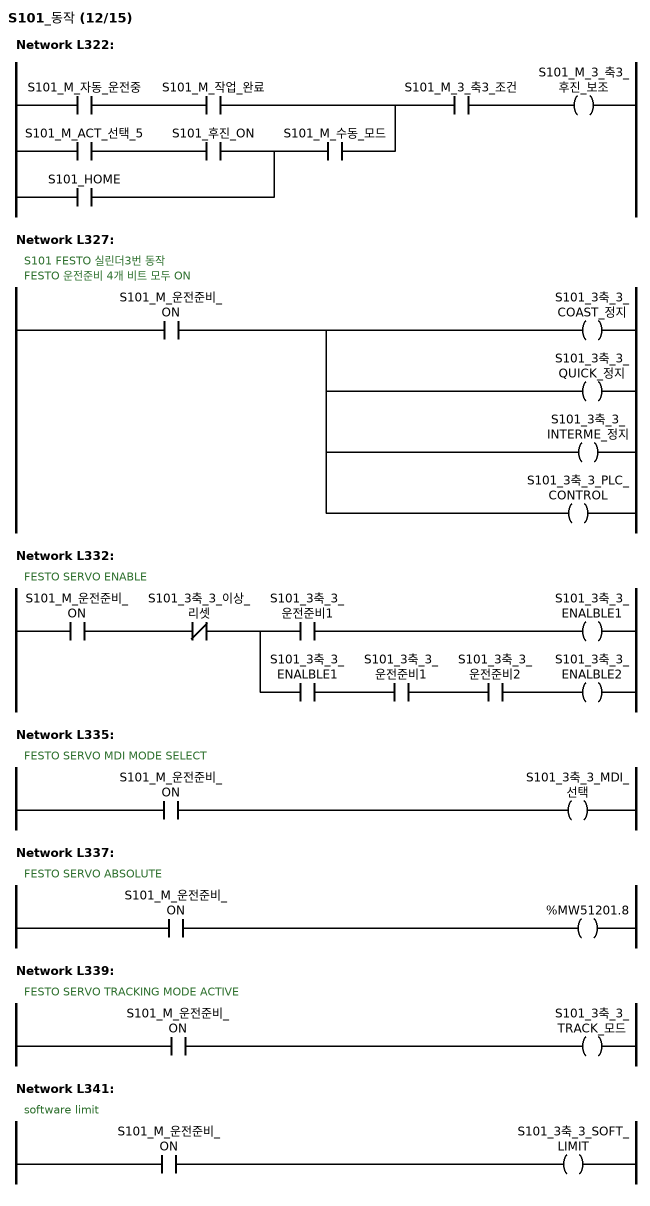
(* [picture p72: S101_동작 rungs L322-L341] *)
(* Rung L322 *)
S101_M_3_축3_후진_보조 := ((S101_M_자동_운전중 AND S101_M_작업_완료) OR (((S101_M_ACT_선택_5 AND S101_후진_ON) OR S101_HOME) AND S101_M_수동_모드)) AND S101_M_3_축3_조건;
(* S101 FESTO 실린더3번 동작 *)
(* FESTO 운전준비 4개 비트 모두 ON *)
(* Rung L327 *)
S101_3축_3_COAST_정지 := S101_M_운전준비_ON;
S101_3축_3_QUICK_정지 := S101_M_운전준비_ON;
S101_3축_3_INTERME_정지 := S101_M_운전준비_ON;
S101_3축_3_PLC_CONTROL := S101_M_운전준비_ON;
(* FESTO SERVO ENABLE *)
(* Rung L332 *)
S101_3축_3_ENALBLE1 := S101_M_운전준비_ON AND NOT S101_3축_3_이상_리셋 AND S101_3축_3_운전준비1;
S101_3축_3_ENALBLE2 := S101_M_운전준비_ON AND NOT S101_3축_3_이상_리셋 AND S101_3축_3_ENALBLE1 AND S101_3축_3_운전준비1 AND S101_3축_3_운전준비2;
(* FESTO SERVO MDI MODE SELECT *)
(* Rung L335 *)
S101_3축_3_MDI_선택 := S101_M_운전준비_ON;
(* FESTO SERVO ABSOLUTE *)
(* Rung L337 *)
%MW51201.8 := S101_M_운전준비_ON;
(* FESTO SERVO TRACKING MODE ACTIVE *)
(* Rung L339 *)
S101_3축_3_TRACK_모드 := S101_M_운전준비_ON;
(* software limit *)
(* Rung L341 *)
S101_3축_3_SOFT_LIMIT := S101_M_운전준비_ON;

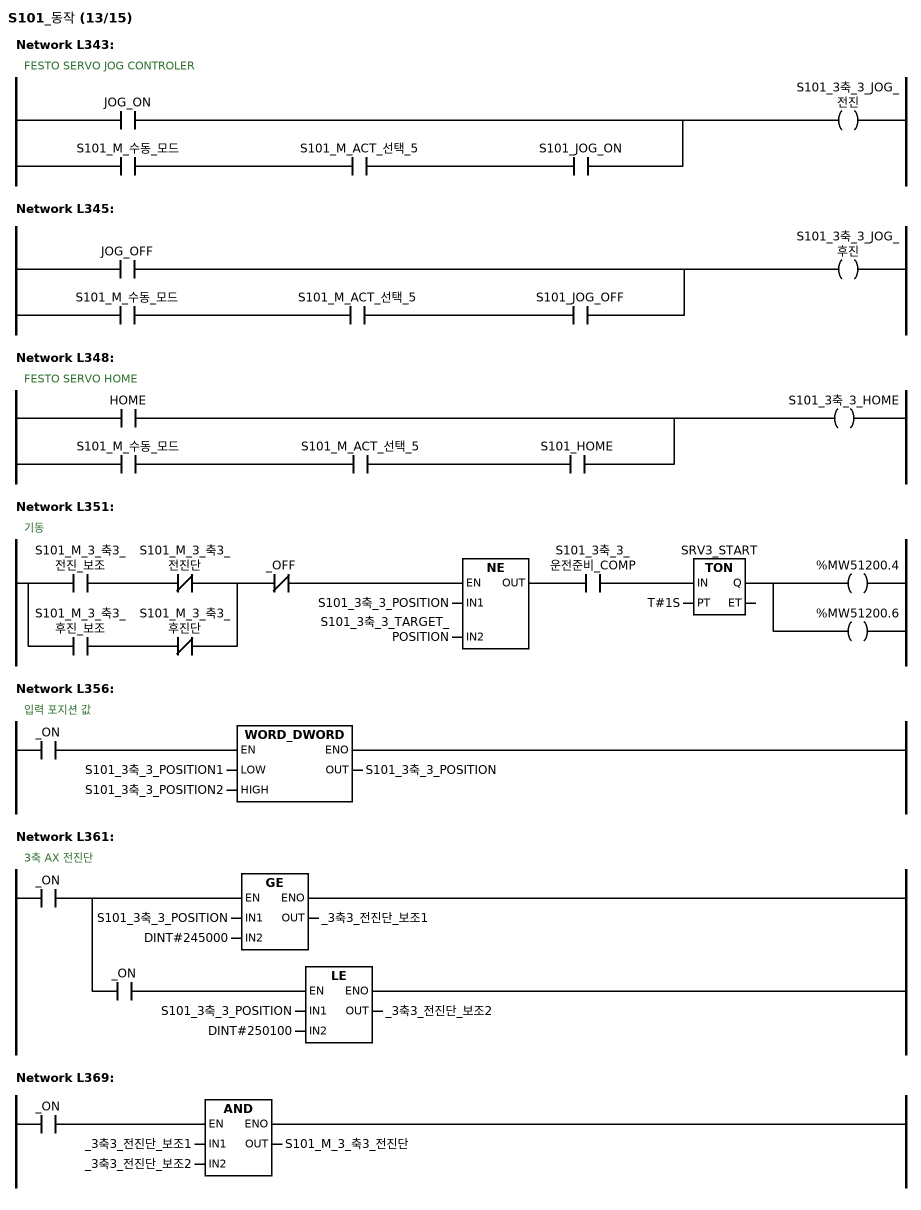
(* FESTO SERVO JOG CONTROLER *)
(* Rung L343 *)
S101_3축_3_JOG_전진 := JOG_ON OR (S101_M_수동_모드 AND S101_M_ACT_선택_5 AND S101_JOG_ON);
(* Rung L345 *)
S101_3축_3_JOG_후진 := JOG_OFF OR (S101_M_수동_모드 AND S101_M_ACT_선택_5 AND S101_JOG_OFF);
(* FESTO SERVO HOME *)
(* Rung L348 *)
S101_3축_3_HOME := HOME OR (S101_M_수동_모드 AND S101_M_ACT_선택_5 AND S101_HOME);
(* 기동 *)
(* Rung L351 *)
IF ((S101_M_3_축3_전진_보조 AND NOT S101_M_3_축3_전진단) OR (S101_M_3_축3_후진_보조 AND NOT S101_M_3_축3_후진단)) AND NOT _OFF THEN
    _t3 := S101_3축_3_POSITION <> S101_3축_3_TARGET_POSITION;
END_IF;
SRV3_START(IN := _t3 AND S101_3축_3_운전준비_COMP, PT := T#1S);
%MW51200.4 := SRV3_START.Q;
%MW51200.6 := SRV3_START.Q;
(* 입력 포지션 값 *)
(* Rung L356 *)
IF _ON THEN
    S101_3축_3_POSITION := WORD_DWORD(LOW := S101_3축_3_POSITION1, HIGH := S101_3축_3_POSITION2);
END_IF;
(* 3축 AX 전진단 *)
(* Rung L361 *)
IF _ON THEN _3축3_전진단_보조1 := S101_3축_3_POSITION >= DINT#245000; END_IF;
IF _ON AND _ON THEN _3축3_전진단_보조2 := S101_3축_3_POSITION <= DINT#250100; END_IF;
(* Rung L369 *)
IF _ON THEN S101_M_3_축3_전진단 := _3축3_전진단_보조1 AND _3축3_전진단_보조2; END_IF;

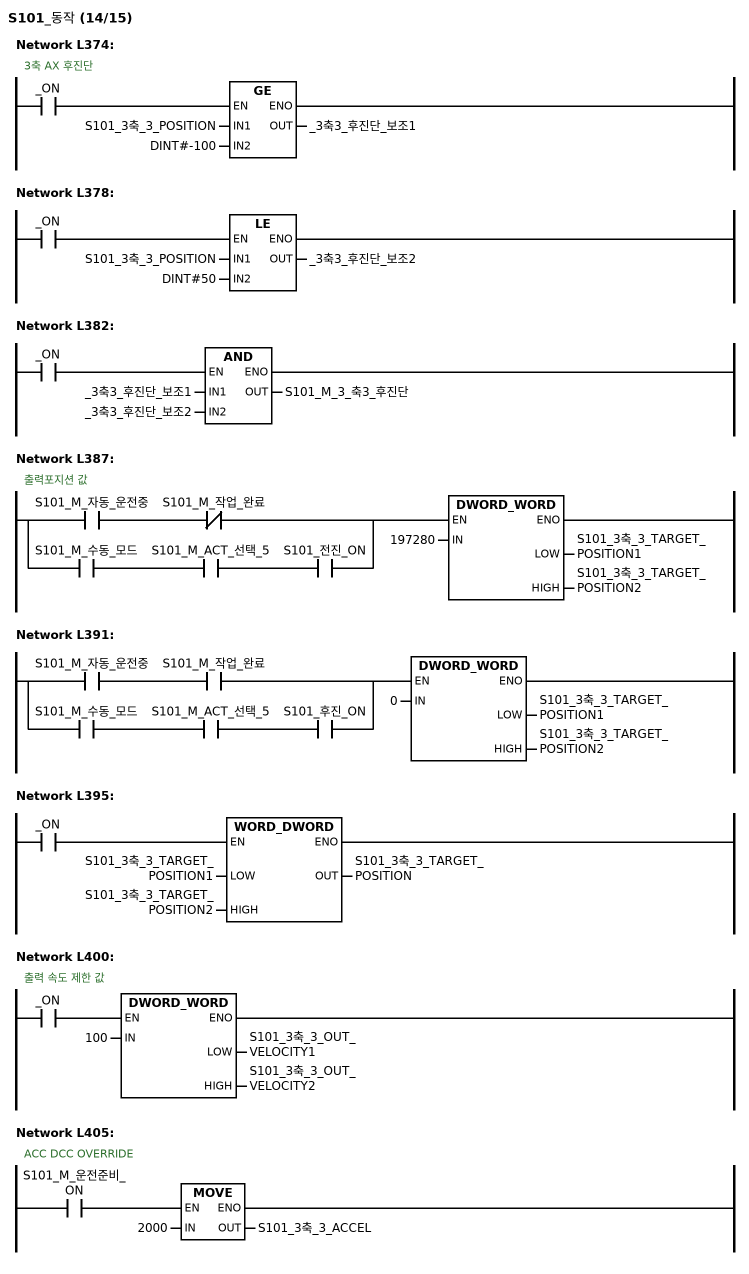
(* 3축 AX 후진단 *)
(* Rung L374 *)
IF _ON THEN _3축3_후진단_보조1 := S101_3축_3_POSITION >= (DINT#-100); END_IF;
(* Rung L378 *)
IF _ON THEN _3축3_후진단_보조2 := S101_3축_3_POSITION <= DINT#50; END_IF;
(* Rung L382 *)
IF _ON THEN S101_M_3_축3_후진단 := _3축3_후진단_보조1 AND _3축3_후진단_보조2; END_IF;
(* 출력포지션 값 *)
(* Rung L387 *)
IF (S101_M_자동_운전중 AND NOT S101_M_작업_완료) OR (S101_M_수동_모드 AND S101_M_ACT_선택_5 AND S101_전진_ON) THEN
    S101_3축_3_TARGET_POSITION1 := DWORD_WORD(IN := 197280, HIGH => S101_3축_3_TARGET_POSITION2);
END_IF;
(* Rung L391 *)
IF (S101_M_자동_운전중 AND S101_M_작업_완료) OR (S101_M_수동_모드 AND S101_M_ACT_선택_5 AND S101_후진_ON) THEN
    S101_3축_3_TARGET_POSITION1 := DWORD_WORD(IN := 0, HIGH => S101_3축_3_TARGET_POSITION2);
END_IF;
(* Rung L395 *)
IF _ON THEN
    S101_3축_3_TARGET_POSITION := WORD_DWORD(LOW := S101_3축_3_TARGET_POSITION1, HIGH := S101_3축_3_TARGET_POSITION2);
END_IF;
(* 출력 속도 제한 값 *)
(* Rung L400 *)
IF _ON THEN S101_3축_3_OUT_VELOCITY1 := DWORD_WORD(IN := 100, HIGH => S101_3축_3_OUT_VELOCITY2); END_IF;
(* ACC DCC OVERRIDE *)
(* Rung L405 *)
IF S101_M_운전준비_ON THEN S101_3축_3_ACCEL := 2000; END_IF;

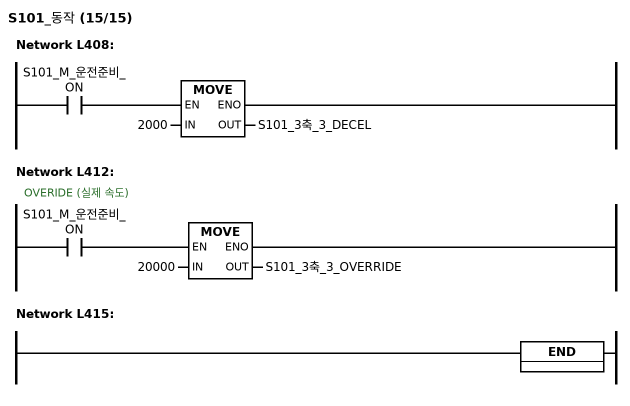
(* Rung L408 *)
IF S101_M_운전준비_ON THEN S101_3축_3_DECEL := 2000; END_IF;
(* OVERIDE (실제 속도) *)
(* Rung L412 *)
IF S101_M_운전준비_ON THEN S101_3축_3_OVERRIDE := 20000; END_IF;
(* Rung L415 *)
END();
END_PROGRAM

PROGRAM S101_LH_APRON_랙방 (* task: 스캔 프로그램 *)
VAR_EXTERNAL
    APRON_LH_RACK1_I_막장감지 : BOOL; (* AT %MW87211.2 *)
    APRON_LH_RACK1_I_종발이감지1 : BOOL; (* AT %MW87211.0 *)
    APRON_LH_RACK1_I_종발이감지2 : BOOL; (* AT %MW87211.1 *)
    APRON_LH_RACK2_I_막장감지 : BOOL; (* AT %MW87211.10 *)
    APRON_LH_RACK2_I_종발이감지1 : BOOL; (* AT %MW87211.8 *)
    APRON_LH_RACK2_I_종발이감지2 : BOOL; (* AT %MW87211.9 *)
    AWAYS_ON : BOOL; (* AT %MW3.1 *)
    OTR_RACK1_I_막장감지 : BOOL; (* AT %MW87020.2 *)
    OTR_RACK1_I_종발이감지1 : BOOL; (* AT %MW87020.0 *)
    OTR_RACK1_I_종발이감지2 : BOOL; (* AT %MW87020.1 *)
    OTR_RACK2_I_막장감지 : BOOL; (* AT %MW87020.10 *)
    OTR_RACK2_I_종발이감지1 : BOOL; (* AT %MW87020.8 *)
    OTR_RACK2_I_종발이감지2 : BOOL; (* AT %MW87020.9 *)
    R101_1_M_RB_PROG_NO : WORD; (* AT %MW20074 *)
    S101_LH_M_APRON_PLT1_FAULT : BOOL; (* AT %MW1200.6 *)
    S101_LH_M_APRON_PLT1_MATCH_OK : BOOL; (* AT %MW1200.5 *)
    S101_LH_M_APRON_PLT1_PLT_NONE : BOOL; (* AT %MW1200.2 *)
    S101_LH_M_APRON_PLT1_PLT_ON : BOOL; (* AT %MW1200.1 *)
    S101_LH_M_APRON_PLT1_PROG_OK : BOOL; (* AT %MW1200.0 *)
    S101_LH_M_APRON_PLT1_로딩완료 : BOOL; (* AT %MW1200.10 *)
    S101_LH_M_APRON_PLT1_제품수량 : WORD; (* AT %MW1224 *)
    S101_LH_M_APRON_PLT1_차종유 : BOOL; (* AT %MW1200.8 *)
    S101_LH_M_APRON_PLT1_차종코드 : WORD; (* AT %MW1216 *)
    S101_LH_M_APRON_PLT1_파트무 : BOOL; (* AT %MW1200.4 *)
    S101_LH_M_APRON_PLT1_파트유 : BOOL; (* AT %MW1200.3 *)
    S101_LH_M_APRON_PLT2_FAULT : BOOL; (* AT %MW1201.6 *)
    S101_LH_M_APRON_PLT2_MATCH_OK : BOOL; (* AT %MW1201.5 *)
    S101_LH_M_APRON_PLT2_PLT_NONE : BOOL; (* AT %MW1201.2 *)
    S101_LH_M_APRON_PLT2_PLT_ON : BOOL; (* AT %MW1201.1 *)
    S101_LH_M_APRON_PLT2_PROG_OK : BOOL; (* AT %MW1201.0 *)
    S101_LH_M_APRON_PLT2_로딩완료 : BOOL; (* AT %MW1201.10 *)
    S101_LH_M_APRON_PLT2_제품수량 : WORD; (* AT %MW1225 *)
    S101_LH_M_APRON_PLT2_차종유 : BOOL; (* AT %MW1201.8 *)
    S101_LH_M_APRON_PLT2_차종코드 : WORD; (* AT %MW1217 *)
    S101_LH_M_APRON_PLT2_파트무 : BOOL; (* AT %MW1201.4 *)
    S101_LH_M_APRON_PLT2_파트유 : BOOL; (* AT %MW1201.3 *)
    전체_M_이상_리셋 : BOOL; (* AT %MW308.2 *) (* 전체 M 이상 리셋 *)
END_VAR
VAR
    INST : TON;
    INST1 : TON;
    INST2 : TON;
    INST3 : TON;
    INST4 : TON;
    INST5 : TON;
    R201_1_M_I_RB_PROG_NO : INT;
    _R101_1_LH_APRON_PLT1_카운터_RST완료 : BOOL;
    _R101_1_LH_APRON_PLT1_카운터_RST요구 : BOOL;
    _R101_1_LH_APRON_PLT2_카운터_RST완료 : BOOL;
    _R101_1_LH_APRON_PLT2_카운터_RST요구 : BOOL;
    _R101_1_LH_PLT1_막장취출완료 : BOOL;
    _R101_1_LH_PLT2_막장취출완료 : BOOL;
    _R101_1_RB_비교_PROG_NO : INT;
    _R201_1_OTR_PLT1_카운터_RST완료 : BOOL;
    _R201_1_OTR_PLT1_카운터_RST요구 : BOOL;
    _R201_1_OTR_PLT2_카운터_RST완료 : BOOL;
    _R201_1_OTR_PLT2_카운터_RST요구 : BOOL;
    _R201_1_PLT1_막장취출완료 : BOOL;
    _R201_1_PLT2_막장취출완료 : BOOL;
    _R201_1_RB_비교_PROG_NO : INT;
    _R201_1_RB_비교_PROG_NO_INT : INT;
    _R201_1_막장취출완료 : BOOL;
    _랙1_제품수량 : INT;
    _랙1_차종코드 : INT;
    _랙2_제품수량 : INT;
    _랙2_차종코드 : INT;
END_VAR
VAR
    _p1 : BOOL;
    _p2 : BOOL;
END_VAR

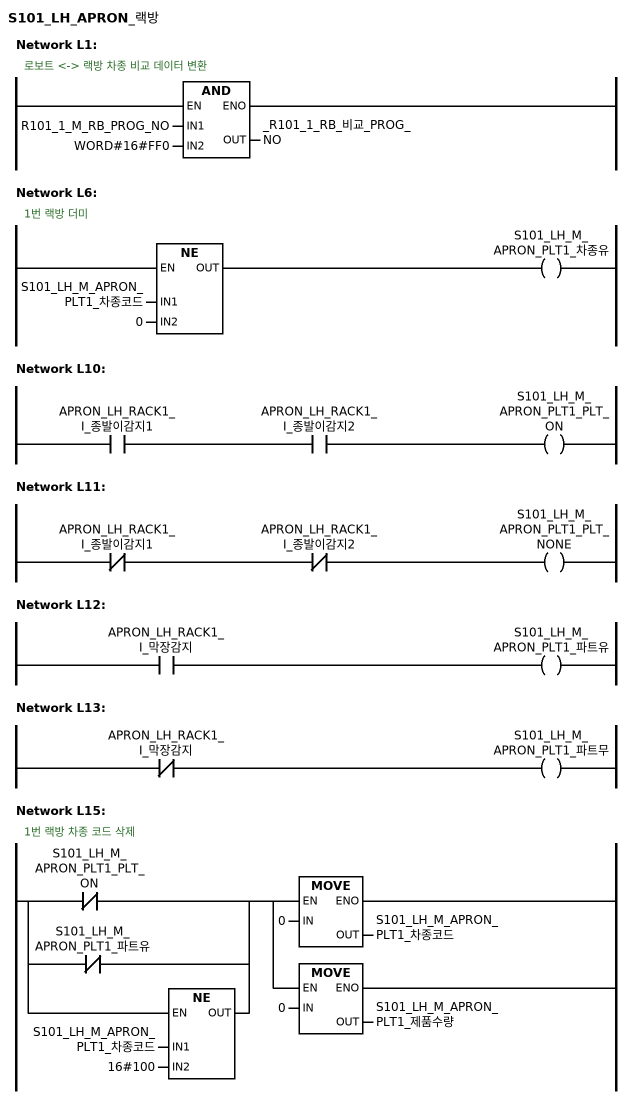
(* 로보트 <-> 랙방 차종 비교 데이터 변환 *)
(* Rung L1 *)
_R101_1_RB_비교_PROG_NO := R101_1_M_RB_PROG_NO AND WORD#16#FF0;
(* 1번 랙방 더미 *)
(* Rung L6 *)
S101_LH_M_APRON_PLT1_차종유 := S101_LH_M_APRON_PLT1_차종코드 <> 0;
(* Rung L10 *)
S101_LH_M_APRON_PLT1_PLT_ON := APRON_LH_RACK1_I_종발이감지1 AND APRON_LH_RACK1_I_종발이감지2;
(* Rung L11 *)
S101_LH_M_APRON_PLT1_PLT_NONE := NOT APRON_LH_RACK1_I_종발이감지1 AND NOT APRON_LH_RACK1_I_종발이감지2;
(* Rung L12 *)
S101_LH_M_APRON_PLT1_파트유 := APRON_LH_RACK1_I_막장감지;
(* Rung L13 *)
S101_LH_M_APRON_PLT1_파트무 := NOT APRON_LH_RACK1_I_막장감지;
(* 1번 랙방 차종 코드 삭제 *)
(* Rung L15 *)
_p1 := NOT S101_LH_M_APRON_PLT1_PLT_ON OR NOT S101_LH_M_APRON_PLT1_파트유 OR (S101_LH_M_APRON_PLT1_차종코드 <> 16#100);
IF _p1 THEN
    S101_LH_M_APRON_PLT1_차종코드 := 0;
    S101_LH_M_APRON_PLT1_제품수량 := 0;
END_IF;
(* 1번 랙방 차종 코드 입력 *)
(* Rung L22: network not rendered *)
(* not connected or not rendered: S101_LH_M_APRON_PLT1_로딩완료, S101_LH_M_APRON_PLT1_PLT_ON, S101_LH_M_APRON_PLT1_파트유, 16#100, S101_LH_M_APRON_PLT1_차종코드, 10, S101_LH_M_APRON_PLT1_제품수량 *)

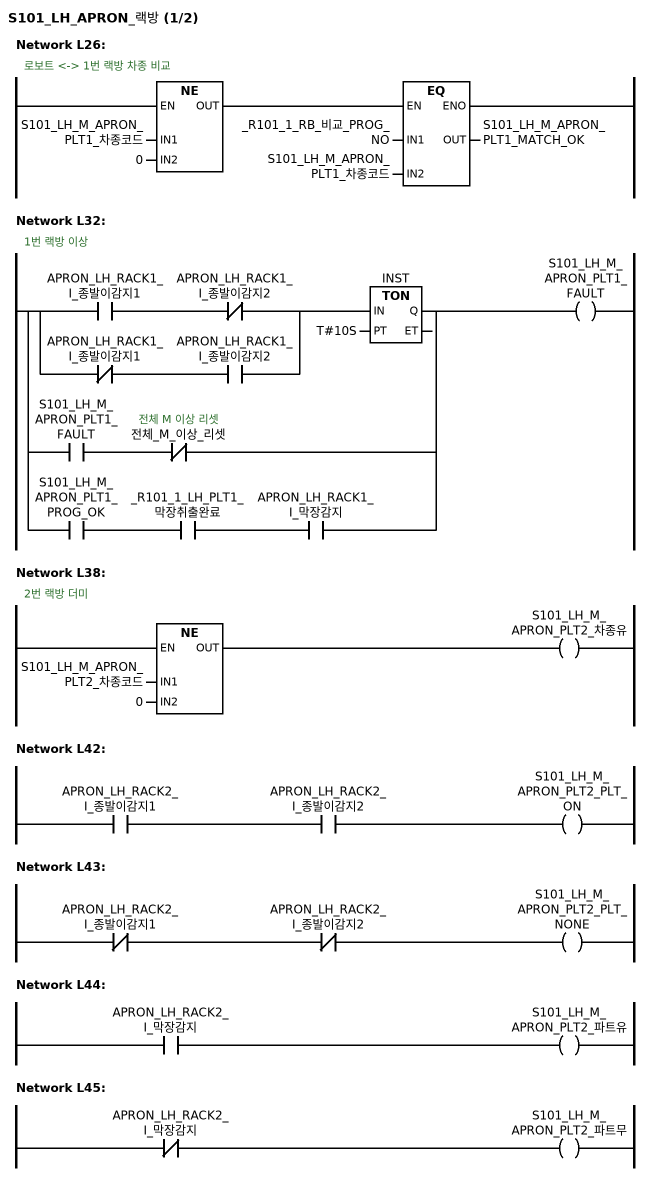
(* 로보트 <-> 1번 랙방 차종 비교 *)
(* Rung L26 *)
IF S101_LH_M_APRON_PLT1_차종코드 <> 0 THEN
    S101_LH_M_APRON_PLT1_MATCH_OK := _R101_1_RB_비교_PROG_NO = S101_LH_M_APRON_PLT1_차종코드;
END_IF;
(* 1번 랙방 이상 *)
(* Rung L32 *)
INST(IN := (APRON_LH_RACK1_I_종발이감지1 AND NOT APRON_LH_RACK1_I_종발이감지2) OR (NOT APRON_LH_RACK1_I_종발이감지1 AND APRON_LH_RACK1_I_종발이감지2), PT := T#10S);
S101_LH_M_APRON_PLT1_FAULT := INST.Q OR (S101_LH_M_APRON_PLT1_FAULT AND NOT 전체_M_이상_리셋) OR (S101_LH_M_APRON_PLT1_PROG_OK AND _R101_1_LH_PLT1_막장취출완료 AND APRON_LH_RACK1_I_막장감지);
(* 2번 랙방 더미 *)
(* Rung L38 *)
S101_LH_M_APRON_PLT2_차종유 := S101_LH_M_APRON_PLT2_차종코드 <> 0;
(* Rung L42 *)
S101_LH_M_APRON_PLT2_PLT_ON := APRON_LH_RACK2_I_종발이감지1 AND APRON_LH_RACK2_I_종발이감지2;
(* Rung L43 *)
S101_LH_M_APRON_PLT2_PLT_NONE := NOT APRON_LH_RACK2_I_종발이감지1 AND NOT APRON_LH_RACK2_I_종발이감지2;
(* Rung L44 *)
S101_LH_M_APRON_PLT2_파트유 := APRON_LH_RACK2_I_막장감지;
(* Rung L45 *)
S101_LH_M_APRON_PLT2_파트무 := NOT APRON_LH_RACK2_I_막장감지;

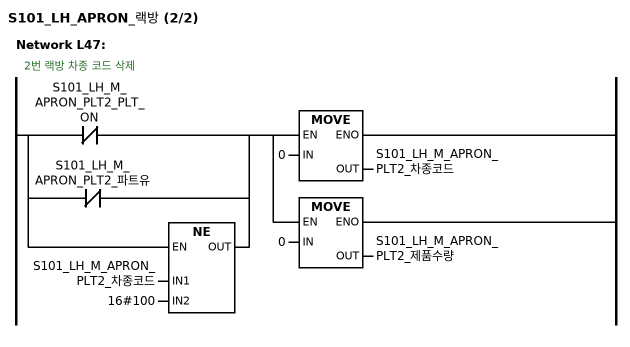
(* 2번 랙방 차종 코드 삭제 *)
(* Rung L47 *)
_p2 := NOT S101_LH_M_APRON_PLT2_PLT_ON OR NOT S101_LH_M_APRON_PLT2_파트유 OR (S101_LH_M_APRON_PLT2_차종코드 <> 16#100);
IF _p2 THEN
    S101_LH_M_APRON_PLT2_차종코드 := 0;
    S101_LH_M_APRON_PLT2_제품수량 := 0;
END_IF;
(* 2번 랙방 차종 코드 입력 *)
(* Rung L54: network not rendered *)
(* not connected or not rendered: S101_LH_M_APRON_PLT2_로딩완료, S101_LH_M_APRON_PLT2_PLT_ON, S101_LH_M_APRON_PLT2_파트유, 16#100, S101_LH_M_APRON_PLT2_차종코드, 10, S101_LH_M_APRON_PLT2_제품수량 *)

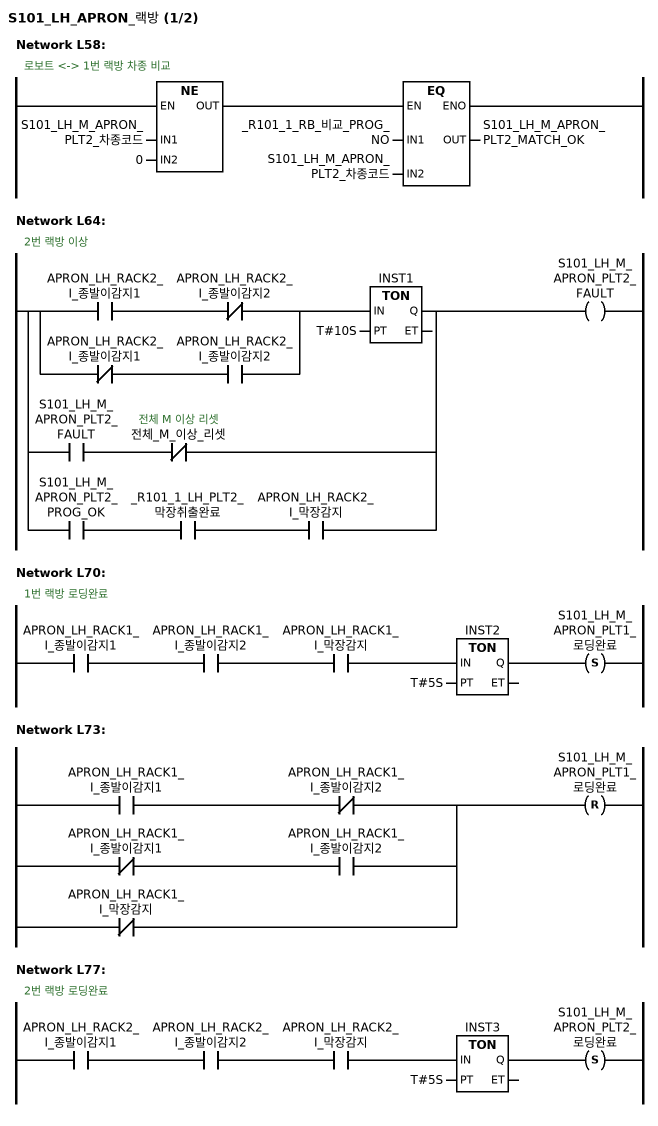
(* 로보트 <-> 1번 랙방 차종 비교 *)
(* Rung L58 *)
IF S101_LH_M_APRON_PLT2_차종코드 <> 0 THEN
    S101_LH_M_APRON_PLT2_MATCH_OK := _R101_1_RB_비교_PROG_NO = S101_LH_M_APRON_PLT2_차종코드;
END_IF;
(* 2번 랙방 이상 *)
(* Rung L64 *)
INST1(IN := (APRON_LH_RACK2_I_종발이감지1 AND NOT APRON_LH_RACK2_I_종발이감지2) OR (NOT APRON_LH_RACK2_I_종발이감지1 AND APRON_LH_RACK2_I_종발이감지2), PT := T#10S);
S101_LH_M_APRON_PLT2_FAULT := INST1.Q OR (S101_LH_M_APRON_PLT2_FAULT AND NOT 전체_M_이상_리셋) OR (S101_LH_M_APRON_PLT2_PROG_OK AND _R101_1_LH_PLT2_막장취출완료 AND APRON_LH_RACK2_I_막장감지);
(* 1번 랙방 로딩완료 *)
(* Rung L70 *)
INST2(IN := APRON_LH_RACK1_I_종발이감지1 AND APRON_LH_RACK1_I_종발이감지2 AND APRON_LH_RACK1_I_막장감지, PT := T#5S);
IF INST2.Q THEN S101_LH_M_APRON_PLT1_로딩완료 := TRUE; END_IF;
(* Rung L73 *)
IF (APRON_LH_RACK1_I_종발이감지1 AND NOT APRON_LH_RACK1_I_종발이감지2) OR (NOT APRON_LH_RACK1_I_종발이감지1 AND APRON_LH_RACK1_I_종발이감지2) OR NOT APRON_LH_RACK1_I_막장감지 THEN
    S101_LH_M_APRON_PLT1_로딩완료 := FALSE;
END_IF;
(* 2번 랙방 로딩완료 *)
(* Rung L77 *)
INST3(IN := APRON_LH_RACK2_I_종발이감지1 AND APRON_LH_RACK2_I_종발이감지2 AND APRON_LH_RACK2_I_막장감지, PT := T#5S);
IF INST3.Q THEN S101_LH_M_APRON_PLT2_로딩완료 := TRUE; END_IF;

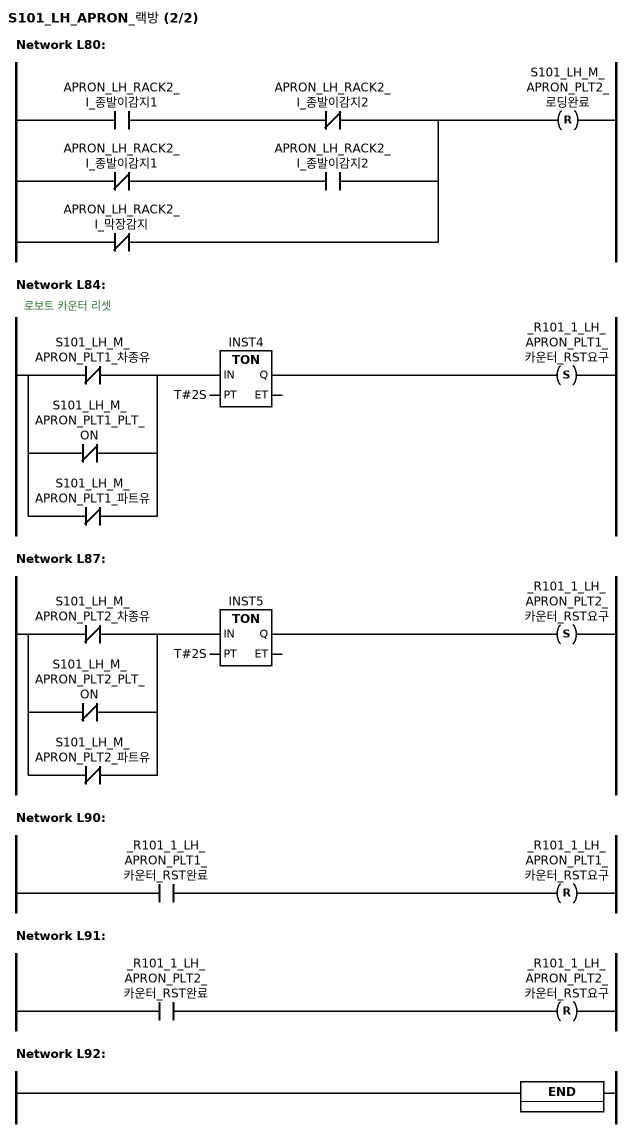
(* Rung L80 *)
IF (APRON_LH_RACK2_I_종발이감지1 AND NOT APRON_LH_RACK2_I_종발이감지2) OR (NOT APRON_LH_RACK2_I_종발이감지1 AND APRON_LH_RACK2_I_종발이감지2) OR NOT APRON_LH_RACK2_I_막장감지 THEN
    S101_LH_M_APRON_PLT2_로딩완료 := FALSE;
END_IF;
(* 로보트 카운터 리셋 *)
(* Rung L84 *)
INST4(IN := NOT S101_LH_M_APRON_PLT1_차종유 OR NOT S101_LH_M_APRON_PLT1_PLT_ON OR NOT S101_LH_M_APRON_PLT1_파트유, PT := T#2S);
IF INST4.Q THEN _R101_1_LH_APRON_PLT1_카운터_RST요구 := TRUE; END_IF;
(* Rung L87 *)
INST5(IN := NOT S101_LH_M_APRON_PLT2_차종유 OR NOT S101_LH_M_APRON_PLT2_PLT_ON OR NOT S101_LH_M_APRON_PLT2_파트유, PT := T#2S);
IF INST5.Q THEN _R101_1_LH_APRON_PLT2_카운터_RST요구 := TRUE; END_IF;
(* Rung L90 *)
IF _R101_1_LH_APRON_PLT1_카운터_RST완료 THEN _R101_1_LH_APRON_PLT1_카운터_RST요구 := FALSE; END_IF;
(* Rung L91 *)
IF _R101_1_LH_APRON_PLT2_카운터_RST완료 THEN _R101_1_LH_APRON_PLT2_카운터_RST요구 := FALSE; END_IF;
(* Rung L92 *)
END();
END_PROGRAM

PROGRAM S101_LH_APRON_랙방_우선순위 (* task: 스캔 프로그램 *)
VAR_EXTERNAL
    S101_LH_M_APRON_PLT1_PLT_ON : BOOL; (* AT %MW1200.1 *)
    S101_LH_M_APRON_PLT1_로딩완료 : BOOL; (* AT %MW1200.10 *)
    S101_LH_M_APRON_PLT1_차종유 : BOOL; (* AT %MW1200.8 *)
    S101_LH_M_APRON_PLT1_파트유 : BOOL; (* AT %MW1200.3 *)
    S101_LH_M_APRON_PLT2_PLT_ON : BOOL; (* AT %MW1201.1 *)
    S101_LH_M_APRON_PLT2_로딩완료 : BOOL; (* AT %MW1201.10 *)
    S101_LH_M_APRON_PLT2_차종유 : BOOL; (* AT %MW1201.8 *)
    S101_LH_M_APRON_PLT2_파트유 : BOOL; (* AT %MW1201.3 *)
    S101_LH_M_APRON_PLT_PRIORITY1 : WORD; (* AT %MW1208 *)
    S101_LH_M_APRON_PLT_PRIORITY2 : WORD; (* AT %MW1209 *)
    S101_LH_M_APRON_PLT_PRIORITY3 : WORD; (* AT %MW1210 *)
    S101_LH_M_APRON_PLT_PRIORITY4 : WORD; (* AT %MW1211 *)
    S101_LH_M_APRON_PLT_PRIORITY5 : WORD; (* AT %MW1212 *)
    S101_LH_M_APRON_PLT_PRIORITY6 : WORD; (* AT %MW1213 *)
    S101_LH_M_APRON_PLT_PRIORITY7 : WORD; (* AT %MW1214 *)
    S101_LH_M_APRON_PLT_PRIORITY8 : WORD; (* AT %MW1215 *)
END_VAR
VAR
    _p1 : BOOL;
    _t2 : BOOL;
    _t3 : BOOL;
    _t4 : BOOL;
    _t5 : BOOL;
    _t6 : BOOL;
    _t7 : BOOL;
    _t8 : BOOL;
    _t9 : BOOL;
    _p10 : BOOL;
    _t11 : BOOL;
    _t12 : BOOL;
    _t13 : BOOL;
    _t14 : BOOL;
    _t15 : BOOL;
    _t16 : BOOL;
    _t17 : BOOL;
    _t18 : BOOL;
END_VAR
(* 랙방번호 우선순위버퍼 전송 *)
(* Rung L1: network not rendered *)
(* not connected or not rendered: S101_LH_M_APRON_PLT1_로딩완료, S101_LH_M_APRON_PLT1_PLT_ON, S101_LH_M_APRON_PLT1_파트유, S101_LH_M_APRON_PLT1_차종유, S101_LH_M_APRON_PLT2_로딩완료, S101_LH_M_APRON_PLT2_PLT_ON, S101_LH_M_APRON_PLT2_파트유, S101_LH_M_APRON_PLT2_차종유, S101_LH_M_APRON_PLT_PRIORITY8, 0, S101_LH_M_APRON_PLT_PRIORITY8, 2, S101_LH_M_APRON_PLT_PRIORITY8 *)
(* 우선순위8->우선순위7 *)
(* Rung L9: network not rendered *)
(* not connected or not rendered: S101_LH_M_APRON_PLT_PRIORITY8, 0, S101_LH_M_APRON_PLT_PRIORITY7, 0, S101_LH_M_APRON_PLT_PRIORITY8, S101_LH_M_APRON_PLT_PRIORITY7, 0, S101_LH_M_APRON_PLT_PRIORITY8 *)
(* 우선순위7->우선순위6 *)
(* Rung L18: network not rendered *)
(* not connected or not rendered: S101_LH_M_APRON_PLT_PRIORITY7, 0, S101_LH_M_APRON_PLT_PRIORITY6, 0, S101_LH_M_APRON_PLT_PRIORITY7, S101_LH_M_APRON_PLT_PRIORITY6, 0, S101_LH_M_APRON_PLT_PRIORITY7 *)
(* 우선순위6->우선순위5 *)
(* Rung L27: network not rendered *)
(* not connected or not rendered: S101_LH_M_APRON_PLT_PRIORITY6, 0, S101_LH_M_APRON_PLT_PRIORITY5, 0, S101_LH_M_APRON_PLT_PRIORITY6, S101_LH_M_APRON_PLT_PRIORITY5, 0, S101_LH_M_APRON_PLT_PRIORITY6 *)
(* 우선순위5->우선순위4 *)
(* Rung L36: network not rendered *)
(* not connected or not rendered: S101_LH_M_APRON_PLT_PRIORITY5, 0, S101_LH_M_APRON_PLT_PRIORITY4, 0, S101_LH_M_APRON_PLT_PRIORITY5, S101_LH_M_APRON_PLT_PRIORITY4, 0, S101_LH_M_APRON_PLT_PRIORITY5 *)
(* 우선순위4->우선순위3 *)
(* Rung L45: network not rendered *)
(* not connected or not rendered: S101_LH_M_APRON_PLT_PRIORITY4, 0, S101_LH_M_APRON_PLT_PRIORITY3, 0, S101_LH_M_APRON_PLT_PRIORITY4, S101_LH_M_APRON_PLT_PRIORITY3, 0, S101_LH_M_APRON_PLT_PRIORITY4 *)
(* 우선순위3->우선순위2 *)
(* Rung L54: network not rendered *)
(* not connected or not rendered: S101_LH_M_APRON_PLT_PRIORITY3, 0, S101_LH_M_APRON_PLT_PRIORITY2, 0, S101_LH_M_APRON_PLT_PRIORITY3, S101_LH_M_APRON_PLT_PRIORITY2, 0, S101_LH_M_APRON_PLT_PRIORITY3 *)
(* 우선순위2->우선순위1 *)
(* Rung L63: network not rendered *)
(* not connected or not rendered: S101_LH_M_APRON_PLT_PRIORITY2, 0, S101_LH_M_APRON_PLT_PRIORITY1, 0, S101_LH_M_APRON_PLT_PRIORITY2, S101_LH_M_APRON_PLT_PRIORITY1, 0, S101_LH_M_APRON_PLT_PRIORITY2 *)

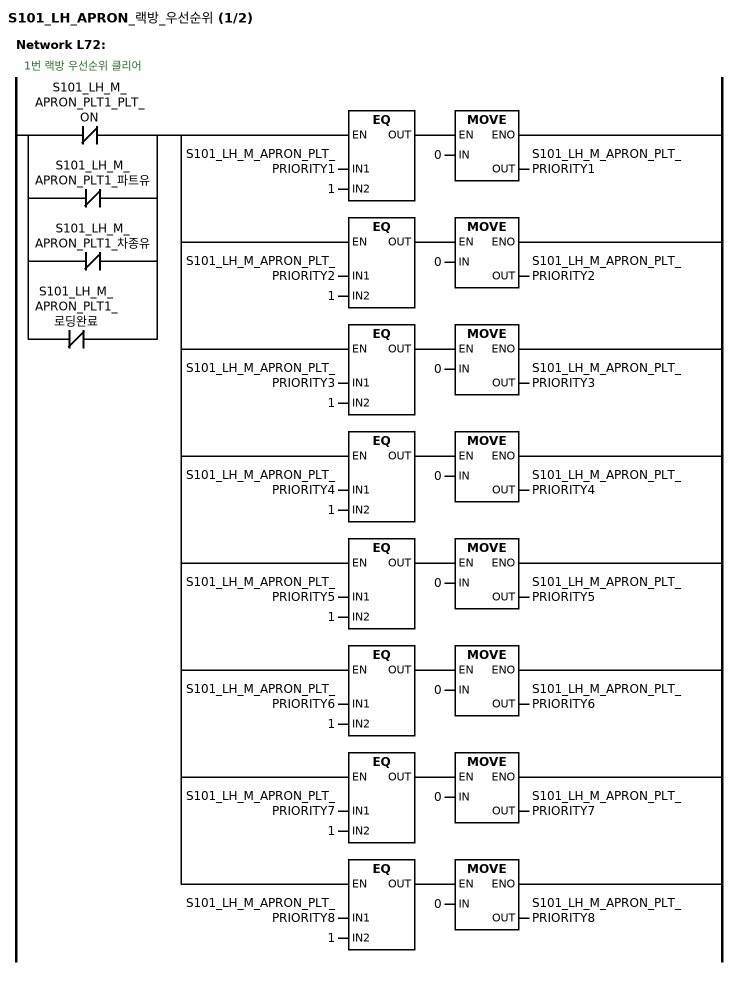
(* 1번 랙방 우선순위 클리어 *)
(* Rung L72 *)
_p1 := NOT S101_LH_M_APRON_PLT1_PLT_ON OR NOT S101_LH_M_APRON_PLT1_파트유 OR NOT S101_LH_M_APRON_PLT1_차종유 OR NOT S101_LH_M_APRON_PLT1_로딩완료;
IF _p1 THEN _t2 := S101_LH_M_APRON_PLT_PRIORITY1 = 1; END_IF;
IF _t2 THEN S101_LH_M_APRON_PLT_PRIORITY1 := 0; END_IF;
IF _p1 THEN _t3 := S101_LH_M_APRON_PLT_PRIORITY2 = 1; END_IF;
IF _t3 THEN S101_LH_M_APRON_PLT_PRIORITY2 := 0; END_IF;
IF _p1 THEN _t4 := S101_LH_M_APRON_PLT_PRIORITY3 = 1; END_IF;
IF _t4 THEN S101_LH_M_APRON_PLT_PRIORITY3 := 0; END_IF;
IF _p1 THEN _t5 := S101_LH_M_APRON_PLT_PRIORITY4 = 1; END_IF;
IF _t5 THEN S101_LH_M_APRON_PLT_PRIORITY4 := 0; END_IF;
IF _p1 THEN _t6 := S101_LH_M_APRON_PLT_PRIORITY5 = 1; END_IF;
IF _t6 THEN S101_LH_M_APRON_PLT_PRIORITY5 := 0; END_IF;
IF _p1 THEN _t7 := S101_LH_M_APRON_PLT_PRIORITY6 = 1; END_IF;
IF _t7 THEN S101_LH_M_APRON_PLT_PRIORITY6 := 0; END_IF;
IF _p1 THEN _t8 := S101_LH_M_APRON_PLT_PRIORITY7 = 1; END_IF;
IF _t8 THEN S101_LH_M_APRON_PLT_PRIORITY7 := 0; END_IF;
IF _p1 THEN _t9 := S101_LH_M_APRON_PLT_PRIORITY8 = 1; END_IF;
IF _t9 THEN S101_LH_M_APRON_PLT_PRIORITY8 := 0; END_IF;

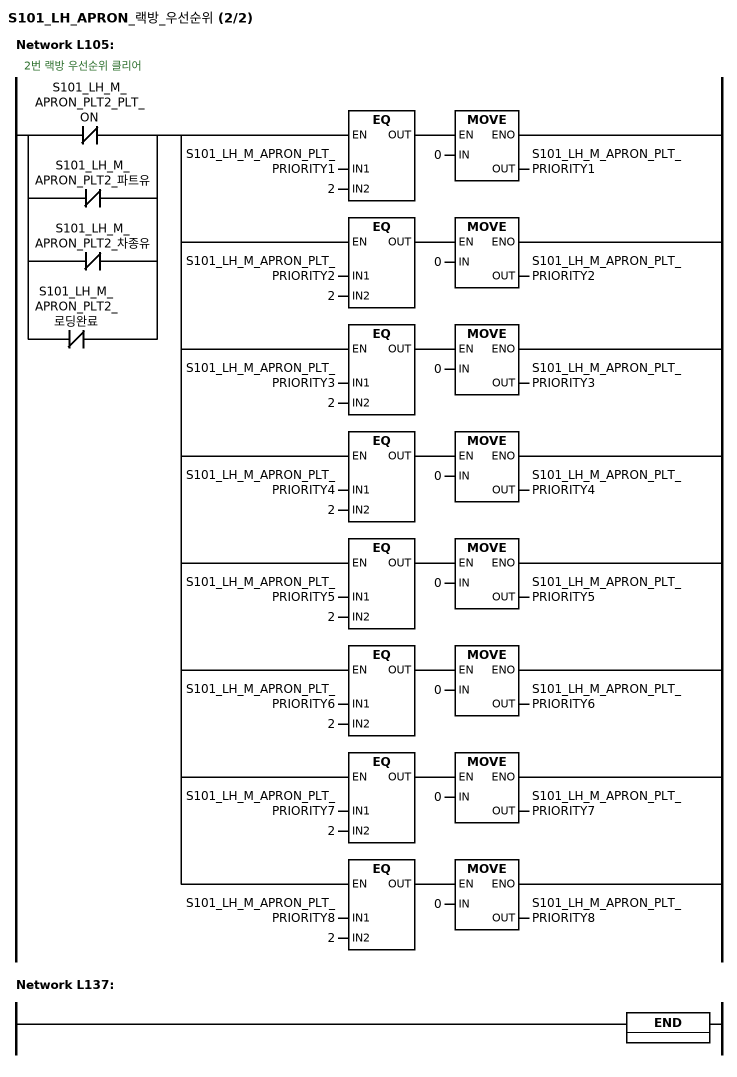
(* 2번 랙방 우선순위 클리어 *)
(* Rung L105 *)
_p10 := NOT S101_LH_M_APRON_PLT2_PLT_ON OR NOT S101_LH_M_APRON_PLT2_파트유 OR NOT S101_LH_M_APRON_PLT2_차종유 OR NOT S101_LH_M_APRON_PLT2_로딩완료;
IF _p10 THEN _t11 := S101_LH_M_APRON_PLT_PRIORITY1 = 2; END_IF;
IF _t11 THEN S101_LH_M_APRON_PLT_PRIORITY1 := 0; END_IF;
IF _p10 THEN _t12 := S101_LH_M_APRON_PLT_PRIORITY2 = 2; END_IF;
IF _t12 THEN S101_LH_M_APRON_PLT_PRIORITY2 := 0; END_IF;
IF _p10 THEN _t13 := S101_LH_M_APRON_PLT_PRIORITY3 = 2; END_IF;
IF _t13 THEN S101_LH_M_APRON_PLT_PRIORITY3 := 0; END_IF;
IF _p10 THEN _t14 := S101_LH_M_APRON_PLT_PRIORITY4 = 2; END_IF;
IF _t14 THEN S101_LH_M_APRON_PLT_PRIORITY4 := 0; END_IF;
IF _p10 THEN _t15 := S101_LH_M_APRON_PLT_PRIORITY5 = 2; END_IF;
IF _t15 THEN S101_LH_M_APRON_PLT_PRIORITY5 := 0; END_IF;
IF _p10 THEN _t16 := S101_LH_M_APRON_PLT_PRIORITY6 = 2; END_IF;
IF _t16 THEN S101_LH_M_APRON_PLT_PRIORITY6 := 0; END_IF;
IF _p10 THEN _t17 := S101_LH_M_APRON_PLT_PRIORITY7 = 2; END_IF;
IF _t17 THEN S101_LH_M_APRON_PLT_PRIORITY7 := 0; END_IF;
IF _p10 THEN _t18 := S101_LH_M_APRON_PLT_PRIORITY8 = 2; END_IF;
IF _t18 THEN S101_LH_M_APRON_PLT_PRIORITY8 := 0; END_IF;
(* Rung L137 *)
END();
END_PROGRAM

PROGRAM S101_RH_APRON_랙방 (* task: 스캔 프로그램 *)
VAR_EXTERNAL
    APRON_RH_RACK1_I_막장감지 : BOOL; (* AT %MW87210.2 *)
    APRON_RH_RACK1_I_종발이감지1 : BOOL; (* AT %MW87210.0 *)
    APRON_RH_RACK1_I_종발이감지2 : BOOL; (* AT %MW87210.1 *)
    APRON_RH_RACK2_I_막장감지 : BOOL; (* AT %MW87210.10 *)
    APRON_RH_RACK2_I_종발이감지1 : BOOL; (* AT %MW87210.8 *)
    APRON_RH_RACK2_I_종발이감지2 : BOOL; (* AT %MW87210.9 *)
    AWAYS_ON : BOOL; (* AT %MW3.1 *)
    OTR_RACK1_I_막장감지 : BOOL; (* AT %MW87020.2 *)
    OTR_RACK1_I_종발이감지1 : BOOL; (* AT %MW87020.0 *)
    OTR_RACK1_I_종발이감지2 : BOOL; (* AT %MW87020.1 *)
    OTR_RACK2_I_막장감지 : BOOL; (* AT %MW87020.10 *)
    OTR_RACK2_I_종발이감지1 : BOOL; (* AT %MW87020.8 *)
    OTR_RACK2_I_종발이감지2 : BOOL; (* AT %MW87020.9 *)
    R101_1_M_RB_PROG_NO : WORD; (* AT %MW20074 *)
    S101_LH_M_APRON_PLT1_FAULT : BOOL; (* AT %MW1200.6 *)
    S101_LH_M_APRON_PLT1_MATCH_OK : BOOL; (* AT %MW1200.5 *)
    S101_LH_M_APRON_PLT1_PLT_NONE : BOOL; (* AT %MW1200.2 *)
    S101_LH_M_APRON_PLT1_PLT_ON : BOOL; (* AT %MW1200.1 *)
    S101_LH_M_APRON_PLT1_PROG_OK : BOOL; (* AT %MW1200.0 *)
    S101_LH_M_APRON_PLT1_로딩완료 : BOOL; (* AT %MW1200.10 *)
    S101_LH_M_APRON_PLT1_제품수량 : WORD; (* AT %MW1224 *)
    S101_LH_M_APRON_PLT1_차종유 : BOOL; (* AT %MW1200.8 *)
    S101_LH_M_APRON_PLT1_차종코드 : WORD; (* AT %MW1216 *)
    S101_LH_M_APRON_PLT1_파트무 : BOOL; (* AT %MW1200.4 *)
    S101_LH_M_APRON_PLT1_파트유 : BOOL; (* AT %MW1200.3 *)
    S101_LH_M_APRON_PLT2_FAULT : BOOL; (* AT %MW1201.6 *)
    S101_LH_M_APRON_PLT2_MATCH_OK : BOOL; (* AT %MW1201.5 *)
    S101_LH_M_APRON_PLT2_PLT_NONE : BOOL; (* AT %MW1201.2 *)
    S101_LH_M_APRON_PLT2_PLT_ON : BOOL; (* AT %MW1201.1 *)
    S101_LH_M_APRON_PLT2_PROG_OK : BOOL; (* AT %MW1201.0 *)
    S101_LH_M_APRON_PLT2_로딩완료 : BOOL; (* AT %MW1201.10 *)
    S101_LH_M_APRON_PLT2_제품수량 : WORD; (* AT %MW1225 *)
    S101_LH_M_APRON_PLT2_차종유 : BOOL; (* AT %MW1201.8 *)
    S101_LH_M_APRON_PLT2_차종코드 : WORD; (* AT %MW1217 *)
    S101_LH_M_APRON_PLT2_파트무 : BOOL; (* AT %MW1201.4 *)
    S101_LH_M_APRON_PLT2_파트유 : BOOL; (* AT %MW1201.3 *)
    S101_RH_M_APRON_PLT1_FAULT : BOOL; (* AT %MW1250.6 *)
    S101_RH_M_APRON_PLT1_MATCH_OK : BOOL; (* AT %MW1250.5 *)
    S101_RH_M_APRON_PLT1_PLT_NONE : BOOL; (* AT %MW1250.2 *)
    S101_RH_M_APRON_PLT1_PLT_ON : BOOL; (* AT %MW1250.1 *)
    S101_RH_M_APRON_PLT1_PROG_OK : BOOL; (* AT %MW1250.0 *)
    S101_RH_M_APRON_PLT1_로딩완료 : BOOL; (* AT %MW1250.10 *)
    S101_RH_M_APRON_PLT1_제품수량 : WORD; (* AT %MW1274 *)
    S101_RH_M_APRON_PLT1_차종유 : BOOL; (* AT %MW1250.8 *)
    S101_RH_M_APRON_PLT1_차종코드 : WORD; (* AT %MW1266 *)
    S101_RH_M_APRON_PLT1_파트무 : BOOL;
    S101_RH_M_APRON_PLT1_파트유 : BOOL; (* AT %MW1250.3 *)
    S101_RH_M_APRON_PLT2_FAULT : BOOL; (* AT %MW1251.6 *)
    S101_RH_M_APRON_PLT2_MATCH_OK : BOOL; (* AT %MW1251.5 *)
    S101_RH_M_APRON_PLT2_PLT_NONE : BOOL; (* AT %MW1251.2 *)
    S101_RH_M_APRON_PLT2_PLT_ON : BOOL; (* AT %MW1251.1 *)
    S101_RH_M_APRON_PLT2_PROG_OK : BOOL; (* AT %MW1251.0 *)
    S101_RH_M_APRON_PLT2_로딩완료 : BOOL; (* AT %MW1251.10 *)
    S101_RH_M_APRON_PLT2_제품수량 : WORD; (* AT %MW1275 *)
    S101_RH_M_APRON_PLT2_차종유 : BOOL; (* AT %MW1251.8 *)
    S101_RH_M_APRON_PLT2_차종코드 : WORD; (* AT %MW1267 *)
    S101_RH_M_APRON_PLT2_파트무 : BOOL; (* AT %MW1251.4 *)
    S101_RH_M_APRON_PLT2_파트유 : BOOL; (* AT %MW1251.3 *)
    전체_M_이상_리셋 : BOOL; (* AT %MW308.2 *) (* 전체 M 이상 리셋 *)
END_VAR
VAR
    INST : TON;
    INST1 : TON;
    INST2 : TON;
    INST3 : TON;
    INST4 : TON;
    INST5 : TON;
    R201_1_M_I_RB_PROG_NO : INT;
    _R101_1_RB_비교_PROG_NO : INT;
    _R101_1_RH_APRON_PLT1_카운터_RST완료 : BOOL;
    _R101_1_RH_APRON_PLT1_카운터_RST요구 : BOOL;
    _R101_1_RH_APRON_PLT2_카운터_RST완료 : BOOL;
    _R101_1_RH_APRON_PLT2_카운터_RST요구 : BOOL;
    _R101_1_RH_PLT1_막장취출완료 : BOOL;
    _R101_1_RH_PLT2_막장취출완료 : BOOL;
    _R201_1_OTR_PLT1_카운터_RST완료 : BOOL;
    _R201_1_OTR_PLT1_카운터_RST요구 : BOOL;
    _R201_1_OTR_PLT2_카운터_RST완료 : BOOL;
    _R201_1_OTR_PLT2_카운터_RST요구 : BOOL;
    _R201_1_PLT1_막장취출완료 : BOOL;
    _R201_1_PLT2_막장취출완료 : BOOL;
    _R201_1_RB_비교_PROG_NO : INT;
    _R201_1_RB_비교_PROG_NO_INT : INT;
    _R201_1_막장취출완료 : BOOL;
    _랙1_제품수량 : INT;
    _랙1_차종코드 : INT;
    _랙2_제품수량 : INT;
    _랙2_차종코드 : INT;
END_VAR
VAR
    _p1 : BOOL;
    _p2 : BOOL;
END_VAR

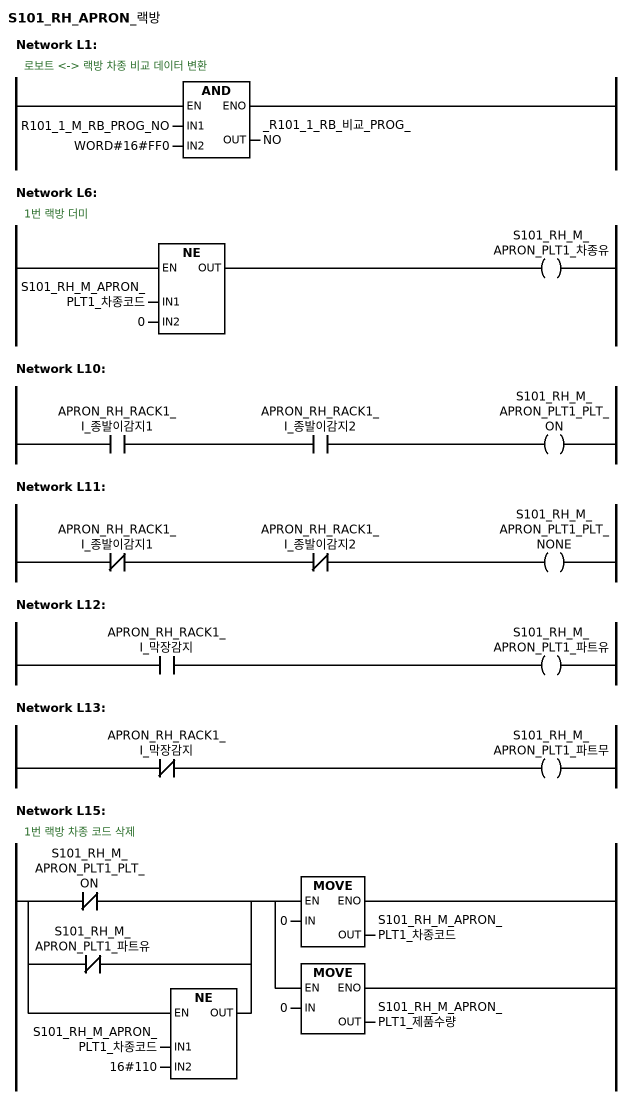
(* 로보트 <-> 랙방 차종 비교 데이터 변환 *)
(* Rung L1 *)
_R101_1_RB_비교_PROG_NO := R101_1_M_RB_PROG_NO AND WORD#16#FF0;
(* 1번 랙방 더미 *)
(* Rung L6 *)
S101_RH_M_APRON_PLT1_차종유 := S101_RH_M_APRON_PLT1_차종코드 <> 0;
(* Rung L10 *)
S101_RH_M_APRON_PLT1_PLT_ON := APRON_RH_RACK1_I_종발이감지1 AND APRON_RH_RACK1_I_종발이감지2;
(* Rung L11 *)
S101_RH_M_APRON_PLT1_PLT_NONE := NOT APRON_RH_RACK1_I_종발이감지1 AND NOT APRON_RH_RACK1_I_종발이감지2;
(* Rung L12 *)
S101_RH_M_APRON_PLT1_파트유 := APRON_RH_RACK1_I_막장감지;
(* Rung L13 *)
S101_RH_M_APRON_PLT1_파트무 := NOT APRON_RH_RACK1_I_막장감지;
(* 1번 랙방 차종 코드 삭제 *)
(* Rung L15 *)
_p1 := NOT S101_RH_M_APRON_PLT1_PLT_ON OR NOT S101_RH_M_APRON_PLT1_파트유 OR (S101_RH_M_APRON_PLT1_차종코드 <> 16#110);
IF _p1 THEN
    S101_RH_M_APRON_PLT1_차종코드 := 0;
    S101_RH_M_APRON_PLT1_제품수량 := 0;
END_IF;
(* 1번 랙방 차종 코드 입력 *)
(* Rung L22: network not rendered *)
(* not connected or not rendered: S101_RH_M_APRON_PLT1_로딩완료, S101_RH_M_APRON_PLT1_PLT_ON, S101_RH_M_APRON_PLT1_파트유, 16#110, S101_RH_M_APRON_PLT1_차종코드, 10, S101_RH_M_APRON_PLT1_제품수량 *)

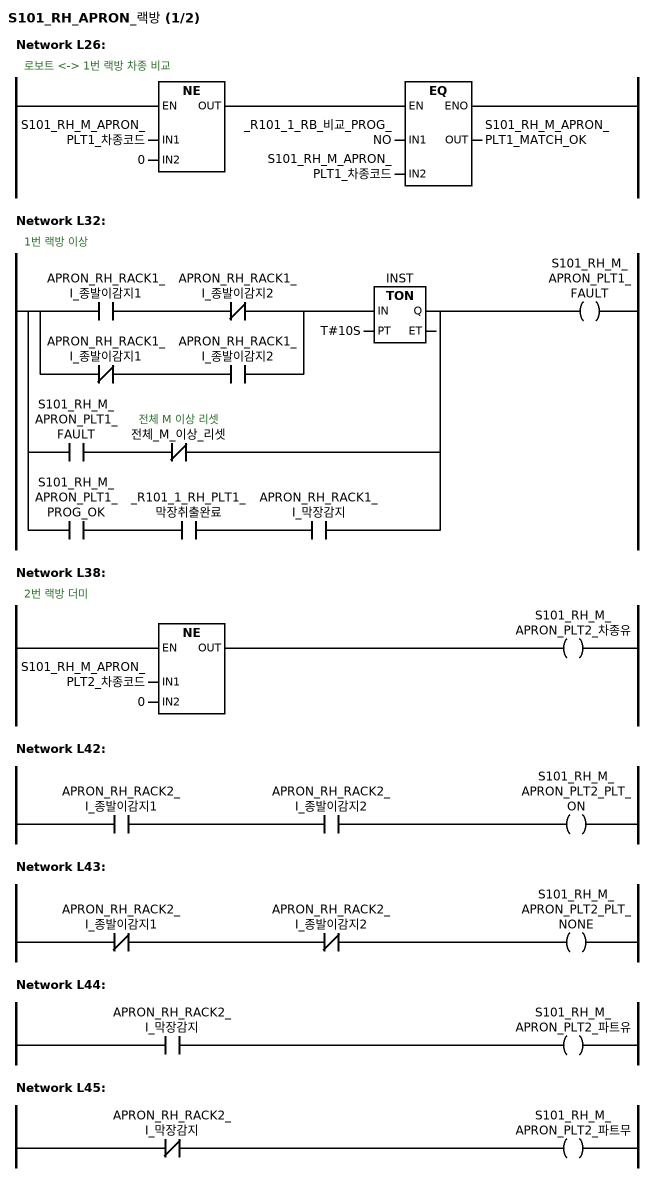
(* 로보트 <-> 1번 랙방 차종 비교 *)
(* Rung L26 *)
IF S101_RH_M_APRON_PLT1_차종코드 <> 0 THEN
    S101_RH_M_APRON_PLT1_MATCH_OK := _R101_1_RB_비교_PROG_NO = S101_RH_M_APRON_PLT1_차종코드;
END_IF;
(* 1번 랙방 이상 *)
(* Rung L32 *)
INST(IN := (APRON_RH_RACK1_I_종발이감지1 AND NOT APRON_RH_RACK1_I_종발이감지2) OR (NOT APRON_RH_RACK1_I_종발이감지1 AND APRON_RH_RACK1_I_종발이감지2), PT := T#10S);
S101_RH_M_APRON_PLT1_FAULT := INST.Q OR (S101_RH_M_APRON_PLT1_FAULT AND NOT 전체_M_이상_리셋) OR (S101_RH_M_APRON_PLT1_PROG_OK AND _R101_1_RH_PLT1_막장취출완료 AND APRON_RH_RACK1_I_막장감지);
(* 2번 랙방 더미 *)
(* Rung L38 *)
S101_RH_M_APRON_PLT2_차종유 := S101_RH_M_APRON_PLT2_차종코드 <> 0;
(* Rung L42 *)
S101_RH_M_APRON_PLT2_PLT_ON := APRON_RH_RACK2_I_종발이감지1 AND APRON_RH_RACK2_I_종발이감지2;
(* Rung L43 *)
S101_RH_M_APRON_PLT2_PLT_NONE := NOT APRON_RH_RACK2_I_종발이감지1 AND NOT APRON_RH_RACK2_I_종발이감지2;
(* Rung L44 *)
S101_RH_M_APRON_PLT2_파트유 := APRON_RH_RACK2_I_막장감지;
(* Rung L45 *)
S101_RH_M_APRON_PLT2_파트무 := NOT APRON_RH_RACK2_I_막장감지;

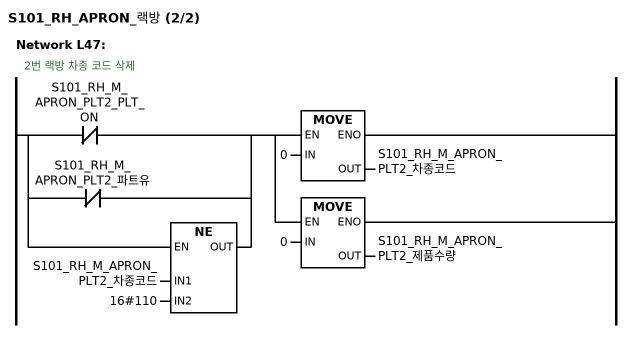
(* 2번 랙방 차종 코드 삭제 *)
(* Rung L47 *)
_p2 := NOT S101_RH_M_APRON_PLT2_PLT_ON OR NOT S101_RH_M_APRON_PLT2_파트유 OR (S101_RH_M_APRON_PLT2_차종코드 <> 16#110);
IF _p2 THEN
    S101_RH_M_APRON_PLT2_차종코드 := 0;
    S101_RH_M_APRON_PLT2_제품수량 := 0;
END_IF;
(* 2번 랙방 차종 코드 입력 *)
(* Rung L54: network not rendered *)
(* not connected or not rendered: S101_RH_M_APRON_PLT2_로딩완료, S101_RH_M_APRON_PLT2_PLT_ON, S101_RH_M_APRON_PLT2_파트유, 16#110, S101_RH_M_APRON_PLT2_차종코드, 10, S101_RH_M_APRON_PLT2_제품수량 *)

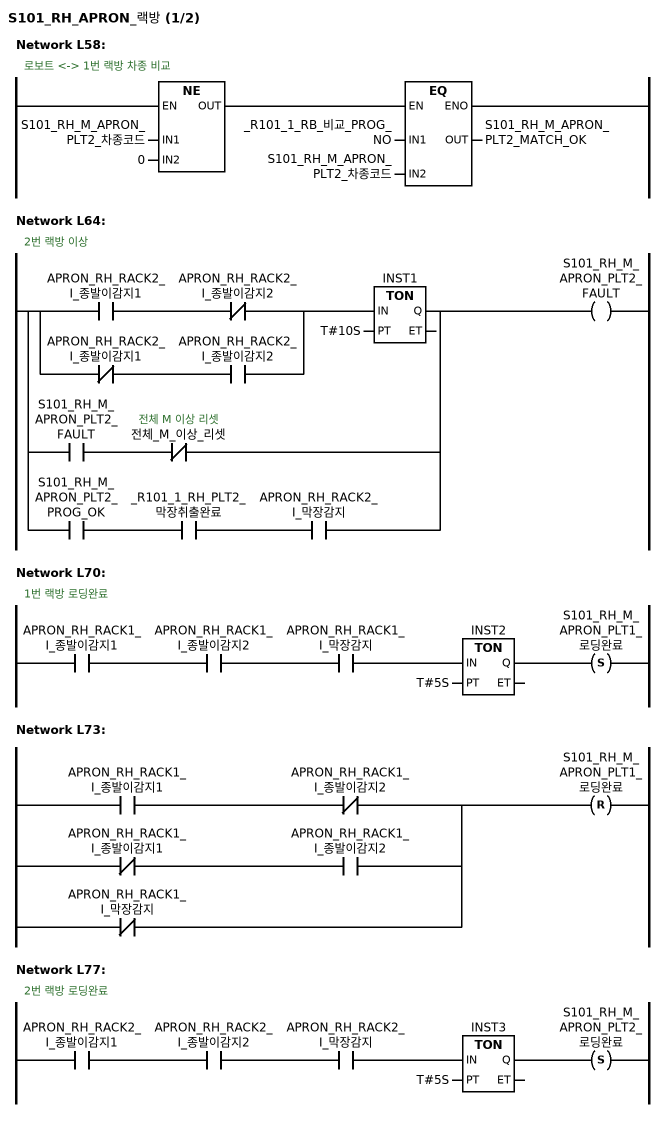
(* 로보트 <-> 1번 랙방 차종 비교 *)
(* Rung L58 *)
IF S101_RH_M_APRON_PLT2_차종코드 <> 0 THEN
    S101_RH_M_APRON_PLT2_MATCH_OK := _R101_1_RB_비교_PROG_NO = S101_RH_M_APRON_PLT2_차종코드;
END_IF;
(* 2번 랙방 이상 *)
(* Rung L64 *)
INST1(IN := (APRON_RH_RACK2_I_종발이감지1 AND NOT APRON_RH_RACK2_I_종발이감지2) OR (NOT APRON_RH_RACK2_I_종발이감지1 AND APRON_RH_RACK2_I_종발이감지2), PT := T#10S);
S101_RH_M_APRON_PLT2_FAULT := INST1.Q OR (S101_RH_M_APRON_PLT2_FAULT AND NOT 전체_M_이상_리셋) OR (S101_RH_M_APRON_PLT2_PROG_OK AND _R101_1_RH_PLT2_막장취출완료 AND APRON_RH_RACK2_I_막장감지);
(* 1번 랙방 로딩완료 *)
(* Rung L70 *)
INST2(IN := APRON_RH_RACK1_I_종발이감지1 AND APRON_RH_RACK1_I_종발이감지2 AND APRON_RH_RACK1_I_막장감지, PT := T#5S);
IF INST2.Q THEN S101_RH_M_APRON_PLT1_로딩완료 := TRUE; END_IF;
(* Rung L73 *)
IF (APRON_RH_RACK1_I_종발이감지1 AND NOT APRON_RH_RACK1_I_종발이감지2) OR (NOT APRON_RH_RACK1_I_종발이감지1 AND APRON_RH_RACK1_I_종발이감지2) OR NOT APRON_RH_RACK1_I_막장감지 THEN
    S101_RH_M_APRON_PLT1_로딩완료 := FALSE;
END_IF;
(* 2번 랙방 로딩완료 *)
(* Rung L77 *)
INST3(IN := APRON_RH_RACK2_I_종발이감지1 AND APRON_RH_RACK2_I_종발이감지2 AND APRON_RH_RACK2_I_막장감지, PT := T#5S);
IF INST3.Q THEN S101_RH_M_APRON_PLT2_로딩완료 := TRUE; END_IF;

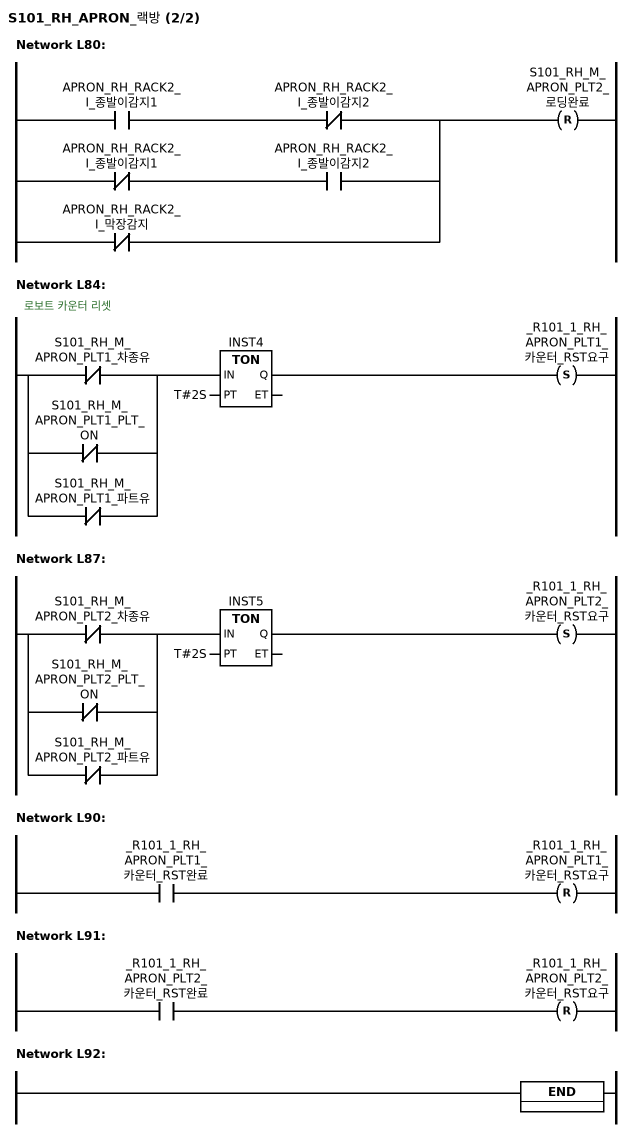
(* Rung L80 *)
IF (APRON_RH_RACK2_I_종발이감지1 AND NOT APRON_RH_RACK2_I_종발이감지2) OR (NOT APRON_RH_RACK2_I_종발이감지1 AND APRON_RH_RACK2_I_종발이감지2) OR NOT APRON_RH_RACK2_I_막장감지 THEN
    S101_RH_M_APRON_PLT2_로딩완료 := FALSE;
END_IF;
(* 로보트 카운터 리셋 *)
(* Rung L84 *)
INST4(IN := NOT S101_RH_M_APRON_PLT1_차종유 OR NOT S101_RH_M_APRON_PLT1_PLT_ON OR NOT S101_RH_M_APRON_PLT1_파트유, PT := T#2S);
IF INST4.Q THEN _R101_1_RH_APRON_PLT1_카운터_RST요구 := TRUE; END_IF;
(* Rung L87 *)
INST5(IN := NOT S101_RH_M_APRON_PLT2_차종유 OR NOT S101_RH_M_APRON_PLT2_PLT_ON OR NOT S101_RH_M_APRON_PLT2_파트유, PT := T#2S);
IF INST5.Q THEN _R101_1_RH_APRON_PLT2_카운터_RST요구 := TRUE; END_IF;
(* Rung L90 *)
IF _R101_1_RH_APRON_PLT1_카운터_RST완료 THEN _R101_1_RH_APRON_PLT1_카운터_RST요구 := FALSE; END_IF;
(* Rung L91 *)
IF _R101_1_RH_APRON_PLT2_카운터_RST완료 THEN _R101_1_RH_APRON_PLT2_카운터_RST요구 := FALSE; END_IF;
(* Rung L92 *)
END();
END_PROGRAM

PROGRAM S101_RH_APRON_랙방_우선순위 (* task: 스캔 프로그램 *)
VAR_EXTERNAL
    S101_LH_M_APRON_PLT1_PLT_ON : BOOL; (* AT %MW1200.1 *)
    S101_LH_M_APRON_PLT1_로딩완료 : BOOL; (* AT %MW1200.10 *)
    S101_LH_M_APRON_PLT1_차종유 : BOOL; (* AT %MW1200.8 *)
    S101_LH_M_APRON_PLT1_파트유 : BOOL; (* AT %MW1200.3 *)
    S101_LH_M_APRON_PLT2_PLT_ON : BOOL; (* AT %MW1201.1 *)
    S101_LH_M_APRON_PLT2_로딩완료 : BOOL; (* AT %MW1201.10 *)
    S101_LH_M_APRON_PLT2_차종유 : BOOL; (* AT %MW1201.8 *)
    S101_LH_M_APRON_PLT2_파트유 : BOOL; (* AT %MW1201.3 *)
    S101_LH_M_APRON_PLT_PRIORITY1 : WORD; (* AT %MW1208 *)
    S101_LH_M_APRON_PLT_PRIORITY2 : WORD; (* AT %MW1209 *)
    S101_LH_M_APRON_PLT_PRIORITY3 : WORD; (* AT %MW1210 *)
    S101_LH_M_APRON_PLT_PRIORITY4 : WORD; (* AT %MW1211 *)
    S101_LH_M_APRON_PLT_PRIORITY5 : WORD; (* AT %MW1212 *)
    S101_LH_M_APRON_PLT_PRIORITY6 : WORD; (* AT %MW1213 *)
    S101_LH_M_APRON_PLT_PRIORITY7 : WORD; (* AT %MW1214 *)
    S101_LH_M_APRON_PLT_PRIORITY8 : WORD; (* AT %MW1215 *)
    S101_RH_M_APRON_PLT1_PLT_ON : BOOL; (* AT %MW1250.1 *)
    S101_RH_M_APRON_PLT1_로딩완료 : BOOL; (* AT %MW1250.10 *)
    S101_RH_M_APRON_PLT1_차종유 : BOOL; (* AT %MW1250.8 *)
    S101_RH_M_APRON_PLT1_파트유 : BOOL; (* AT %MW1250.3 *)
    S101_RH_M_APRON_PLT2_PLT_ON : BOOL; (* AT %MW1251.1 *)
    S101_RH_M_APRON_PLT2_로딩완료 : BOOL; (* AT %MW1251.10 *)
    S101_RH_M_APRON_PLT2_차종유 : BOOL; (* AT %MW1251.8 *)
    S101_RH_M_APRON_PLT2_파트유 : BOOL; (* AT %MW1251.3 *)
    S101_RH_M_APRON_PLT_PRIORITY1 : WORD; (* AT %MW1258 *)
    S101_RH_M_APRON_PLT_PRIORITY2 : WORD; (* AT %MW1259 *)
    S101_RH_M_APRON_PLT_PRIORITY3 : WORD; (* AT %MW1260 *)
    S101_RH_M_APRON_PLT_PRIORITY4 : WORD; (* AT %MW1261 *)
    S101_RH_M_APRON_PLT_PRIORITY5 : WORD; (* AT %MW1262 *)
    S101_RH_M_APRON_PLT_PRIORITY6 : WORD; (* AT %MW1263 *)
    S101_RH_M_APRON_PLT_PRIORITY7 : WORD; (* AT %MW1264 *)
    S101_RH_M_APRON_PLT_PRIORITY8 : WORD; (* AT %MW1265 *)
END_VAR
VAR
    _p1 : BOOL;
    _t2 : BOOL;
    _t3 : BOOL;
    _t4 : BOOL;
    _t5 : BOOL;
    _t6 : BOOL;
    _t7 : BOOL;
    _t8 : BOOL;
    _t9 : BOOL;
    _p10 : BOOL;
    _t11 : BOOL;
    _t12 : BOOL;
    _t13 : BOOL;
    _t14 : BOOL;
    _t15 : BOOL;
    _t16 : BOOL;
    _t17 : BOOL;
    _t18 : BOOL;
END_VAR
(* 랙방번호 우선순위버퍼 전송 *)
(* Rung L1: network not rendered *)
(* not connected or not rendered: S101_RH_M_APRON_PLT1_로딩완료, S101_RH_M_APRON_PLT1_PLT_ON, S101_RH_M_APRON_PLT1_파트유, S101_RH_M_APRON_PLT1_차종유, S101_RH_M_APRON_PLT2_로딩완료, S101_RH_M_APRON_PLT2_PLT_ON, S101_RH_M_APRON_PLT2_파트유, S101_RH_M_APRON_PLT2_차종유, S101_RH_M_APRON_PLT_PRIORITY8, 0, S101_RH_M_APRON_PLT_PRIORITY8, 2, S101_RH_M_APRON_PLT_PRIORITY8 *)
(* 우선순위8->우선순위7 *)
(* Rung L9: network not rendered *)
(* not connected or not rendered: S101_RH_M_APRON_PLT_PRIORITY8, 0, S101_RH_M_APRON_PLT_PRIORITY7, 0, S101_RH_M_APRON_PLT_PRIORITY8, S101_RH_M_APRON_PLT_PRIORITY7, 0, S101_RH_M_APRON_PLT_PRIORITY8 *)
(* 우선순위7->우선순위6 *)
(* Rung L18: network not rendered *)
(* not connected or not rendered: S101_RH_M_APRON_PLT_PRIORITY7, 0, S101_RH_M_APRON_PLT_PRIORITY6, 0, S101_RH_M_APRON_PLT_PRIORITY7, S101_RH_M_APRON_PLT_PRIORITY6, 0, S101_RH_M_APRON_PLT_PRIORITY7 *)
(* 우선순위6->우선순위5 *)
(* Rung L27: network not rendered *)
(* not connected or not rendered: S101_RH_M_APRON_PLT_PRIORITY6, 0, S101_RH_M_APRON_PLT_PRIORITY5, 0, S101_RH_M_APRON_PLT_PRIORITY6, S101_RH_M_APRON_PLT_PRIORITY5, 0, S101_RH_M_APRON_PLT_PRIORITY6 *)
(* 우선순위5->우선순위4 *)
(* Rung L36: network not rendered *)
(* not connected or not rendered: S101_RH_M_APRON_PLT_PRIORITY5, 0, S101_RH_M_APRON_PLT_PRIORITY4, 0, S101_RH_M_APRON_PLT_PRIORITY5, S101_RH_M_APRON_PLT_PRIORITY4, 0, S101_RH_M_APRON_PLT_PRIORITY5 *)
(* 우선순위4->우선순위3 *)
(* Rung L45: network not rendered *)
(* not connected or not rendered: S101_RH_M_APRON_PLT_PRIORITY4, 0, S101_RH_M_APRON_PLT_PRIORITY3, 0, S101_RH_M_APRON_PLT_PRIORITY4, S101_RH_M_APRON_PLT_PRIORITY3, 0, S101_RH_M_APRON_PLT_PRIORITY4 *)
(* 우선순위3->우선순위2 *)
(* Rung L54: network not rendered *)
(* not connected or not rendered: S101_RH_M_APRON_PLT_PRIORITY3, 0, S101_RH_M_APRON_PLT_PRIORITY2, 0, S101_RH_M_APRON_PLT_PRIORITY3, S101_RH_M_APRON_PLT_PRIORITY2, 0, S101_RH_M_APRON_PLT_PRIORITY3 *)
(* 우선순위2->우선순위1 *)
(* Rung L63: network not rendered *)
(* not connected or not rendered: S101_RH_M_APRON_PLT_PRIORITY2, 0, S101_RH_M_APRON_PLT_PRIORITY1, 0, S101_RH_M_APRON_PLT_PRIORITY2, S101_RH_M_APRON_PLT_PRIORITY1, 0, S101_RH_M_APRON_PLT_PRIORITY2 *)

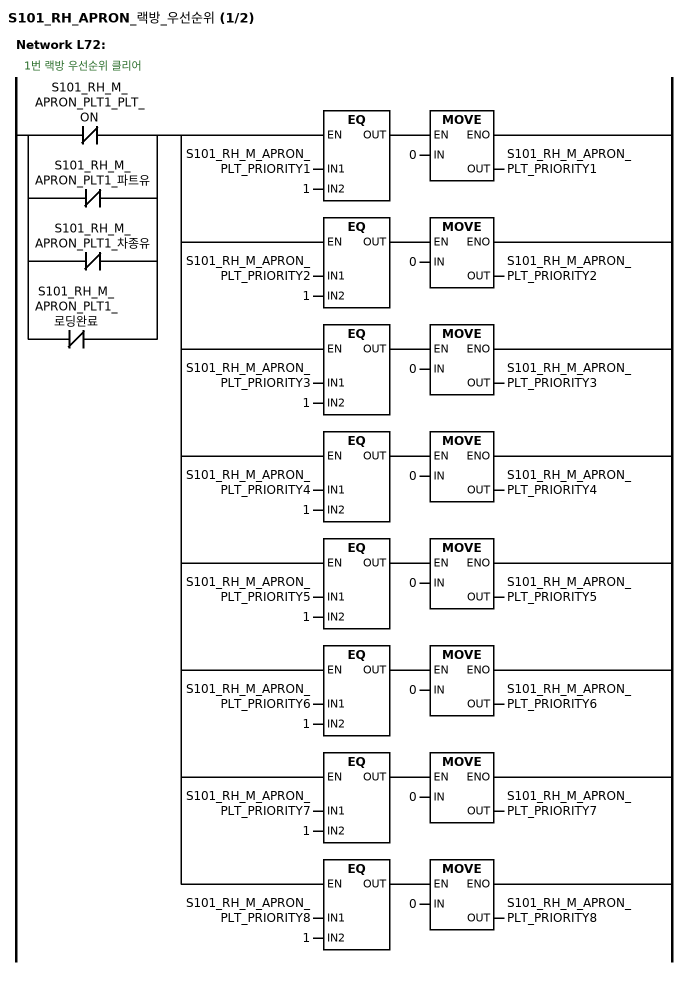
(* 1번 랙방 우선순위 클리어 *)
(* Rung L72 *)
_p1 := NOT S101_RH_M_APRON_PLT1_PLT_ON OR NOT S101_RH_M_APRON_PLT1_파트유 OR NOT S101_RH_M_APRON_PLT1_차종유 OR NOT S101_RH_M_APRON_PLT1_로딩완료;
IF _p1 THEN _t2 := S101_RH_M_APRON_PLT_PRIORITY1 = 1; END_IF;
IF _t2 THEN S101_RH_M_APRON_PLT_PRIORITY1 := 0; END_IF;
IF _p1 THEN _t3 := S101_RH_M_APRON_PLT_PRIORITY2 = 1; END_IF;
IF _t3 THEN S101_RH_M_APRON_PLT_PRIORITY2 := 0; END_IF;
IF _p1 THEN _t4 := S101_RH_M_APRON_PLT_PRIORITY3 = 1; END_IF;
IF _t4 THEN S101_RH_M_APRON_PLT_PRIORITY3 := 0; END_IF;
IF _p1 THEN _t5 := S101_RH_M_APRON_PLT_PRIORITY4 = 1; END_IF;
IF _t5 THEN S101_RH_M_APRON_PLT_PRIORITY4 := 0; END_IF;
IF _p1 THEN _t6 := S101_RH_M_APRON_PLT_PRIORITY5 = 1; END_IF;
IF _t6 THEN S101_RH_M_APRON_PLT_PRIORITY5 := 0; END_IF;
IF _p1 THEN _t7 := S101_RH_M_APRON_PLT_PRIORITY6 = 1; END_IF;
IF _t7 THEN S101_RH_M_APRON_PLT_PRIORITY6 := 0; END_IF;
IF _p1 THEN _t8 := S101_RH_M_APRON_PLT_PRIORITY7 = 1; END_IF;
IF _t8 THEN S101_RH_M_APRON_PLT_PRIORITY7 := 0; END_IF;
IF _p1 THEN _t9 := S101_RH_M_APRON_PLT_PRIORITY8 = 1; END_IF;
IF _t9 THEN S101_RH_M_APRON_PLT_PRIORITY8 := 0; END_IF;

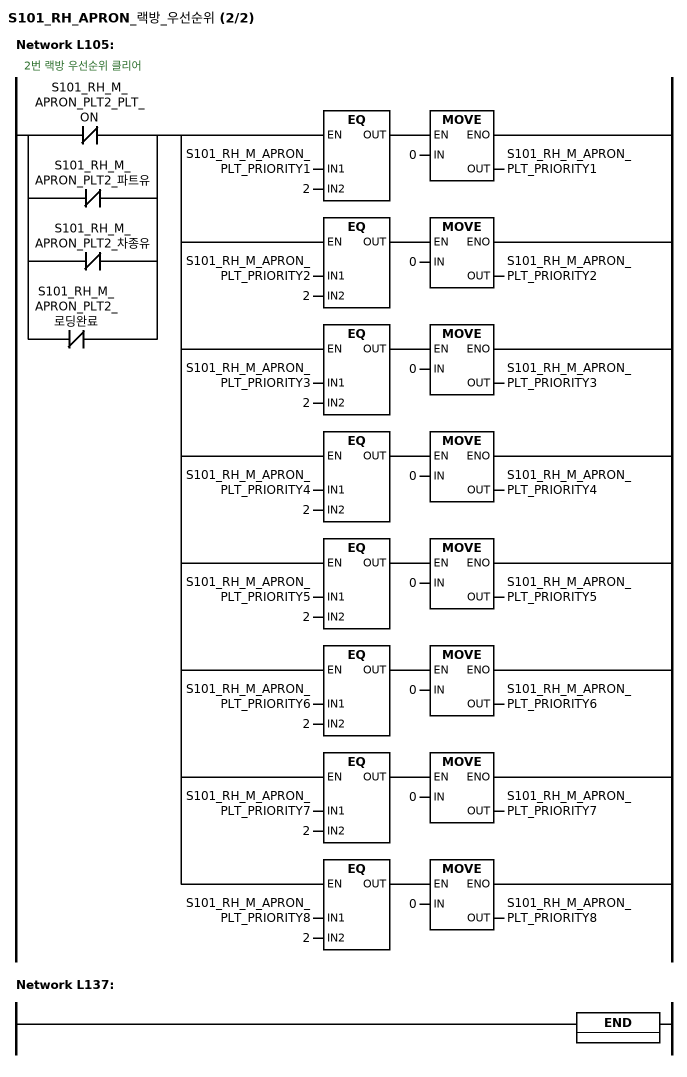
(* 2번 랙방 우선순위 클리어 *)
(* Rung L105 *)
_p10 := NOT S101_RH_M_APRON_PLT2_PLT_ON OR NOT S101_RH_M_APRON_PLT2_파트유 OR NOT S101_RH_M_APRON_PLT2_차종유 OR NOT S101_RH_M_APRON_PLT2_로딩완료;
IF _p10 THEN _t11 := S101_RH_M_APRON_PLT_PRIORITY1 = 2; END_IF;
IF _t11 THEN S101_RH_M_APRON_PLT_PRIORITY1 := 0; END_IF;
IF _p10 THEN _t12 := S101_RH_M_APRON_PLT_PRIORITY2 = 2; END_IF;
IF _t12 THEN S101_RH_M_APRON_PLT_PRIORITY2 := 0; END_IF;
IF _p10 THEN _t13 := S101_RH_M_APRON_PLT_PRIORITY3 = 2; END_IF;
IF _t13 THEN S101_RH_M_APRON_PLT_PRIORITY3 := 0; END_IF;
IF _p10 THEN _t14 := S101_RH_M_APRON_PLT_PRIORITY4 = 2; END_IF;
IF _t14 THEN S101_RH_M_APRON_PLT_PRIORITY4 := 0; END_IF;
IF _p10 THEN _t15 := S101_RH_M_APRON_PLT_PRIORITY5 = 2; END_IF;
IF _t15 THEN S101_RH_M_APRON_PLT_PRIORITY5 := 0; END_IF;
IF _p10 THEN _t16 := S101_RH_M_APRON_PLT_PRIORITY6 = 2; END_IF;
IF _t16 THEN S101_RH_M_APRON_PLT_PRIORITY6 := 0; END_IF;
IF _p10 THEN _t17 := S101_RH_M_APRON_PLT_PRIORITY7 = 2; END_IF;
IF _t17 THEN S101_RH_M_APRON_PLT_PRIORITY7 := 0; END_IF;
IF _p10 THEN _t18 := S101_RH_M_APRON_PLT_PRIORITY8 = 2; END_IF;
IF _t18 THEN S101_RH_M_APRON_PLT_PRIORITY8 := 0; END_IF;
(* Rung L137 *)
END();
END_PROGRAM

PROGRAM S101_로보트 (* task: 스캔 프로그램 *)
VAR_EXTERNAL
    AWAYS_OFF : BOOL; (* AT %MW3.0 *)
    AWAYS_ON : BOOL; (* AT %MW3.1 *)
    MCP_M_부저_정지 : BOOL; (* AT %MW350.5 *)
    MCP_M_비상정지 : BOOL; (* AT %MW350.7 *)
    MCP_PBL_운전준비_ON : BOOL; (* AT %MW87630.0 *) (* 입력 접점 00 *)
    R101_1_1_I_RB_INPUT : ARRAY[0..3] OF WORD; (* AT %MW84040 *)
    R101_1_1_M_I_RB_1차_작업완료 : BOOL; (* AT %MW20041.2 *)
    R101_1_1_M_I_RB_2차_작업완료 : BOOL; (* AT %MW20041.3 *)
    R101_1_1_M_I_RB_3차_작업완료 : BOOL; (* AT %MW20041.4 *)
    R101_1_1_M_I_RB_4차_작업완료 : BOOL; (* AT %MW20041.5 *)
    R101_1_1_M_I_RB_5차_작업완료 : BOOL; (* AT %MW20041.6 *)
    R101_1_1_M_I_RB_6차_작업완료 : BOOL; (* AT %MW20041.7 *)
    R101_1_1_M_I_RB_7차_작업완료 : BOOL; (* AT %MW20041.8 *)
    R101_1_1_M_I_RB_PAUSE_보조 : BOOL; (* AT %MW20040.5 *)
    R101_1_1_M_I_RB_PLC_RUN_CHK_이상 : BOOL; (* AT %MW20040.7 *)
    R101_1_1_M_I_RB_간섭무_1 : BOOL; (* AT %MW20042.0 *)
    R101_1_1_M_I_RB_간섭무_10 : BOOL; (* AT %MW20042.9 *)
    R101_1_1_M_I_RB_간섭무_11 : BOOL; (* AT %MW20042.10 *)
    R101_1_1_M_I_RB_간섭무_12 : BOOL; (* AT %MW20042.11 *)
    R101_1_1_M_I_RB_간섭무_2 : BOOL; (* AT %MW20042.1 *)
    R101_1_1_M_I_RB_간섭무_3 : BOOL; (* AT %MW20042.2 *)
    R101_1_1_M_I_RB_간섭무_4 : BOOL; (* AT %MW20042.3 *)
    R101_1_1_M_I_RB_간섭무_5 : BOOL; (* AT %MW20042.4 *)
    R101_1_1_M_I_RB_간섭무_6 : BOOL; (* AT %MW20042.5 *)
    R101_1_1_M_I_RB_간섭무_7 : BOOL; (* AT %MW20042.6 *)
    R101_1_1_M_I_RB_간섭무_8 : BOOL; (* AT %MW20042.7 *)
    R101_1_1_M_I_RB_간섭무_9 : BOOL; (* AT %MW20042.8 *)
    R101_1_1_M_I_RB_비상정지 : BOOL; (* AT %MW20040.4 *)
    R101_1_1_M_I_RB_운전준비 : BOOL; (* AT %MW20040.0 *)
    R101_1_1_M_I_RB_원위치 : BOOL; (* AT %MW20040.3 *)
    R101_1_1_M_I_RB_이상 : BOOL; (* AT %MW20040.2 *)
    R101_1_1_M_I_RB_자동 : BOOL; (* AT %MW20040.1 *)
    R101_1_1_M_I_RB_최종작업완료 : BOOL; (* AT %MW20041.0 *)
    R101_1_1_M_I_RB_프로그램_이상 : BOOL; (* AT %MW20040.6 *)
    R101_1_1_M_O_RB_1_CYCLE_SET : BOOL; (* AT %MW21040.3 *)
    R101_1_1_M_O_RB_1차_작업완료_리셋 : BOOL; (* AT %MW21042.0 *)
    R101_1_1_M_O_RB_2차_작업완료_리셋 : BOOL; (* AT %MW21042.1 *)
    R101_1_1_M_O_RB_2차_진입OK : BOOL; (* AT %MW21041.8 *)
    R101_1_1_M_O_RB_3차_작업완료_리셋 : BOOL; (* AT %MW21042.2 *)
    R101_1_1_M_O_RB_3차_진입OK : BOOL; (* AT %MW21041.9 *)
    R101_1_1_M_O_RB_4차_작업완료_리셋 : BOOL; (* AT %MW21042.3 *)
    R101_1_1_M_O_RB_4차_진입OK : BOOL; (* AT %MW21041.10 *)
    R101_1_1_M_O_RB_5차_작업완료_리셋 : BOOL; (* AT %MW21042.4 *)
    R101_1_1_M_O_RB_5차_진입OK : BOOL; (* AT %MW21041.11 *)
    R101_1_1_M_O_RB_6차_작업완료_리셋 : BOOL; (* AT %MW21042.5 *)
    R101_1_1_M_O_RB_6차_진입OK : BOOL; (* AT %MW21041.12 *)
    R101_1_1_M_O_RB_7차_작업완료_리셋 : BOOL; (* AT %MW21042.6 *)
    R101_1_1_M_O_RB_7차_진입OK : BOOL; (* AT %MW21041.13 *)
    R101_1_1_M_O_RB_ATD_OK : BOOL; (* AT %MW21040.6 *)
    R101_1_1_M_O_RB_PLT_10_진입OK : BOOL; (* AT %MW21043.10 *)
    R101_1_1_M_O_RB_PLT_11_진입OK : BOOL; (* AT %MW21043.11 *)
    R101_1_1_M_O_RB_PLT_12_진입OK : BOOL; (* AT %MW21043.12 *)
    R101_1_1_M_O_RB_PLT_1_진입OK : BOOL; (* AT %MW21043.1 *)
    R101_1_1_M_O_RB_PLT_2_진입OK : BOOL; (* AT %MW21043.2 *)
    R101_1_1_M_O_RB_PLT_3_진입OK : BOOL; (* AT %MW21043.3 *)
    R101_1_1_M_O_RB_PLT_4_진입OK : BOOL; (* AT %MW21043.4 *)
    R101_1_1_M_O_RB_PLT_5_진입OK : BOOL; (* AT %MW21043.5 *)
    R101_1_1_M_O_RB_PLT_6_진입OK : BOOL; (* AT %MW21043.6 *)
    R101_1_1_M_O_RB_PLT_7_진입OK : BOOL; (* AT %MW21043.7 *)
    R101_1_1_M_O_RB_PLT_8_진입OK : BOOL; (* AT %MW21043.8 *)
    R101_1_1_M_O_RB_PLT_9_진입OK : BOOL; (* AT %MW21043.9 *)
    R101_1_1_M_O_RB_PLT_카운터리셋_보조 : BOOL; (* AT %MW21040.10 *)
    R101_1_1_M_O_RB_RESTART_OK : BOOL; (* AT %MW21040.2 *)
    R101_1_1_M_O_RB_START_OK : BOOL; (* AT %MW21040.0 *)
    R101_1_1_M_O_RB_TEST_MODE_5000회 : BOOL; (* AT %MW21040.12 *)
    R101_1_1_M_O_RB_TIP_교체_시작 : BOOL; (* AT %MW21040.7 *)
    R101_1_1_M_O_RB_TIP_교체_완료 : BOOL; (* AT %MW21040.8 *)
    R101_1_1_M_O_RB_VIP_MODE : BOOL; (* AT %MW21040.11 *)
    R101_1_1_M_O_RB_냉각수_차단_요청 : BOOL; (* AT %MW21040.9 *)
    R101_1_1_M_O_RB_진입OK_AX차종 : BOOL; (* AT %MW21041.0 *)
    R101_1_1_M_O_RB_진입OK_B차종 : BOOL; (* AT %MW21041.1 *)
    R101_1_1_M_O_RB_진입OK_C차종 : BOOL; (* AT %MW21041.2 *)
    R101_1_1_M_O_RB_진입OK_D차종 : BOOL; (* AT %MW21041.3 *)
    R101_1_1_M_O_RB_진입OK_E차종 : BOOL; (* AT %MW21041.4 *)
    R101_1_1_M_O_RB_진입OK_F차종 : BOOL; (* AT %MW21041.5 *)
    R101_1_1_M_O_RB_진입OK_G차종 : BOOL; (* AT %MW21041.6 *)
    R101_1_1_M_O_RB_진입OK_H차종 : BOOL; (* AT %MW21041.7 *)
    R101_1_1_M_O_RB_최종_작업완료_리셋 : BOOL; (* AT %MW21040.5 *)
    R101_1_1_M_O_RB_프로그램_OK : BOOL; (* AT %MW21040.1 *)
    R101_1_1_M_RB_PROG_NO : WORD; (* AT %MW20044 *)
    R101_1_1_M_STN_차종_ON : BOOL; (* AT %MW1002.2 *)
    R101_1_1_M_차종1_AX : BOOL; (* AT %MW10001.0 *) (* R101_1_1_M_차종1_AX *)
    R101_1_1_O_RB_OUTPUT : ARRAY[0..3] OF WORD; (* AT %MW94040 *)
    R101_1_I_RB_INPUT : ARRAY[0..3] OF WORD; (* AT %MW84070 *)
    R101_1_M_I_RB_1차_작업완료 : BOOL; (* AT %MW20071.2 *)
    R101_1_M_I_RB_2차_작업완료 : BOOL; (* AT %MW20071.3 *)
    R101_1_M_I_RB_3차_작업완료 : BOOL; (* AT %MW20071.4 *)
    R101_1_M_I_RB_4차_작업완료 : BOOL; (* AT %MW20071.5 *)
    R101_1_M_I_RB_5차_작업완료 : BOOL; (* AT %MW20071.6 *)
    R101_1_M_I_RB_6차_작업완료 : BOOL; (* AT %MW20071.7 *)
    R101_1_M_I_RB_7차_작업완료 : BOOL; (* AT %MW20071.8 *)
    R101_1_M_I_RB_PAUSE_보조 : BOOL; (* AT %MW20070.5 *)
    R101_1_M_I_RB_PLC_RUN_CHK_이상 : BOOL; (* AT %MW20070.7 *)
    R101_1_M_I_RB_간섭무_1 : BOOL; (* AT %MW20072.0 *)
    R101_1_M_I_RB_간섭무_10 : BOOL; (* AT %MW20072.9 *)
    R101_1_M_I_RB_간섭무_11 : BOOL; (* AT %MW20072.10 *)
    R101_1_M_I_RB_간섭무_12 : BOOL; (* AT %MW20072.11 *)
    R101_1_M_I_RB_간섭무_2 : BOOL; (* AT %MW20072.1 *)
    R101_1_M_I_RB_간섭무_3 : BOOL; (* AT %MW20072.2 *)
    R101_1_M_I_RB_간섭무_4 : BOOL; (* AT %MW20072.3 *)
    R101_1_M_I_RB_간섭무_5 : BOOL; (* AT %MW20072.4 *)
    R101_1_M_I_RB_간섭무_6 : BOOL; (* AT %MW20072.5 *)
    R101_1_M_I_RB_간섭무_7 : BOOL; (* AT %MW20072.6 *)
    R101_1_M_I_RB_간섭무_8 : BOOL; (* AT %MW20072.7 *)
    R101_1_M_I_RB_간섭무_9 : BOOL; (* AT %MW20072.8 *)
    R101_1_M_I_RB_비상정지 : BOOL; (* AT %MW20070.4 *)
    R101_1_M_I_RB_운전준비 : BOOL; (* AT %MW20070.0 *)
    R101_1_M_I_RB_원위치 : BOOL; (* AT %MW20070.3 *)
    R101_1_M_I_RB_이상 : BOOL; (* AT %MW20070.2 *)
    R101_1_M_I_RB_자동 : BOOL; (* AT %MW20070.1 *)
    R101_1_M_I_RB_최종작업완료 : BOOL; (* AT %MW20071.0 *)
    R101_1_M_I_RB_프로그램_이상 : BOOL; (* AT %MW20070.6 *)
    R101_1_M_O_RB_1_CYCLE_SET : BOOL; (* AT %MW21070.3 *)
    R101_1_M_O_RB_1차_작업완료_리셋 : BOOL; (* AT %MW21072.0 *)
    R101_1_M_O_RB_2차_작업완료_리셋 : BOOL; (* AT %MW21072.1 *)
    R101_1_M_O_RB_2차_진입OK : BOOL; (* AT %MW21071.8 *)
    R101_1_M_O_RB_3차_작업완료_리셋 : BOOL; (* AT %MW21072.2 *)
    R101_1_M_O_RB_3차_진입OK : BOOL; (* AT %MW21071.9 *)
    R101_1_M_O_RB_4차_작업완료_리셋 : BOOL; (* AT %MW21072.3 *)
    R101_1_M_O_RB_4차_진입OK : BOOL; (* AT %MW21071.10 *)
    R101_1_M_O_RB_5차_작업완료_리셋 : BOOL; (* AT %MW21072.4 *)
    R101_1_M_O_RB_5차_진입OK : BOOL; (* AT %MW21071.11 *)
    R101_1_M_O_RB_6차_작업완료_리셋 : BOOL; (* AT %MW21072.5 *)
    R101_1_M_O_RB_6차_진입OK : BOOL; (* AT %MW21071.12 *)
    R101_1_M_O_RB_7차_작업완료_리셋 : BOOL; (* AT %MW21072.6 *)
    R101_1_M_O_RB_7차_진입OK : BOOL; (* AT %MW21071.13 *)
    R101_1_M_O_RB_ATD_OK : BOOL; (* AT %MW21070.6 *)
    R101_1_M_O_RB_PLT_10_진입OK : BOOL; (* AT %MW21073.10 *)
    R101_1_M_O_RB_PLT_11_진입OK : BOOL; (* AT %MW21073.11 *)
    R101_1_M_O_RB_PLT_12_진입OK : BOOL; (* AT %MW21073.12 *)
    R101_1_M_O_RB_PLT_1_진입OK : BOOL; (* AT %MW21073.1 *)
    R101_1_M_O_RB_PLT_2_진입OK : BOOL; (* AT %MW21073.2 *)
    R101_1_M_O_RB_PLT_3_진입OK : BOOL; (* AT %MW21073.3 *)
    R101_1_M_O_RB_PLT_4_진입OK : BOOL; (* AT %MW21073.4 *)
    R101_1_M_O_RB_PLT_5_진입OK : BOOL; (* AT %MW21073.5 *)
    R101_1_M_O_RB_PLT_6_진입OK : BOOL; (* AT %MW21073.6 *)
    R101_1_M_O_RB_PLT_7_진입OK : BOOL; (* AT %MW21073.7 *)
    R101_1_M_O_RB_PLT_8_진입OK : BOOL; (* AT %MW21073.8 *)
    R101_1_M_O_RB_PLT_9_진입OK : BOOL; (* AT %MW21073.9 *)
    R101_1_M_O_RB_PLT_카운터리셋_보조 : BOOL; (* AT %MW21070.10 *)
    R101_1_M_O_RB_RESTART_OK : BOOL; (* AT %MW21070.2 *)
    R101_1_M_O_RB_START_OK : BOOL; (* AT %MW21070.0 *)
    R101_1_M_O_RB_TEST_MODE_5000회 : BOOL; (* AT %MW21070.12 *)
    R101_1_M_O_RB_TIP_교체_시작 : BOOL; (* AT %MW21070.7 *)
    R101_1_M_O_RB_TIP_교체_완료 : BOOL; (* AT %MW21070.8 *)
    R101_1_M_O_RB_VIP_MODE : BOOL; (* AT %MW21070.11 *)
    R101_1_M_O_RB_냉각수_차단_요청 : BOOL; (* AT %MW21070.9 *)
    R101_1_M_O_RB_진입OK_AX차종 : BOOL; (* AT %MW21071.0 *)
    R101_1_M_O_RB_진입OK_B차종 : BOOL; (* AT %MW21071.1 *)
    R101_1_M_O_RB_진입OK_C차종 : BOOL; (* AT %MW21071.2 *)
    R101_1_M_O_RB_진입OK_D차종 : BOOL; (* AT %MW21071.3 *)
    R101_1_M_O_RB_진입OK_E차종 : BOOL; (* AT %MW21071.4 *)
    R101_1_M_O_RB_진입OK_F차종 : BOOL; (* AT %MW21071.5 *)
    R101_1_M_O_RB_진입OK_G차종 : BOOL; (* AT %MW21071.6 *)
    R101_1_M_O_RB_진입OK_H차종 : BOOL; (* AT %MW21071.7 *)
    R101_1_M_O_RB_최종_작업완료_리셋 : BOOL; (* AT %MW21070.5 *)
    R101_1_M_O_RB_프로그램_OK : BOOL; (* AT %MW21070.1 *)
    R101_1_M_RB_PROG_NO : WORD; (* AT %MW20074 *)
    R101_1_O_RB_MUTUAL_INT1 : BOOL; (* AT %MW94073.0 *)
    R101_1_O_RB_OUTPUT : ARRAY[0..3] OF WORD; (* AT %MW94070 *)
    R101_2_I_RB_INPUT : ARRAY[0..3] OF WORD; (* AT %MW84060 *)
    R101_2_M_I_RB_1차_작업완료 : BOOL; (* AT %MW20061.2 *)
    R101_2_M_I_RB_2차_작업완료 : BOOL; (* AT %MW20061.3 *)
    R101_2_M_I_RB_3차_작업완료 : BOOL; (* AT %MW20061.4 *)
    R101_2_M_I_RB_4차_작업완료 : BOOL; (* AT %MW20061.5 *)
    R101_2_M_I_RB_5차_작업완료 : BOOL; (* AT %MW20061.6 *)
    R101_2_M_I_RB_6차_작업완료 : BOOL; (* AT %MW20061.7 *)
    R101_2_M_I_RB_7차_작업완료 : BOOL; (* AT %MW20061.8 *)
    R101_2_M_I_RB_PAUSE_보조 : BOOL; (* AT %MW20060.5 *)
    R101_2_M_I_RB_PLC_RUN_CHK_이상 : BOOL; (* AT %MW20060.7 *)
    R101_2_M_I_RB_간섭무_1 : BOOL; (* AT %MW20062.0 *)
    R101_2_M_I_RB_간섭무_10 : BOOL; (* AT %MW20062.9 *)
    R101_2_M_I_RB_간섭무_11 : BOOL; (* AT %MW20062.10 *)
    R101_2_M_I_RB_간섭무_12 : BOOL; (* AT %MW20062.11 *)
    R101_2_M_I_RB_간섭무_2 : BOOL; (* AT %MW20062.1 *)
    R101_2_M_I_RB_간섭무_3 : BOOL; (* AT %MW20062.2 *)
    R101_2_M_I_RB_간섭무_4 : BOOL; (* AT %MW20062.3 *)
    R101_2_M_I_RB_간섭무_5 : BOOL; (* AT %MW20062.4 *)
    R101_2_M_I_RB_간섭무_6 : BOOL; (* AT %MW20062.5 *)
    R101_2_M_I_RB_간섭무_7 : BOOL; (* AT %MW20062.6 *)
    R101_2_M_I_RB_간섭무_8 : BOOL; (* AT %MW20062.7 *)
    R101_2_M_I_RB_간섭무_9 : BOOL; (* AT %MW20062.8 *)
    R101_2_M_I_RB_비상정지 : BOOL; (* AT %MW20060.4 *)
    R101_2_M_I_RB_운전준비 : BOOL; (* AT %MW20060.0 *)
    R101_2_M_I_RB_원위치 : BOOL; (* AT %MW20060.3 *)
    R101_2_M_I_RB_이상 : BOOL; (* AT %MW20060.2 *)
    R101_2_M_I_RB_자동 : BOOL; (* AT %MW20060.1 *)
    R101_2_M_I_RB_최종작업완료 : BOOL; (* AT %MW20061.0 *)
    R101_2_M_I_RB_프로그램_이상 : BOOL; (* AT %MW20060.6 *)
    R101_2_M_O_RB_1_CYCLE_SET : BOOL; (* AT %MW21060.3 *)
    R101_2_M_O_RB_1차_작업완료_리셋 : BOOL; (* AT %MW21062.0 *)
    R101_2_M_O_RB_2차_작업완료_리셋 : BOOL; (* AT %MW21062.1 *)
    R101_2_M_O_RB_2차_진입OK : BOOL; (* AT %MW21061.8 *)
    R101_2_M_O_RB_3차_작업완료_리셋 : BOOL; (* AT %MW21062.2 *)
    R101_2_M_O_RB_3차_진입OK : BOOL; (* AT %MW21061.9 *)
    R101_2_M_O_RB_4차_작업완료_리셋 : BOOL; (* AT %MW21062.3 *)
    R101_2_M_O_RB_4차_진입OK : BOOL; (* AT %MW21061.10 *)
    R101_2_M_O_RB_5차_작업완료_리셋 : BOOL; (* AT %MW21062.4 *)
    R101_2_M_O_RB_5차_진입OK : BOOL; (* AT %MW21061.11 *)
    R101_2_M_O_RB_6차_작업완료_리셋 : BOOL; (* AT %MW21062.5 *)
    R101_2_M_O_RB_6차_진입OK : BOOL; (* AT %MW21061.12 *)
    R101_2_M_O_RB_7차_작업완료_리셋 : BOOL; (* AT %MW21062.6 *)
    R101_2_M_O_RB_7차_진입OK : BOOL; (* AT %MW21061.13 *)
    R101_2_M_O_RB_ATD_OK : BOOL; (* AT %MW21060.6 *)
    R101_2_M_O_RB_PLT_10_진입OK : BOOL; (* AT %MW21063.10 *)
    R101_2_M_O_RB_PLT_11_진입OK : BOOL; (* AT %MW21063.11 *)
    R101_2_M_O_RB_PLT_12_진입OK : BOOL; (* AT %MW21063.12 *)
    R101_2_M_O_RB_PLT_1_진입OK : BOOL; (* AT %MW21063.1 *)
    R101_2_M_O_RB_PLT_2_진입OK : BOOL; (* AT %MW21063.2 *)
    R101_2_M_O_RB_PLT_3_진입OK : BOOL; (* AT %MW21063.3 *)
    R101_2_M_O_RB_PLT_4_진입OK : BOOL; (* AT %MW21063.4 *)
    R101_2_M_O_RB_PLT_5_진입OK : BOOL; (* AT %MW21063.5 *)
    R101_2_M_O_RB_PLT_6_진입OK : BOOL; (* AT %MW21063.6 *)
    R101_2_M_O_RB_PLT_7_진입OK : BOOL; (* AT %MW21063.7 *)
    R101_2_M_O_RB_PLT_8_진입OK : BOOL; (* AT %MW21063.8 *)
    R101_2_M_O_RB_PLT_9_진입OK : BOOL; (* AT %MW21063.9 *)
    R101_2_M_O_RB_PLT_카운터리셋_보조 : BOOL; (* AT %MW21060.10 *)
    R101_2_M_O_RB_RESTART_OK : BOOL; (* AT %MW21060.2 *)
    R101_2_M_O_RB_START_OK : BOOL; (* AT %MW21060.0 *)
    R101_2_M_O_RB_TEST_MODE_5000회 : BOOL; (* AT %MW21060.12 *)
    R101_2_M_O_RB_TIP_교체_시작 : BOOL; (* AT %MW21060.7 *)
    R101_2_M_O_RB_TIP_교체_완료 : BOOL; (* AT %MW21060.8 *)
    R101_2_M_O_RB_VIP_MODE : BOOL; (* AT %MW21060.11 *)
    R101_2_M_O_RB_냉각수_차단_요청 : BOOL; (* AT %MW21060.9 *)
    R101_2_M_O_RB_진입OK_AX차종 : BOOL; (* AT %MW21061.0 *)
    R101_2_M_O_RB_진입OK_B차종 : BOOL; (* AT %MW21061.1 *)
    R101_2_M_O_RB_진입OK_C차종 : BOOL; (* AT %MW21061.2 *)
    R101_2_M_O_RB_진입OK_D차종 : BOOL; (* AT %MW21061.3 *)
    R101_2_M_O_RB_진입OK_E차종 : BOOL; (* AT %MW21061.4 *)
    R101_2_M_O_RB_진입OK_F차종 : BOOL; (* AT %MW21061.5 *)
    R101_2_M_O_RB_진입OK_G차종 : BOOL; (* AT %MW21061.6 *)
    R101_2_M_O_RB_진입OK_H차종 : BOOL; (* AT %MW21061.7 *)
    R101_2_M_O_RB_최종_작업완료_리셋 : BOOL; (* AT %MW21060.5 *)
    R101_2_M_O_RB_프로그램_OK : BOOL; (* AT %MW21060.1 *)
    R101_2_M_RB_PROG_NO : WORD; (* AT %MW20064 *)
    R101_2_O_RB_MUTUAL_INT1 : BOOL; (* AT %MW94063.0 *)
    R101_2_O_RB_OUTPUT : ARRAY[0..3] OF WORD; (* AT %MW94060 *)
    R101_3_I_RB_INPUT : ARRAY[0..3] OF WORD; (* AT %MW84050 *)
    R101_3_M_I_RB_1차_작업완료 : BOOL; (* AT %MW20051.2 *)
    R101_3_M_I_RB_2차_작업완료 : BOOL; (* AT %MW20051.3 *)
    R101_3_M_I_RB_3차_작업완료 : BOOL; (* AT %MW20051.4 *)
    R101_3_M_I_RB_4차_작업완료 : BOOL; (* AT %MW20051.5 *)
    R101_3_M_I_RB_5차_작업완료 : BOOL; (* AT %MW20051.6 *)
    R101_3_M_I_RB_6차_작업완료 : BOOL; (* AT %MW20051.7 *)
    R101_3_M_I_RB_7차_작업완료 : BOOL; (* AT %MW20051.8 *)
    R101_3_M_I_RB_PAUSE_보조 : BOOL; (* AT %MW20050.5 *)
    R101_3_M_I_RB_PLC_RUN_CHK_이상 : BOOL; (* AT %MW20050.7 *)
    R101_3_M_I_RB_간섭무_1 : BOOL; (* AT %MW20052.0 *)
    R101_3_M_I_RB_간섭무_10 : BOOL; (* AT %MW20052.9 *)
    R101_3_M_I_RB_간섭무_11 : BOOL; (* AT %MW20052.10 *)
    R101_3_M_I_RB_간섭무_12 : BOOL; (* AT %MW20052.11 *)
    R101_3_M_I_RB_간섭무_2 : BOOL; (* AT %MW20052.1 *)
    R101_3_M_I_RB_간섭무_3 : BOOL; (* AT %MW20052.2 *)
    R101_3_M_I_RB_간섭무_4 : BOOL; (* AT %MW20052.3 *)
    R101_3_M_I_RB_간섭무_5 : BOOL; (* AT %MW20052.4 *)
    R101_3_M_I_RB_간섭무_6 : BOOL; (* AT %MW20052.5 *)
    R101_3_M_I_RB_간섭무_7 : BOOL; (* AT %MW20052.6 *)
    R101_3_M_I_RB_간섭무_8 : BOOL; (* AT %MW20052.7 *)
    R101_3_M_I_RB_간섭무_9 : BOOL; (* AT %MW20052.8 *)
    R101_3_M_I_RB_비상정지 : BOOL; (* AT %MW20050.4 *)
    R101_3_M_I_RB_운전준비 : BOOL; (* AT %MW20050.0 *)
    R101_3_M_I_RB_원위치 : BOOL; (* AT %MW20050.3 *)
    R101_3_M_I_RB_이상 : BOOL; (* AT %MW20050.2 *)
    R101_3_M_I_RB_자동 : BOOL; (* AT %MW20050.1 *)
    R101_3_M_I_RB_최종작업완료 : BOOL; (* AT %MW20051.0 *)
    R101_3_M_I_RB_프로그램_이상 : BOOL; (* AT %MW20050.6 *)
    R101_3_M_O_RB_1_CYCLE_SET : BOOL; (* AT %MW21050.3 *)
    R101_3_M_O_RB_1차_작업완료_리셋 : BOOL; (* AT %MW21052.0 *)
    R101_3_M_O_RB_2차_작업완료_리셋 : BOOL; (* AT %MW21052.1 *)
    R101_3_M_O_RB_2차_진입OK : BOOL; (* AT %MW21051.8 *)
    R101_3_M_O_RB_3차_작업완료_리셋 : BOOL; (* AT %MW21052.2 *)
    R101_3_M_O_RB_3차_진입OK : BOOL; (* AT %MW21051.9 *)
    R101_3_M_O_RB_4차_작업완료_리셋 : BOOL; (* AT %MW21052.3 *)
    R101_3_M_O_RB_4차_진입OK : BOOL; (* AT %MW21051.10 *)
    R101_3_M_O_RB_5차_작업완료_리셋 : BOOL; (* AT %MW21052.4 *)
    R101_3_M_O_RB_5차_진입OK : BOOL; (* AT %MW21051.11 *)
    R101_3_M_O_RB_6차_작업완료_리셋 : BOOL; (* AT %MW21052.5 *)
    R101_3_M_O_RB_6차_진입OK : BOOL; (* AT %MW21051.12 *)
    R101_3_M_O_RB_7차_작업완료_리셋 : BOOL; (* AT %MW21052.6 *)
    R101_3_M_O_RB_7차_진입OK : BOOL; (* AT %MW21051.13 *)
    R101_3_M_O_RB_ATD_OK : BOOL; (* AT %MW21050.6 *)
    R101_3_M_O_RB_PLT_10_진입OK : BOOL; (* AT %MW21053.10 *)
    R101_3_M_O_RB_PLT_11_진입OK : BOOL; (* AT %MW21053.11 *)
    R101_3_M_O_RB_PLT_12_진입OK : BOOL; (* AT %MW21053.12 *)
    R101_3_M_O_RB_PLT_1_진입OK : BOOL; (* AT %MW21053.1 *)
    R101_3_M_O_RB_PLT_2_진입OK : BOOL; (* AT %MW21053.2 *)
    R101_3_M_O_RB_PLT_3_진입OK : BOOL; (* AT %MW21053.3 *)
    R101_3_M_O_RB_PLT_4_진입OK : BOOL; (* AT %MW21053.4 *)
    R101_3_M_O_RB_PLT_5_진입OK : BOOL; (* AT %MW21053.5 *)
    R101_3_M_O_RB_PLT_6_진입OK : BOOL; (* AT %MW21053.6 *)
    R101_3_M_O_RB_PLT_7_진입OK : BOOL; (* AT %MW21053.7 *)
    R101_3_M_O_RB_PLT_8_진입OK : BOOL; (* AT %MW21053.8 *)
    R101_3_M_O_RB_PLT_9_진입OK : BOOL; (* AT %MW21053.9 *)
    R101_3_M_O_RB_PLT_카운터리셋_보조 : BOOL; (* AT %MW21050.10 *)
    R101_3_M_O_RB_RESTART_OK : BOOL; (* AT %MW21050.2 *)
    R101_3_M_O_RB_START_OK : BOOL; (* AT %MW21050.0 *)
    R101_3_M_O_RB_TEST_MODE_5000회 : BOOL; (* AT %MW21050.12 *)
    R101_3_M_O_RB_TIP_교체_시작 : BOOL; (* AT %MW21050.7 *)
    R101_3_M_O_RB_TIP_교체_완료 : BOOL; (* AT %MW21050.8 *)
    R101_3_M_O_RB_VIP_MODE : BOOL; (* AT %MW21050.11 *)
    R101_3_M_O_RB_냉각수_차단_요청 : BOOL; (* AT %MW21050.9 *)
    R101_3_M_O_RB_진입OK_AX차종 : BOOL; (* AT %MW21051.0 *)
    R101_3_M_O_RB_진입OK_B차종 : BOOL; (* AT %MW21051.1 *)
    R101_3_M_O_RB_진입OK_C차종 : BOOL; (* AT %MW21051.2 *)
    R101_3_M_O_RB_진입OK_D차종 : BOOL; (* AT %MW21051.3 *)
    R101_3_M_O_RB_진입OK_E차종 : BOOL; (* AT %MW21051.4 *)
    R101_3_M_O_RB_진입OK_F차종 : BOOL; (* AT %MW21051.5 *)
    R101_3_M_O_RB_진입OK_G차종 : BOOL; (* AT %MW21051.6 *)
    R101_3_M_O_RB_진입OK_H차종 : BOOL; (* AT %MW21051.7 *)
    R101_3_M_O_RB_최종_작업완료_리셋 : BOOL; (* AT %MW21050.5 *)
    R101_3_M_O_RB_프로그램_OK : BOOL; (* AT %MW21050.1 *)
    R101_3_M_RB_PROG_NO : WORD; (* AT %MW20054 *)
    R101_3_O_RB_OUTPUT : ARRAY[0..3] OF WORD; (* AT %MW94050 *)
    R101_3축_리어_I_RB_INPUT : ARRAY[0..3] OF WORD; (* AT %MW84030 *)
    R101_3축_리어_M_I_RB_1차_작업완료 : BOOL; (* AT %MW20031.2 *)
    R101_3축_리어_M_I_RB_2차_작업완료 : BOOL; (* AT %MW20031.3 *)
    R101_3축_리어_M_I_RB_3차_작업완료 : BOOL; (* AT %MW20031.4 *)
    R101_3축_리어_M_I_RB_4차_작업완료 : BOOL; (* AT %MW20031.5 *)
    R101_3축_리어_M_I_RB_5차_작업완료 : BOOL; (* AT %MW20031.6 *)
    R101_3축_리어_M_I_RB_6차_작업완료 : BOOL; (* AT %MW20031.7 *)
    R101_3축_리어_M_I_RB_7차_작업완료 : BOOL; (* AT %MW20031.8 *)
    R101_3축_리어_M_I_RB_PAUSE_보조 : BOOL; (* AT %MW20030.5 *)
    R101_3축_리어_M_I_RB_PLC_RUN_CHK_이상 : BOOL; (* AT %MW20030.7 *)
    R101_3축_리어_M_I_RB_간섭무_1 : BOOL; (* AT %MW20032.0 *)
    R101_3축_리어_M_I_RB_간섭무_10 : BOOL; (* AT %MW20032.9 *)
    R101_3축_리어_M_I_RB_간섭무_11 : BOOL; (* AT %MW20032.10 *)
    R101_3축_리어_M_I_RB_간섭무_12 : BOOL; (* AT %MW20032.11 *)
    R101_3축_리어_M_I_RB_간섭무_2 : BOOL; (* AT %MW20032.1 *)
    R101_3축_리어_M_I_RB_간섭무_3 : BOOL; (* AT %MW20032.2 *)
    R101_3축_리어_M_I_RB_간섭무_4 : BOOL; (* AT %MW20032.3 *)
    R101_3축_리어_M_I_RB_간섭무_5 : BOOL; (* AT %MW20032.4 *)
    R101_3축_리어_M_I_RB_간섭무_6 : BOOL; (* AT %MW20032.5 *)
    R101_3축_리어_M_I_RB_간섭무_7 : BOOL; (* AT %MW20032.6 *)
    R101_3축_리어_M_I_RB_간섭무_8 : BOOL; (* AT %MW20032.7 *)
    R101_3축_리어_M_I_RB_간섭무_9 : BOOL; (* AT %MW20032.8 *)
    R101_3축_리어_M_I_RB_비상정지 : BOOL; (* AT %MW20030.4 *)
    R101_3축_리어_M_I_RB_운전준비 : BOOL; (* AT %MW20030.0 *)
    R101_3축_리어_M_I_RB_원위치 : BOOL; (* AT %MW20030.3 *)
    R101_3축_리어_M_I_RB_이상 : BOOL; (* AT %MW20030.2 *)
    R101_3축_리어_M_I_RB_자동 : BOOL; (* AT %MW20030.1 *)
    R101_3축_리어_M_I_RB_최종작업완료 : BOOL; (* AT %MW20031.0 *)
    R101_3축_리어_M_I_RB_프로그램_이상 : BOOL; (* AT %MW20030.6 *)
    R101_3축_리어_M_O_RB_1_CYCLE_SET : BOOL; (* AT %MW21030.3 *)
    R101_3축_리어_M_O_RB_1차_작업완료_리셋 : BOOL; (* AT %MW21032.0 *)
    R101_3축_리어_M_O_RB_2차_작업완료_리셋 : BOOL; (* AT %MW21032.1 *)
    R101_3축_리어_M_O_RB_2차_진입OK : BOOL; (* AT %MW21031.8 *)
    R101_3축_리어_M_O_RB_3차_작업완료_리셋 : BOOL; (* AT %MW21032.2 *)
    R101_3축_리어_M_O_RB_3차_진입OK : BOOL; (* AT %MW21031.9 *)
    R101_3축_리어_M_O_RB_4차_작업완료_리셋 : BOOL; (* AT %MW21032.3 *)
    R101_3축_리어_M_O_RB_4차_진입OK : BOOL; (* AT %MW21031.10 *)
    R101_3축_리어_M_O_RB_5차_작업완료_리셋 : BOOL; (* AT %MW21032.4 *)
    R101_3축_리어_M_O_RB_5차_진입OK : BOOL; (* AT %MW21031.11 *)
    R101_3축_리어_M_O_RB_6차_작업완료_리셋 : BOOL; (* AT %MW21032.5 *)
    R101_3축_리어_M_O_RB_6차_진입OK : BOOL; (* AT %MW21031.12 *)
    R101_3축_리어_M_O_RB_7차_작업완료_리셋 : BOOL; (* AT %MW21032.6 *)
    R101_3축_리어_M_O_RB_7차_진입OK : BOOL; (* AT %MW21031.13 *)
    R101_3축_리어_M_O_RB_ATD_OK : BOOL; (* AT %MW21030.6 *)
    R101_3축_리어_M_O_RB_PLT_10_진입OK : BOOL; (* AT %MW21033.10 *)
    R101_3축_리어_M_O_RB_PLT_11_진입OK : BOOL; (* AT %MW21033.11 *)
    R101_3축_리어_M_O_RB_PLT_12_진입OK : BOOL; (* AT %MW21033.12 *)
    R101_3축_리어_M_O_RB_PLT_1_진입OK : BOOL; (* AT %MW21033.1 *)
    R101_3축_리어_M_O_RB_PLT_2_진입OK : BOOL; (* AT %MW21033.2 *)
    R101_3축_리어_M_O_RB_PLT_3_진입OK : BOOL; (* AT %MW21033.3 *)
    R101_3축_리어_M_O_RB_PLT_4_진입OK : BOOL; (* AT %MW21033.4 *)
    R101_3축_리어_M_O_RB_PLT_5_진입OK : BOOL; (* AT %MW21033.5 *)
    R101_3축_리어_M_O_RB_PLT_6_진입OK : BOOL; (* AT %MW21033.6 *)
    R101_3축_리어_M_O_RB_PLT_7_진입OK : BOOL; (* AT %MW21033.7 *)
    R101_3축_리어_M_O_RB_PLT_8_진입OK : BOOL; (* AT %MW21033.8 *)
    R101_3축_리어_M_O_RB_PLT_9_진입OK : BOOL; (* AT %MW21033.9 *)
    R101_3축_리어_M_O_RB_PLT_카운터리셋_보조 : BOOL; (* AT %MW21030.10 *)
    R101_3축_리어_M_O_RB_RESTART_OK : BOOL; (* AT %MW21030.2 *)
    R101_3축_리어_M_O_RB_START_OK : BOOL; (* AT %MW21030.0 *)
    R101_3축_리어_M_O_RB_TEST_MODE_5000회 : BOOL; (* AT %MW21030.12 *)
    R101_3축_리어_M_O_RB_TIP_교체_시작 : BOOL; (* AT %MW21030.7 *)
    R101_3축_리어_M_O_RB_TIP_교체_완료 : BOOL; (* AT %MW21030.8 *)
    R101_3축_리어_M_O_RB_VIP_MODE : BOOL; (* AT %MW21030.11 *)
    R101_3축_리어_M_O_RB_냉각수_차단_요청 : BOOL; (* AT %MW21030.9 *)
    R101_3축_리어_M_O_RB_진입OK_AX차종 : BOOL; (* AT %MW21031.0 *)
    R101_3축_리어_M_O_RB_진입OK_B차종 : BOOL; (* AT %MW21031.1 *)
    R101_3축_리어_M_O_RB_진입OK_C차종 : BOOL; (* AT %MW21031.2 *)
    R101_3축_리어_M_O_RB_진입OK_D차종 : BOOL; (* AT %MW21031.3 *)
    R101_3축_리어_M_O_RB_진입OK_E차종 : BOOL; (* AT %MW21031.4 *)
    R101_3축_리어_M_O_RB_진입OK_F차종 : BOOL; (* AT %MW21031.5 *)
    R101_3축_리어_M_O_RB_진입OK_G차종 : BOOL; (* AT %MW21031.6 *)
    R101_3축_리어_M_O_RB_진입OK_H차종 : BOOL; (* AT %MW21031.7 *)
    R101_3축_리어_M_O_RB_최종_작업완료_리셋 : BOOL; (* AT %MW21030.5 *)
    R101_3축_리어_M_O_RB_프로그램_OK : BOOL; (* AT %MW21030.1 *)
    R101_3축_리어_M_RB_PROG_NO : WORD; (* AT %MW20034 *)
    R101_3축_리어_O_RB_OUTPUT : ARRAY[0..3] OF WORD; (* AT %MW94030 *)
    R101_3축_센터_I_RB_INPUT : ARRAY[0..3] OF WORD; (* AT %MW84020 *)
    R101_3축_센터_M_I_RB_1차_작업완료 : BOOL; (* AT %MW20021.2 *)
    R101_3축_센터_M_I_RB_2차_작업완료 : BOOL; (* AT %MW20021.3 *)
    R101_3축_센터_M_I_RB_3차_작업완료 : BOOL; (* AT %MW20021.4 *)
    R101_3축_센터_M_I_RB_4차_작업완료 : BOOL; (* AT %MW20021.5 *)
    R101_3축_센터_M_I_RB_5차_작업완료 : BOOL; (* AT %MW20021.6 *)
    R101_3축_센터_M_I_RB_6차_작업완료 : BOOL; (* AT %MW20021.7 *)
    R101_3축_센터_M_I_RB_7차_작업완료 : BOOL; (* AT %MW20021.8 *)
    R101_3축_센터_M_I_RB_PAUSE_보조 : BOOL; (* AT %MW20020.5 *)
    R101_3축_센터_M_I_RB_PLC_RUN_CHK_이상 : BOOL; (* AT %MW20020.7 *)
    R101_3축_센터_M_I_RB_간섭무_1 : BOOL; (* AT %MW20022.0 *)
    R101_3축_센터_M_I_RB_간섭무_10 : BOOL; (* AT %MW20022.9 *)
    R101_3축_센터_M_I_RB_간섭무_11 : BOOL; (* AT %MW20022.10 *)
    R101_3축_센터_M_I_RB_간섭무_12 : BOOL; (* AT %MW20022.11 *)
    R101_3축_센터_M_I_RB_간섭무_2 : BOOL; (* AT %MW20022.1 *)
    R101_3축_센터_M_I_RB_간섭무_3 : BOOL; (* AT %MW20022.2 *)
    R101_3축_센터_M_I_RB_간섭무_4 : BOOL; (* AT %MW20022.3 *)
    R101_3축_센터_M_I_RB_간섭무_5 : BOOL; (* AT %MW20022.4 *)
    R101_3축_센터_M_I_RB_간섭무_6 : BOOL; (* AT %MW20022.5 *)
    R101_3축_센터_M_I_RB_간섭무_7 : BOOL; (* AT %MW20022.6 *)
    R101_3축_센터_M_I_RB_간섭무_8 : BOOL; (* AT %MW20022.7 *)
    R101_3축_센터_M_I_RB_간섭무_9 : BOOL; (* AT %MW20022.8 *)
    R101_3축_센터_M_I_RB_비상정지 : BOOL; (* AT %MW20020.4 *)
    R101_3축_센터_M_I_RB_운전준비 : BOOL; (* AT %MW20020.0 *)
    R101_3축_센터_M_I_RB_원위치 : BOOL; (* AT %MW20020.3 *)
    R101_3축_센터_M_I_RB_이상 : BOOL; (* AT %MW20020.2 *)
    R101_3축_센터_M_I_RB_자동 : BOOL; (* AT %MW20020.1 *)
    R101_3축_센터_M_I_RB_최종작업완료 : BOOL; (* AT %MW20021.0 *)
    R101_3축_센터_M_I_RB_프로그램_이상 : BOOL; (* AT %MW20020.6 *)
    R101_3축_센터_M_O_RB_1_CYCLE_SET : BOOL; (* AT %MW21020.3 *)
    R101_3축_센터_M_O_RB_1차_작업완료_리셋 : BOOL; (* AT %MW21022.0 *)
    R101_3축_센터_M_O_RB_2차_작업완료_리셋 : BOOL; (* AT %MW21022.1 *)
    R101_3축_센터_M_O_RB_2차_진입OK : BOOL; (* AT %MW21021.8 *)
    R101_3축_센터_M_O_RB_3차_작업완료_리셋 : BOOL; (* AT %MW21022.2 *)
    R101_3축_센터_M_O_RB_3차_진입OK : BOOL; (* AT %MW21021.9 *)
    R101_3축_센터_M_O_RB_4차_작업완료_리셋 : BOOL; (* AT %MW21022.3 *)
    R101_3축_센터_M_O_RB_4차_진입OK : BOOL; (* AT %MW21021.10 *)
    R101_3축_센터_M_O_RB_5차_작업완료_리셋 : BOOL; (* AT %MW21022.4 *)
    R101_3축_센터_M_O_RB_5차_진입OK : BOOL; (* AT %MW21021.11 *)
    R101_3축_센터_M_O_RB_6차_작업완료_리셋 : BOOL; (* AT %MW21022.5 *)
    R101_3축_센터_M_O_RB_6차_진입OK : BOOL; (* AT %MW21021.12 *)
    R101_3축_센터_M_O_RB_7차_작업완료_리셋 : BOOL; (* AT %MW21022.6 *)
    R101_3축_센터_M_O_RB_7차_진입OK : BOOL; (* AT %MW21021.13 *)
    R101_3축_센터_M_O_RB_ATD_OK : BOOL; (* AT %MW21020.6 *)
    R101_3축_센터_M_O_RB_PLT_10_진입OK : BOOL; (* AT %MW21023.10 *)
    R101_3축_센터_M_O_RB_PLT_11_진입OK : BOOL; (* AT %MW21023.11 *)
    R101_3축_센터_M_O_RB_PLT_12_진입OK : BOOL; (* AT %MW21023.12 *)
    R101_3축_센터_M_O_RB_PLT_1_진입OK : BOOL; (* AT %MW21023.1 *)
    R101_3축_센터_M_O_RB_PLT_2_진입OK : BOOL; (* AT %MW21023.2 *)
    R101_3축_센터_M_O_RB_PLT_3_진입OK : BOOL; (* AT %MW21023.3 *)
    R101_3축_센터_M_O_RB_PLT_4_진입OK : BOOL; (* AT %MW21023.4 *)
    R101_3축_센터_M_O_RB_PLT_5_진입OK : BOOL; (* AT %MW21023.5 *)
    R101_3축_센터_M_O_RB_PLT_6_진입OK : BOOL; (* AT %MW21023.6 *)
    R101_3축_센터_M_O_RB_PLT_7_진입OK : BOOL; (* AT %MW21023.7 *)
    R101_3축_센터_M_O_RB_PLT_8_진입OK : BOOL; (* AT %MW21023.8 *)
    R101_3축_센터_M_O_RB_PLT_9_진입OK : BOOL; (* AT %MW21023.9 *)
    R101_3축_센터_M_O_RB_PLT_카운터리셋_보조 : BOOL; (* AT %MW21020.10 *)
    R101_3축_센터_M_O_RB_RESTART_OK : BOOL; (* AT %MW21020.2 *)
    R101_3축_센터_M_O_RB_START_OK : BOOL; (* AT %MW21020.0 *)
    R101_3축_센터_M_O_RB_TEST_MODE_5000회 : BOOL; (* AT %MW21020.12 *)
    R101_3축_센터_M_O_RB_TIP_교체_시작 : BOOL; (* AT %MW21020.7 *)
    R101_3축_센터_M_O_RB_TIP_교체_완료 : BOOL; (* AT %MW21020.8 *)
    R101_3축_센터_M_O_RB_VIP_MODE : BOOL; (* AT %MW21020.11 *)
    R101_3축_센터_M_O_RB_냉각수_차단_요청 : BOOL; (* AT %MW21020.9 *)
    R101_3축_센터_M_O_RB_진입OK_AX차종 : BOOL; (* AT %MW21021.0 *)
    R101_3축_센터_M_O_RB_진입OK_B차종 : BOOL; (* AT %MW21021.1 *)
    R101_3축_센터_M_O_RB_진입OK_C차종 : BOOL; (* AT %MW21021.2 *)
    R101_3축_센터_M_O_RB_진입OK_D차종 : BOOL; (* AT %MW21021.3 *)
    R101_3축_센터_M_O_RB_진입OK_E차종 : BOOL; (* AT %MW21021.4 *)
    R101_3축_센터_M_O_RB_진입OK_F차종 : BOOL; (* AT %MW21021.5 *)
    R101_3축_센터_M_O_RB_진입OK_G차종 : BOOL; (* AT %MW21021.6 *)
    R101_3축_센터_M_O_RB_진입OK_H차종 : BOOL; (* AT %MW21021.7 *)
    R101_3축_센터_M_O_RB_최종_작업완료_리셋 : BOOL; (* AT %MW21020.5 *)
    R101_3축_센터_M_O_RB_프로그램_OK : BOOL; (* AT %MW21020.1 *)
    R101_3축_센터_M_RB_PROG_NO : WORD; (* AT %MW20024 *)
    R101_3축_센터_O_RB_OUTPUT : ARRAY[0..3] OF WORD; (* AT %MW94020 *)
    R101_3축_프론트_I_RB_INPUT : ARRAY[0..3] OF WORD; (* AT %MW84010 *)
    R101_3축_프론트_M_I_RB_1차_작업완료 : BOOL; (* AT %MW20011.2 *)
    R101_3축_프론트_M_I_RB_2차_작업완료 : BOOL; (* AT %MW20011.3 *)
    R101_3축_프론트_M_I_RB_3차_작업완료 : BOOL; (* AT %MW20011.4 *)
    R101_3축_프론트_M_I_RB_4차_작업완료 : BOOL; (* AT %MW20011.5 *)
    R101_3축_프론트_M_I_RB_5차_작업완료 : BOOL; (* AT %MW20011.6 *)
    R101_3축_프론트_M_I_RB_6차_작업완료 : BOOL; (* AT %MW20011.7 *)
    R101_3축_프론트_M_I_RB_7차_작업완료 : BOOL; (* AT %MW20011.8 *)
    R101_3축_프론트_M_I_RB_PAUSE_보조 : BOOL; (* AT %MW20010.5 *)
    R101_3축_프론트_M_I_RB_PLC_RUN_CHK_이상 : BOOL; (* AT %MW20010.7 *)
    R101_3축_프론트_M_I_RB_간섭무_1 : BOOL; (* AT %MW20012.0 *)
    R101_3축_프론트_M_I_RB_간섭무_10 : BOOL; (* AT %MW20012.9 *)
    R101_3축_프론트_M_I_RB_간섭무_11 : BOOL; (* AT %MW20012.10 *)
    R101_3축_프론트_M_I_RB_간섭무_12 : BOOL; (* AT %MW20012.11 *)
    R101_3축_프론트_M_I_RB_간섭무_2 : BOOL; (* AT %MW20012.1 *)
    R101_3축_프론트_M_I_RB_간섭무_3 : BOOL; (* AT %MW20012.2 *)
    R101_3축_프론트_M_I_RB_간섭무_4 : BOOL; (* AT %MW20012.3 *)
    R101_3축_프론트_M_I_RB_간섭무_5 : BOOL; (* AT %MW20012.4 *)
    R101_3축_프론트_M_I_RB_간섭무_6 : BOOL; (* AT %MW20012.5 *)
    R101_3축_프론트_M_I_RB_간섭무_7 : BOOL; (* AT %MW20012.6 *)
    R101_3축_프론트_M_I_RB_간섭무_8 : BOOL; (* AT %MW20012.7 *)
    R101_3축_프론트_M_I_RB_간섭무_9 : BOOL; (* AT %MW20012.8 *)
    R101_3축_프론트_M_I_RB_비상정지 : BOOL; (* AT %MW20010.4 *)
    R101_3축_프론트_M_I_RB_운전준비 : BOOL; (* AT %MW20010.0 *)
    R101_3축_프론트_M_I_RB_원위치 : BOOL; (* AT %MW20010.3 *)
    R101_3축_프론트_M_I_RB_이상 : BOOL; (* AT %MW20010.2 *)
    R101_3축_프론트_M_I_RB_자동 : BOOL; (* AT %MW20010.1 *)
    R101_3축_프론트_M_I_RB_최종작업완료 : BOOL; (* AT %MW20011.0 *)
    R101_3축_프론트_M_I_RB_프로그램_이상 : BOOL; (* AT %MW20010.6 *)
    R101_3축_프론트_M_O_RB_1_CYCLE_SET : BOOL; (* AT %MW21010.3 *)
    R101_3축_프론트_M_O_RB_1차_작업완료_리셋 : BOOL; (* AT %MW21012.0 *)
    R101_3축_프론트_M_O_RB_2차_작업완료_리셋 : BOOL; (* AT %MW21012.1 *)
    R101_3축_프론트_M_O_RB_2차_진입OK : BOOL; (* AT %MW21011.8 *)
    R101_3축_프론트_M_O_RB_3차_작업완료_리셋 : BOOL; (* AT %MW21012.2 *)
    R101_3축_프론트_M_O_RB_3차_진입OK : BOOL; (* AT %MW21011.9 *)
    R101_3축_프론트_M_O_RB_4차_작업완료_리셋 : BOOL; (* AT %MW21012.3 *)
    R101_3축_프론트_M_O_RB_4차_진입OK : BOOL; (* AT %MW21011.10 *)
    R101_3축_프론트_M_O_RB_5차_작업완료_리셋 : BOOL; (* AT %MW21012.4 *)
    R101_3축_프론트_M_O_RB_5차_진입OK : BOOL; (* AT %MW21011.11 *)
    R101_3축_프론트_M_O_RB_6차_작업완료_리셋 : BOOL; (* AT %MW21012.5 *)
    R101_3축_프론트_M_O_RB_6차_진입OK : BOOL; (* AT %MW21011.12 *)
    R101_3축_프론트_M_O_RB_7차_작업완료_리셋 : BOOL; (* AT %MW21012.6 *)
    R101_3축_프론트_M_O_RB_7차_진입OK : BOOL; (* AT %MW21011.13 *)
    R101_3축_프론트_M_O_RB_ATD_OK : BOOL; (* AT %MW21010.6 *)
    R101_3축_프론트_M_O_RB_PLT_10_진입OK : BOOL; (* AT %MW21013.10 *)
    R101_3축_프론트_M_O_RB_PLT_11_진입OK : BOOL; (* AT %MW21013.11 *)
    R101_3축_프론트_M_O_RB_PLT_12_진입OK : BOOL; (* AT %MW21013.12 *)
    R101_3축_프론트_M_O_RB_PLT_1_진입OK : BOOL; (* AT %MW21013.1 *)
    R101_3축_프론트_M_O_RB_PLT_2_진입OK : BOOL; (* AT %MW21013.2 *)
    R101_3축_프론트_M_O_RB_PLT_3_진입OK : BOOL; (* AT %MW21013.3 *)
    R101_3축_프론트_M_O_RB_PLT_4_진입OK : BOOL; (* AT %MW21013.4 *)
    R101_3축_프론트_M_O_RB_PLT_5_진입OK : BOOL; (* AT %MW21013.5 *)
    R101_3축_프론트_M_O_RB_PLT_6_진입OK : BOOL; (* AT %MW21013.6 *)
    R101_3축_프론트_M_O_RB_PLT_7_진입OK : BOOL; (* AT %MW21013.7 *)
    R101_3축_프론트_M_O_RB_PLT_8_진입OK : BOOL; (* AT %MW21013.8 *)
    R101_3축_프론트_M_O_RB_PLT_9_진입OK : BOOL; (* AT %MW21013.9 *)
    R101_3축_프론트_M_O_RB_PLT_카운터리셋_보조 : BOOL; (* AT %MW21010.10 *)
    R101_3축_프론트_M_O_RB_RESTART_OK : BOOL; (* AT %MW21010.2 *)
    R101_3축_프론트_M_O_RB_START_OK : BOOL; (* AT %MW21010.0 *)
    R101_3축_프론트_M_O_RB_TEST_MODE_5000회 : BOOL; (* AT %MW21010.12 *)
    R101_3축_프론트_M_O_RB_TIP_교체_시작 : BOOL; (* AT %MW21010.7 *)
    R101_3축_프론트_M_O_RB_TIP_교체_완료 : BOOL; (* AT %MW21010.8 *)
    R101_3축_프론트_M_O_RB_VIP_MODE : BOOL; (* AT %MW21010.11 *)
    R101_3축_프론트_M_O_RB_냉각수_차단_요청 : BOOL; (* AT %MW21010.9 *)
    R101_3축_프론트_M_O_RB_진입OK_AX차종 : BOOL; (* AT %MW21011.0 *)
    R101_3축_프론트_M_O_RB_진입OK_B차종 : BOOL; (* AT %MW21011.1 *)
    R101_3축_프론트_M_O_RB_진입OK_C차종 : BOOL; (* AT %MW21011.2 *)
    R101_3축_프론트_M_O_RB_진입OK_D차종 : BOOL; (* AT %MW21011.3 *)
    R101_3축_프론트_M_O_RB_진입OK_E차종 : BOOL; (* AT %MW21011.4 *)
    R101_3축_프론트_M_O_RB_진입OK_F차종 : BOOL; (* AT %MW21011.5 *)
    R101_3축_프론트_M_O_RB_진입OK_G차종 : BOOL; (* AT %MW21011.6 *)
    R101_3축_프론트_M_O_RB_진입OK_H차종 : BOOL; (* AT %MW21011.7 *)
    R101_3축_프론트_M_O_RB_최종_작업완료_리셋 : BOOL; (* AT %MW21010.5 *)
    R101_3축_프론트_M_O_RB_프로그램_OK : BOOL; (* AT %MW21010.1 *)
    R101_3축_프론트_M_RB_PROG_NO : WORD; (* AT %MW20014 *)
    R101_3축_프론트_O_RB_OUTPUT : ARRAY[0..3] OF WORD; (* AT %MW94010 *)
    S101_LH_M_APRON_PLT1_FAULT : BOOL; (* AT %MW1200.6 *)
    S101_LH_M_APRON_PLT1_MATCH_OK : BOOL; (* AT %MW1200.5 *)
    S101_LH_M_APRON_PLT1_PROG_OK : BOOL; (* AT %MW1200.0 *)
    S101_LH_M_APRON_PLT1_차종코드 : WORD; (* AT %MW1216 *)
    S101_LH_M_APRON_PLT2_FAULT : BOOL; (* AT %MW1201.6 *)
    S101_LH_M_APRON_PLT2_MATCH_OK : BOOL; (* AT %MW1201.5 *)
    S101_LH_M_APRON_PLT2_PROG_OK : BOOL; (* AT %MW1201.0 *)
    S101_LH_M_APRON_PLT2_차종코드 : WORD; (* AT %MW1217 *)
    S101_LH_M_APRON_PLT3_차종코드 : WORD; (* AT %MW1218 *)
    S101_LH_M_APRON_PLT_PRIORITY1 : WORD; (* AT %MW1208 *)
    S101_M_AX_래치_전진단 : BOOL; (* AT %MW1100.3 *)
    S101_M_DASH_클램프_후진단 : BOOL; (* AT %MW1105.4 *)
    S101_M_SHIFT_후진단 : BOOL; (* AT %MW1101.4 *)
    S101_M_STN_DASH_로딩완료 : BOOL; (* AT %MW1001.12 *)
    S101_M_STN_LH_로딩완료 : BOOL; (* AT %MW1001.10 *)
    S101_M_STN_RH_로딩완료 : BOOL; (* AT %MW1001.11 *)
    S101_M_STN_차종_NONE : BOOL; (* AT %MW1002.1 *)
    S101_M_STN_차종_ON : BOOL; (* AT %MW1002.0 *)
    S101_M_공정_APRON_제품감지_ON : BOOL; (* AT %MW1001.3 *)
    S101_M_공정_DASH_제품감지_ON : BOOL; (* AT %MW1001.5 *)
    S101_M_공정_간섭무 : BOOL; (* AT %MW1004.1 *)
    S101_M_수동_모드 : BOOL; (* AT %MW1000.3 *)
    S101_M_자동_START : BOOL; (* AT %MW1000.5 *)
    S101_M_자동_운전중 : BOOL; (* AT %MW1000.4 *)
    S101_M_작업_완료 : BOOL; (* AT %MW1001.0 *)
    S101_M_전체_3축_로봇1차_작업완료 : BOOL; (* AT %MW1001.1 *)
    S101_M_전체_용접로보트_1차_작업완료 : BOOL; (* AT %MW1001.8 *)
    S101_M_전체_용접로보트_최종_작업완료 : BOOL; (* AT %MW1001.9 *)
    S101_M_전체_클램프_잠김단 : BOOL; (* AT %MW1004.12 *)
    S101_M_차종1_AX : BOOL; (* AT %MW10021.0 *) (* S101_M_차종1_AX *)
    S101_M_총괄_이상 : BOOL; (* AT %MW1009.0 *)
    S101_M_핀클램프_후진단 : BOOL; (* AT %MW1106.4 *)
    S101_PRS_I_AX_LH_파트_ON : BOOL; (* AT %MW86102.0 *)
    S101_PRS_I_AX_RH_파트_ON : BOOL; (* AT %MW86102.1 *)
    S101_RH_M_APRON_PLT1_FAULT : BOOL; (* AT %MW1250.6 *)
    S101_RH_M_APRON_PLT1_MATCH_OK : BOOL; (* AT %MW1250.5 *)
    S101_RH_M_APRON_PLT1_PROG_OK : BOOL; (* AT %MW1250.0 *)
    S101_RH_M_APRON_PLT1_차종코드 : WORD; (* AT %MW1266 *)
    S101_RH_M_APRON_PLT2_FAULT : BOOL; (* AT %MW1251.6 *)
    S101_RH_M_APRON_PLT2_MATCH_OK : BOOL; (* AT %MW1251.5 *)
    S101_RH_M_APRON_PLT2_PROG_OK : BOOL; (* AT %MW1251.0 *)
    S101_RH_M_APRON_PLT2_차종코드 : WORD; (* AT %MW1267 *)
    S101_RH_M_APRON_PLT_PRIORITY1 : WORD; (* AT %MW1258 *)
    로보트제외 : BOOL;
    셔틀_M_작업완료 : BOOL; (* AT %MW501.0 *)
    전체_M_GATE_CYCLE_정지 : BOOL; (* AT %MW308.0 *) (* 전체 M GATE CYCLE STOP *)
    전체_M_GATE_비상정지_정상 : BOOL; (* AT %MW308.4 *)
    전체_M_운전준비_보조 : BOOL; (* AT %MW308.5 *)
    전체_M_이상_리셋 : BOOL; (* AT %MW308.2 *) (* 전체 M 이상 리셋 *)
    전체_공정_M_총괄_비상정지_정상 : BOOL; (* AT %MW304.1 *) (* 전체 공정 M 총괄 비상정지 정상 *)
END_VAR
VAR
    INST : FB494_Robot_Hyundai_HMMI_v1;
    INST1 : FB494_Robot_Hyundai_HMMI_v1;
    INST2 : FB494_Robot_Hyundai_HMMI_v1;
    INST3 : FB494_Robot_Hyundai_HMMI_v1;
    INST4 : FB494_Robot_Hyundai_HMMI_v1;
    INST5 : FB494_Robot_Hyundai_HMMI_v1;
    INST6 : FB494_Robot_Hyundai_HMMI_v1;
    _R101_1_1_PLT_언로딩완료 : BOOL;
    _작업완료_SET_BIT : BOOL;
END_VAR
(* ladder body could not be read *)
END_PROGRAM

PROGRAM S101_3축_로보트 (* task: 스캔 프로그램 *)
VAR_EXTERNAL
    AWAYS_OFF : BOOL; (* AT %MW3.0 *)
    AWAYS_ON : BOOL; (* AT %MW3.1 *)
    MCP_M_부저_정지 : BOOL; (* AT %MW350.5 *)
    MCP_M_비상정지 : BOOL; (* AT %MW350.7 *)
    MCP_PBL_운전준비_ON : BOOL; (* AT %MW87630.0 *) (* 입력 접점 00 *)
    R101_1_M_I_RB_1차_작업완료 : BOOL; (* AT %MW20071.2 *)
    R101_1_M_I_RB_최종작업완료 : BOOL; (* AT %MW20071.0 *)
    R101_1_M_O_RB_1차_작업완료_리셋 : BOOL; (* AT %MW21072.0 *)
    R101_1_M_O_RB_최종_작업완료_리셋 : BOOL; (* AT %MW21070.5 *)
    R101_2_M_I_RB_1차_작업완료 : BOOL; (* AT %MW20061.2 *)
    R101_2_M_I_RB_최종작업완료 : BOOL; (* AT %MW20061.0 *)
    R101_2_M_O_RB_1차_작업완료_리셋 : BOOL; (* AT %MW21062.0 *)
    R101_2_M_O_RB_최종_작업완료_리셋 : BOOL; (* AT %MW21060.5 *)
    R101_3축_리어_I_RB_INPUT : ARRAY[0..3] OF WORD; (* AT %MW84030 *)
    R101_3축_리어_M_I_RB_1차_작업완료 : BOOL; (* AT %MW20031.2 *)
    R101_3축_리어_M_I_RB_2차_작업완료 : BOOL; (* AT %MW20031.3 *)
    R101_3축_리어_M_I_RB_3차_작업완료 : BOOL; (* AT %MW20031.4 *)
    R101_3축_리어_M_I_RB_4차_작업완료 : BOOL; (* AT %MW20031.5 *)
    R101_3축_리어_M_I_RB_5차_작업완료 : BOOL; (* AT %MW20031.6 *)
    R101_3축_리어_M_I_RB_6차_작업완료 : BOOL; (* AT %MW20031.7 *)
    R101_3축_리어_M_I_RB_7차_작업완료 : BOOL; (* AT %MW20031.8 *)
    R101_3축_리어_M_I_RB_PAUSE_보조 : BOOL; (* AT %MW20030.5 *)
    R101_3축_리어_M_I_RB_PLC_RUN_CHK_이상 : BOOL; (* AT %MW20030.7 *)
    R101_3축_리어_M_I_RB_간섭무_1 : BOOL; (* AT %MW20032.0 *)
    R101_3축_리어_M_I_RB_간섭무_10 : BOOL; (* AT %MW20032.9 *)
    R101_3축_리어_M_I_RB_간섭무_11 : BOOL; (* AT %MW20032.10 *)
    R101_3축_리어_M_I_RB_간섭무_12 : BOOL; (* AT %MW20032.11 *)
    R101_3축_리어_M_I_RB_간섭무_2 : BOOL; (* AT %MW20032.1 *)
    R101_3축_리어_M_I_RB_간섭무_3 : BOOL; (* AT %MW20032.2 *)
    R101_3축_리어_M_I_RB_간섭무_4 : BOOL; (* AT %MW20032.3 *)
    R101_3축_리어_M_I_RB_간섭무_5 : BOOL; (* AT %MW20032.4 *)
    R101_3축_리어_M_I_RB_간섭무_6 : BOOL; (* AT %MW20032.5 *)
    R101_3축_리어_M_I_RB_간섭무_7 : BOOL; (* AT %MW20032.6 *)
    R101_3축_리어_M_I_RB_간섭무_8 : BOOL; (* AT %MW20032.7 *)
    R101_3축_리어_M_I_RB_간섭무_9 : BOOL; (* AT %MW20032.8 *)
    R101_3축_리어_M_I_RB_비상정지 : BOOL; (* AT %MW20030.4 *)
    R101_3축_리어_M_I_RB_운전준비 : BOOL; (* AT %MW20030.0 *)
    R101_3축_리어_M_I_RB_원위치 : BOOL; (* AT %MW20030.3 *)
    R101_3축_리어_M_I_RB_이상 : BOOL; (* AT %MW20030.2 *)
    R101_3축_리어_M_I_RB_자동 : BOOL; (* AT %MW20030.1 *)
    R101_3축_리어_M_I_RB_최종작업완료 : BOOL; (* AT %MW20031.0 *)
    R101_3축_리어_M_I_RB_프로그램_이상 : BOOL; (* AT %MW20030.6 *)
    R101_3축_리어_M_O_RB_1_CYCLE_SET : BOOL; (* AT %MW21030.3 *)
    R101_3축_리어_M_O_RB_1차_작업완료_리셋 : BOOL; (* AT %MW21032.0 *)
    R101_3축_리어_M_O_RB_2차_작업완료_리셋 : BOOL; (* AT %MW21032.1 *)
    R101_3축_리어_M_O_RB_2차_진입OK : BOOL; (* AT %MW21031.8 *)
    R101_3축_리어_M_O_RB_3차_작업완료_리셋 : BOOL; (* AT %MW21032.2 *)
    R101_3축_리어_M_O_RB_3차_진입OK : BOOL; (* AT %MW21031.9 *)
    R101_3축_리어_M_O_RB_4차_작업완료_리셋 : BOOL; (* AT %MW21032.3 *)
    R101_3축_리어_M_O_RB_4차_진입OK : BOOL; (* AT %MW21031.10 *)
    R101_3축_리어_M_O_RB_5차_작업완료_리셋 : BOOL; (* AT %MW21032.4 *)
    R101_3축_리어_M_O_RB_5차_진입OK : BOOL; (* AT %MW21031.11 *)
    R101_3축_리어_M_O_RB_6차_작업완료_리셋 : BOOL; (* AT %MW21032.5 *)
    R101_3축_리어_M_O_RB_6차_진입OK : BOOL; (* AT %MW21031.12 *)
    R101_3축_리어_M_O_RB_7차_작업완료_리셋 : BOOL; (* AT %MW21032.6 *)
    R101_3축_리어_M_O_RB_7차_진입OK : BOOL; (* AT %MW21031.13 *)
    R101_3축_리어_M_O_RB_ATD_OK : BOOL; (* AT %MW21030.6 *)
    R101_3축_리어_M_O_RB_PLT_10_진입OK : BOOL; (* AT %MW21033.10 *)
    R101_3축_리어_M_O_RB_PLT_11_진입OK : BOOL; (* AT %MW21033.11 *)
    R101_3축_리어_M_O_RB_PLT_12_진입OK : BOOL; (* AT %MW21033.12 *)
    R101_3축_리어_M_O_RB_PLT_1_진입OK : BOOL; (* AT %MW21033.1 *)
    R101_3축_리어_M_O_RB_PLT_2_진입OK : BOOL; (* AT %MW21033.2 *)
    R101_3축_리어_M_O_RB_PLT_3_진입OK : BOOL; (* AT %MW21033.3 *)
    R101_3축_리어_M_O_RB_PLT_4_진입OK : BOOL; (* AT %MW21033.4 *)
    R101_3축_리어_M_O_RB_PLT_5_진입OK : BOOL; (* AT %MW21033.5 *)
    R101_3축_리어_M_O_RB_PLT_6_진입OK : BOOL; (* AT %MW21033.6 *)
    R101_3축_리어_M_O_RB_PLT_7_진입OK : BOOL; (* AT %MW21033.7 *)
    R101_3축_리어_M_O_RB_PLT_8_진입OK : BOOL; (* AT %MW21033.8 *)
    R101_3축_리어_M_O_RB_PLT_9_진입OK : BOOL; (* AT %MW21033.9 *)
    R101_3축_리어_M_O_RB_PLT_카운터리셋_보조 : BOOL; (* AT %MW21030.10 *)
    R101_3축_리어_M_O_RB_RESTART_OK : BOOL; (* AT %MW21030.2 *)
    R101_3축_리어_M_O_RB_START_OK : BOOL; (* AT %MW21030.0 *)
    R101_3축_리어_M_O_RB_TEST_MODE_5000회 : BOOL; (* AT %MW21030.12 *)
    R101_3축_리어_M_O_RB_TIP_교체_시작 : BOOL; (* AT %MW21030.7 *)
    R101_3축_리어_M_O_RB_TIP_교체_완료 : BOOL; (* AT %MW21030.8 *)
    R101_3축_리어_M_O_RB_VIP_MODE : BOOL; (* AT %MW21030.11 *)
    R101_3축_리어_M_O_RB_냉각수_차단_요청 : BOOL; (* AT %MW21030.9 *)
    R101_3축_리어_M_O_RB_진입OK_AX차종 : BOOL; (* AT %MW21031.0 *)
    R101_3축_리어_M_O_RB_진입OK_B차종 : BOOL; (* AT %MW21031.1 *)
    R101_3축_리어_M_O_RB_진입OK_C차종 : BOOL; (* AT %MW21031.2 *)
    R101_3축_리어_M_O_RB_진입OK_D차종 : BOOL; (* AT %MW21031.3 *)
    R101_3축_리어_M_O_RB_진입OK_E차종 : BOOL; (* AT %MW21031.4 *)
    R101_3축_리어_M_O_RB_진입OK_F차종 : BOOL; (* AT %MW21031.5 *)
    R101_3축_리어_M_O_RB_진입OK_G차종 : BOOL; (* AT %MW21031.6 *)
    R101_3축_리어_M_O_RB_진입OK_H차종 : BOOL; (* AT %MW21031.7 *)
    R101_3축_리어_M_O_RB_최종_작업완료_리셋 : BOOL; (* AT %MW21030.5 *)
    R101_3축_리어_M_O_RB_프로그램_OK : BOOL; (* AT %MW21030.1 *)
    R101_3축_리어_M_RB_PROG_NO : WORD; (* AT %MW20034 *)
    R101_3축_리어_O_RB_OUTPUT : ARRAY[0..3] OF WORD; (* AT %MW94030 *)
    R101_3축_센터_I_RB_INPUT : ARRAY[0..3] OF WORD; (* AT %MW84020 *)
    R101_3축_센터_M_I_RB_1차_작업완료 : BOOL; (* AT %MW20021.2 *)
    R101_3축_센터_M_I_RB_2차_작업완료 : BOOL; (* AT %MW20021.3 *)
    R101_3축_센터_M_I_RB_3차_작업완료 : BOOL; (* AT %MW20021.4 *)
    R101_3축_센터_M_I_RB_4차_작업완료 : BOOL; (* AT %MW20021.5 *)
    R101_3축_센터_M_I_RB_5차_작업완료 : BOOL; (* AT %MW20021.6 *)
    R101_3축_센터_M_I_RB_6차_작업완료 : BOOL; (* AT %MW20021.7 *)
    R101_3축_센터_M_I_RB_7차_작업완료 : BOOL; (* AT %MW20021.8 *)
    R101_3축_센터_M_I_RB_PAUSE_보조 : BOOL; (* AT %MW20020.5 *)
    R101_3축_센터_M_I_RB_PLC_RUN_CHK_이상 : BOOL; (* AT %MW20020.7 *)
    R101_3축_센터_M_I_RB_간섭무_1 : BOOL; (* AT %MW20022.0 *)
    R101_3축_센터_M_I_RB_간섭무_10 : BOOL; (* AT %MW20022.9 *)
    R101_3축_센터_M_I_RB_간섭무_11 : BOOL; (* AT %MW20022.10 *)
    R101_3축_센터_M_I_RB_간섭무_12 : BOOL; (* AT %MW20022.11 *)
    R101_3축_센터_M_I_RB_간섭무_2 : BOOL; (* AT %MW20022.1 *)
    R101_3축_센터_M_I_RB_간섭무_3 : BOOL; (* AT %MW20022.2 *)
    R101_3축_센터_M_I_RB_간섭무_4 : BOOL; (* AT %MW20022.3 *)
    R101_3축_센터_M_I_RB_간섭무_5 : BOOL; (* AT %MW20022.4 *)
    R101_3축_센터_M_I_RB_간섭무_6 : BOOL; (* AT %MW20022.5 *)
    R101_3축_센터_M_I_RB_간섭무_7 : BOOL; (* AT %MW20022.6 *)
    R101_3축_센터_M_I_RB_간섭무_8 : BOOL; (* AT %MW20022.7 *)
    R101_3축_센터_M_I_RB_간섭무_9 : BOOL; (* AT %MW20022.8 *)
    R101_3축_센터_M_I_RB_비상정지 : BOOL; (* AT %MW20020.4 *)
    R101_3축_센터_M_I_RB_운전준비 : BOOL; (* AT %MW20020.0 *)
    R101_3축_센터_M_I_RB_원위치 : BOOL; (* AT %MW20020.3 *)
    R101_3축_센터_M_I_RB_이상 : BOOL; (* AT %MW20020.2 *)
    R101_3축_센터_M_I_RB_자동 : BOOL; (* AT %MW20020.1 *)
    R101_3축_센터_M_I_RB_최종작업완료 : BOOL; (* AT %MW20021.0 *)
    R101_3축_센터_M_I_RB_프로그램_이상 : BOOL; (* AT %MW20020.6 *)
    R101_3축_센터_M_O_RB_1_CYCLE_SET : BOOL; (* AT %MW21020.3 *)
    R101_3축_센터_M_O_RB_1차_작업완료_리셋 : BOOL; (* AT %MW21022.0 *)
    R101_3축_센터_M_O_RB_2차_작업완료_리셋 : BOOL; (* AT %MW21022.1 *)
    R101_3축_센터_M_O_RB_2차_진입OK : BOOL; (* AT %MW21021.8 *)
    R101_3축_센터_M_O_RB_3차_작업완료_리셋 : BOOL; (* AT %MW21022.2 *)
    R101_3축_센터_M_O_RB_3차_진입OK : BOOL; (* AT %MW21021.9 *)
    R101_3축_센터_M_O_RB_4차_작업완료_리셋 : BOOL; (* AT %MW21022.3 *)
    R101_3축_센터_M_O_RB_4차_진입OK : BOOL; (* AT %MW21021.10 *)
    R101_3축_센터_M_O_RB_5차_작업완료_리셋 : BOOL; (* AT %MW21022.4 *)
    R101_3축_센터_M_O_RB_5차_진입OK : BOOL; (* AT %MW21021.11 *)
    R101_3축_센터_M_O_RB_6차_작업완료_리셋 : BOOL; (* AT %MW21022.5 *)
    R101_3축_센터_M_O_RB_6차_진입OK : BOOL; (* AT %MW21021.12 *)
    R101_3축_센터_M_O_RB_7차_작업완료_리셋 : BOOL; (* AT %MW21022.6 *)
    R101_3축_센터_M_O_RB_7차_진입OK : BOOL; (* AT %MW21021.13 *)
    R101_3축_센터_M_O_RB_ATD_OK : BOOL; (* AT %MW21020.6 *)
    R101_3축_센터_M_O_RB_PLT_10_진입OK : BOOL; (* AT %MW21023.10 *)
    R101_3축_센터_M_O_RB_PLT_11_진입OK : BOOL; (* AT %MW21023.11 *)
    R101_3축_센터_M_O_RB_PLT_12_진입OK : BOOL; (* AT %MW21023.12 *)
    R101_3축_센터_M_O_RB_PLT_1_진입OK : BOOL; (* AT %MW21023.1 *)
    R101_3축_센터_M_O_RB_PLT_2_진입OK : BOOL; (* AT %MW21023.2 *)
    R101_3축_센터_M_O_RB_PLT_3_진입OK : BOOL; (* AT %MW21023.3 *)
    R101_3축_센터_M_O_RB_PLT_4_진입OK : BOOL; (* AT %MW21023.4 *)
    R101_3축_센터_M_O_RB_PLT_5_진입OK : BOOL; (* AT %MW21023.5 *)
    R101_3축_센터_M_O_RB_PLT_6_진입OK : BOOL; (* AT %MW21023.6 *)
    R101_3축_센터_M_O_RB_PLT_7_진입OK : BOOL; (* AT %MW21023.7 *)
    R101_3축_센터_M_O_RB_PLT_8_진입OK : BOOL; (* AT %MW21023.8 *)
    R101_3축_센터_M_O_RB_PLT_9_진입OK : BOOL; (* AT %MW21023.9 *)
    R101_3축_센터_M_O_RB_PLT_카운터리셋_보조 : BOOL; (* AT %MW21020.10 *)
    R101_3축_센터_M_O_RB_RESTART_OK : BOOL; (* AT %MW21020.2 *)
    R101_3축_센터_M_O_RB_START_OK : BOOL; (* AT %MW21020.0 *)
    R101_3축_센터_M_O_RB_TEST_MODE_5000회 : BOOL; (* AT %MW21020.12 *)
    R101_3축_센터_M_O_RB_TIP_교체_시작 : BOOL; (* AT %MW21020.7 *)
    R101_3축_센터_M_O_RB_TIP_교체_완료 : BOOL; (* AT %MW21020.8 *)
    R101_3축_센터_M_O_RB_VIP_MODE : BOOL; (* AT %MW21020.11 *)
    R101_3축_센터_M_O_RB_냉각수_차단_요청 : BOOL; (* AT %MW21020.9 *)
    R101_3축_센터_M_O_RB_진입OK_AX차종 : BOOL; (* AT %MW21021.0 *)
    R101_3축_센터_M_O_RB_진입OK_B차종 : BOOL; (* AT %MW21021.1 *)
    R101_3축_센터_M_O_RB_진입OK_C차종 : BOOL; (* AT %MW21021.2 *)
    R101_3축_센터_M_O_RB_진입OK_D차종 : BOOL; (* AT %MW21021.3 *)
    R101_3축_센터_M_O_RB_진입OK_E차종 : BOOL; (* AT %MW21021.4 *)
    R101_3축_센터_M_O_RB_진입OK_F차종 : BOOL; (* AT %MW21021.5 *)
    R101_3축_센터_M_O_RB_진입OK_G차종 : BOOL; (* AT %MW21021.6 *)
    R101_3축_센터_M_O_RB_진입OK_H차종 : BOOL; (* AT %MW21021.7 *)
    R101_3축_센터_M_O_RB_최종_작업완료_리셋 : BOOL; (* AT %MW21020.5 *)
    R101_3축_센터_M_O_RB_프로그램_OK : BOOL; (* AT %MW21020.1 *)
    R101_3축_센터_M_RB_PROG_NO : WORD; (* AT %MW20024 *)
    R101_3축_센터_O_RB_OUTPUT : ARRAY[0..3] OF WORD; (* AT %MW94020 *)
    R101_3축_프론트_I_RB_INPUT : ARRAY[0..3] OF WORD; (* AT %MW84010 *)
    R101_3축_프론트_M_I_RB_1차_작업완료 : BOOL; (* AT %MW20011.2 *)
    R101_3축_프론트_M_I_RB_2차_작업완료 : BOOL; (* AT %MW20011.3 *)
    R101_3축_프론트_M_I_RB_3차_작업완료 : BOOL; (* AT %MW20011.4 *)
    R101_3축_프론트_M_I_RB_4차_작업완료 : BOOL; (* AT %MW20011.5 *)
    R101_3축_프론트_M_I_RB_5차_작업완료 : BOOL; (* AT %MW20011.6 *)
    R101_3축_프론트_M_I_RB_6차_작업완료 : BOOL; (* AT %MW20011.7 *)
    R101_3축_프론트_M_I_RB_7차_작업완료 : BOOL; (* AT %MW20011.8 *)
    R101_3축_프론트_M_I_RB_PAUSE_보조 : BOOL; (* AT %MW20010.5 *)
    R101_3축_프론트_M_I_RB_PLC_RUN_CHK_이상 : BOOL; (* AT %MW20010.7 *)
    R101_3축_프론트_M_I_RB_간섭무_1 : BOOL; (* AT %MW20012.0 *)
    R101_3축_프론트_M_I_RB_간섭무_10 : BOOL; (* AT %MW20012.9 *)
    R101_3축_프론트_M_I_RB_간섭무_11 : BOOL; (* AT %MW20012.10 *)
    R101_3축_프론트_M_I_RB_간섭무_12 : BOOL; (* AT %MW20012.11 *)
    R101_3축_프론트_M_I_RB_간섭무_2 : BOOL; (* AT %MW20012.1 *)
    R101_3축_프론트_M_I_RB_간섭무_3 : BOOL; (* AT %MW20012.2 *)
    R101_3축_프론트_M_I_RB_간섭무_4 : BOOL; (* AT %MW20012.3 *)
    R101_3축_프론트_M_I_RB_간섭무_5 : BOOL; (* AT %MW20012.4 *)
    R101_3축_프론트_M_I_RB_간섭무_6 : BOOL; (* AT %MW20012.5 *)
    R101_3축_프론트_M_I_RB_간섭무_7 : BOOL; (* AT %MW20012.6 *)
    R101_3축_프론트_M_I_RB_간섭무_8 : BOOL; (* AT %MW20012.7 *)
    R101_3축_프론트_M_I_RB_간섭무_9 : BOOL; (* AT %MW20012.8 *)
    R101_3축_프론트_M_I_RB_비상정지 : BOOL; (* AT %MW20010.4 *)
    R101_3축_프론트_M_I_RB_운전준비 : BOOL; (* AT %MW20010.0 *)
    R101_3축_프론트_M_I_RB_원위치 : BOOL; (* AT %MW20010.3 *)
    R101_3축_프론트_M_I_RB_이상 : BOOL; (* AT %MW20010.2 *)
    R101_3축_프론트_M_I_RB_자동 : BOOL; (* AT %MW20010.1 *)
    R101_3축_프론트_M_I_RB_최종작업완료 : BOOL; (* AT %MW20011.0 *)
    R101_3축_프론트_M_I_RB_프로그램_이상 : BOOL; (* AT %MW20010.6 *)
    R101_3축_프론트_M_O_RB_1_CYCLE_SET : BOOL; (* AT %MW21010.3 *)
    R101_3축_프론트_M_O_RB_1차_작업완료_리셋 : BOOL; (* AT %MW21012.0 *)
    R101_3축_프론트_M_O_RB_2차_작업완료_리셋 : BOOL; (* AT %MW21012.1 *)
    R101_3축_프론트_M_O_RB_2차_진입OK : BOOL; (* AT %MW21011.8 *)
    R101_3축_프론트_M_O_RB_3차_작업완료_리셋 : BOOL; (* AT %MW21012.2 *)
    R101_3축_프론트_M_O_RB_3차_진입OK : BOOL; (* AT %MW21011.9 *)
    R101_3축_프론트_M_O_RB_4차_작업완료_리셋 : BOOL; (* AT %MW21012.3 *)
    R101_3축_프론트_M_O_RB_4차_진입OK : BOOL; (* AT %MW21011.10 *)
    R101_3축_프론트_M_O_RB_5차_작업완료_리셋 : BOOL; (* AT %MW21012.4 *)
    R101_3축_프론트_M_O_RB_5차_진입OK : BOOL; (* AT %MW21011.11 *)
    R101_3축_프론트_M_O_RB_6차_작업완료_리셋 : BOOL; (* AT %MW21012.5 *)
    R101_3축_프론트_M_O_RB_6차_진입OK : BOOL; (* AT %MW21011.12 *)
    R101_3축_프론트_M_O_RB_7차_작업완료_리셋 : BOOL; (* AT %MW21012.6 *)
    R101_3축_프론트_M_O_RB_7차_진입OK : BOOL; (* AT %MW21011.13 *)
    R101_3축_프론트_M_O_RB_ATD_OK : BOOL; (* AT %MW21010.6 *)
    R101_3축_프론트_M_O_RB_PLT_10_진입OK : BOOL; (* AT %MW21013.10 *)
    R101_3축_프론트_M_O_RB_PLT_11_진입OK : BOOL; (* AT %MW21013.11 *)
    R101_3축_프론트_M_O_RB_PLT_12_진입OK : BOOL; (* AT %MW21013.12 *)
    R101_3축_프론트_M_O_RB_PLT_1_진입OK : BOOL; (* AT %MW21013.1 *)
    R101_3축_프론트_M_O_RB_PLT_2_진입OK : BOOL; (* AT %MW21013.2 *)
    R101_3축_프론트_M_O_RB_PLT_3_진입OK : BOOL; (* AT %MW21013.3 *)
    R101_3축_프론트_M_O_RB_PLT_4_진입OK : BOOL; (* AT %MW21013.4 *)
    R101_3축_프론트_M_O_RB_PLT_5_진입OK : BOOL; (* AT %MW21013.5 *)
    R101_3축_프론트_M_O_RB_PLT_6_진입OK : BOOL; (* AT %MW21013.6 *)
    R101_3축_프론트_M_O_RB_PLT_7_진입OK : BOOL; (* AT %MW21013.7 *)
    R101_3축_프론트_M_O_RB_PLT_8_진입OK : BOOL; (* AT %MW21013.8 *)
    R101_3축_프론트_M_O_RB_PLT_9_진입OK : BOOL; (* AT %MW21013.9 *)
    R101_3축_프론트_M_O_RB_PLT_카운터리셋_보조 : BOOL; (* AT %MW21010.10 *)
    R101_3축_프론트_M_O_RB_RESTART_OK : BOOL; (* AT %MW21010.2 *)
    R101_3축_프론트_M_O_RB_START_OK : BOOL; (* AT %MW21010.0 *)
    R101_3축_프론트_M_O_RB_TEST_MODE_5000회 : BOOL; (* AT %MW21010.12 *)
    R101_3축_프론트_M_O_RB_TIP_교체_시작 : BOOL; (* AT %MW21010.7 *)
    R101_3축_프론트_M_O_RB_TIP_교체_완료 : BOOL; (* AT %MW21010.8 *)
    R101_3축_프론트_M_O_RB_VIP_MODE : BOOL; (* AT %MW21010.11 *)
    R101_3축_프론트_M_O_RB_냉각수_차단_요청 : BOOL; (* AT %MW21010.9 *)
    R101_3축_프론트_M_O_RB_진입OK_AX차종 : BOOL; (* AT %MW21011.0 *)
    R101_3축_프론트_M_O_RB_진입OK_B차종 : BOOL; (* AT %MW21011.1 *)
    R101_3축_프론트_M_O_RB_진입OK_C차종 : BOOL; (* AT %MW21011.2 *)
    R101_3축_프론트_M_O_RB_진입OK_D차종 : BOOL; (* AT %MW21011.3 *)
    R101_3축_프론트_M_O_RB_진입OK_E차종 : BOOL; (* AT %MW21011.4 *)
    R101_3축_프론트_M_O_RB_진입OK_F차종 : BOOL; (* AT %MW21011.5 *)
    R101_3축_프론트_M_O_RB_진입OK_G차종 : BOOL; (* AT %MW21011.6 *)
    R101_3축_프론트_M_O_RB_진입OK_H차종 : BOOL; (* AT %MW21011.7 *)
    R101_3축_프론트_M_O_RB_최종_작업완료_리셋 : BOOL; (* AT %MW21010.5 *)
    R101_3축_프론트_M_O_RB_프로그램_OK : BOOL; (* AT %MW21010.1 *)
    R101_3축_프론트_M_RB_PROG_NO : WORD; (* AT %MW20014 *)
    R101_3축_프론트_O_RB_OUTPUT : ARRAY[0..3] OF WORD; (* AT %MW94010 *)
    S101_M_수동_모드 : BOOL; (* AT %MW1000.3 *)
    S101_M_자동_START : BOOL; (* AT %MW1000.5 *)
    S101_M_자동_운전중 : BOOL; (* AT %MW1000.4 *)
    S101_M_작업_완료 : BOOL; (* AT %MW1001.0 *)
    S101_M_전체_3축_로봇1차_작업완료 : BOOL; (* AT %MW1001.1 *)
    S101_M_전체_용접로보트_1차_작업완료 : BOOL; (* AT %MW1001.8 *)
    S101_M_전체_용접로보트_최종_작업완료 : BOOL; (* AT %MW1001.9 *)
    S101_M_차종1_AX : BOOL; (* AT %MW10021.0 *) (* S101_M_차종1_AX *)
    S101_M_총괄_이상 : BOOL; (* AT %MW1009.0 *)
    셔틀_M_작업완료 : BOOL; (* AT %MW501.0 *)
    전체_M_GATE_비상정지_정상 : BOOL; (* AT %MW308.4 *)
    전체_M_운전준비_보조 : BOOL; (* AT %MW308.5 *)
    전체_M_이상_리셋 : BOOL; (* AT %MW308.2 *) (* 전체 M 이상 리셋 *)
    전체_공정_M_총괄_비상정지_정상 : BOOL; (* AT %MW304.1 *) (* 전체 공정 M 총괄 비상정지 정상 *)
END_VAR
VAR
    INST : FB494_Robot_Hyundai_HMMI_v1;
    INST1 : FB494_Robot_Hyundai_HMMI_v1;
    INST2 : FB494_Robot_Hyundai_HMMI_v1;
    _작업완료_SET_BIT : BOOL;
END_VAR
(* ladder body could not be read *)
END_PROGRAM

PROGRAM S101_용접타점수 (* task: 스캔 프로그램 *)
VAR_EXTERNAL
    R101_1_I_RB_용접타점수 : WORD; (* AT %MW84075 *)
    R101_1_M_AX_차종_용접타점수 : WORD; (* AT %MW8110 *) (* R101_1_M_AX_차종_용접타점수 *)
    R101_1_M_I_RB_1차_작업완료 : BOOL; (* AT %MW20071.2 *)
    R101_1_M_용접완료 : BOOL; (* AT %MW1011.1 *)
    R101_1_M_용접타점수_OK : BOOL; (* AT %MW1011.5 *)
    R101_2_I_RB_용접타점수 : WORD; (* AT %MW84065 *)
    R101_2_M_AX_차종_용접타점수 : WORD; (* AT %MW8120 *) (* R101_2_M_AX_차종_용접타점수 *)
    R101_2_M_I_RB_1차_작업완료 : BOOL; (* AT %MW20061.2 *)
    R101_2_M_용접완료 : BOOL; (* AT %MW1011.2 *)
    R101_2_M_용접타점수_OK : BOOL; (* AT %MW1011.6 *)
    S101_M_전체_용접완료 : BOOL; (* AT %MW1011.0 *)
    S101_M_차종1_AX : BOOL; (* AT %MW10021.0 *) (* S101_M_차종1_AX *)
END_VAR
VAR
    _t1 : BOOL;
    _t2 : BOOL;
END_VAR

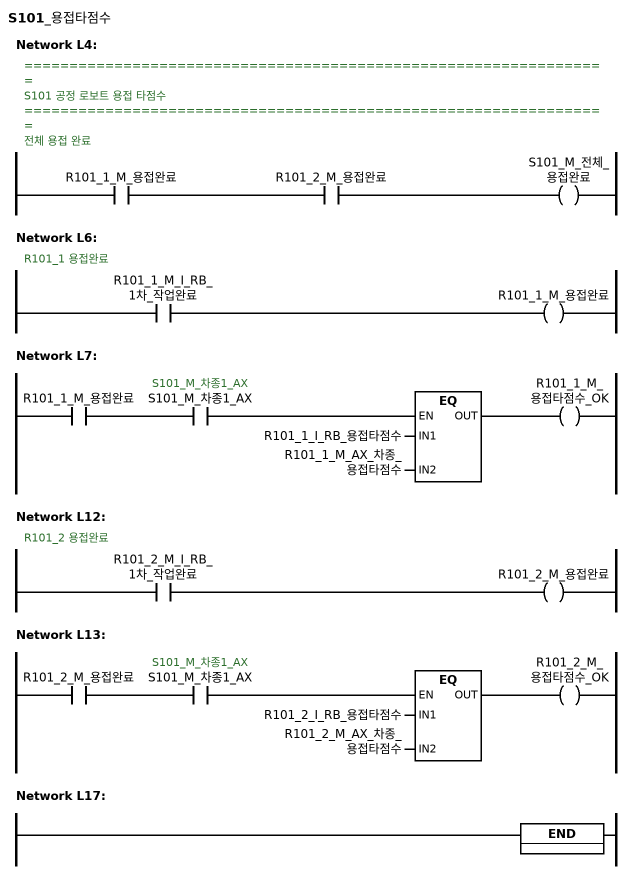
(* ================================================================= *)
(* S101 공정 로보트 용접 타점수 *)
(* ================================================================= *)
(* 전체 용접 완료 *)
(* Rung L4 *)
S101_M_전체_용접완료 := R101_1_M_용접완료 AND R101_2_M_용접완료;
(* R101_1 용접완료 *)
(* Rung L6 *)
R101_1_M_용접완료 := R101_1_M_I_RB_1차_작업완료;
(* Rung L7 *)
IF R101_1_M_용접완료 AND S101_M_차종1_AX THEN _t1 := R101_1_I_RB_용접타점수 = R101_1_M_AX_차종_용접타점수; END_IF;
R101_1_M_용접타점수_OK := _t1;
(* R101_2 용접완료 *)
(* Rung L12 *)
R101_2_M_용접완료 := R101_2_M_I_RB_1차_작업완료;
(* Rung L13 *)
IF R101_2_M_용접완료 AND S101_M_차종1_AX THEN _t2 := R101_2_I_RB_용접타점수 = R101_2_M_AX_차종_용접타점수; END_IF;
R101_2_M_용접타점수_OK := _t2;
(* Rung L17 *)
END();
END_PROGRAM

PROGRAM S101_이상 (* task: 스캔 프로그램 *)
VAR
    INST10 : TON;
    INST11 : TON;
    INST12 : TON;
    INST13 : TON;
    INST14 : TON;
    INST15 : TON;
    INST16 : TON;
    INST17 : TON;
    INST18 : TON;
    INST19 : TON;
    INST20 : TON;
    INST21 : TON;
    INST22 : TON;
    INST23 : TON;
    INST24 : TON;
    INST25 : TON;
    INST26 : TON;
    INST27 : TON;
    INST28 : TON;
    INST29 : TON;
    INST30 : TON;
    INST31 : TON;
    INST32 : TON;
    INST33 : TON;
    INST34 : TON;
    INST35 : TON;
    INST36 : TON;
    INST37 : TON;
    INST38 : TON;
    INST39 : TON;
    INST40 : TON;
    INST41 : TON;
    INST42 : TON;
    INST43 : TON;
    INST8 : TON;
    INST9 : TON;
END_VAR
VAR_EXTERNAL
    R101_1_1_M_RB_통신이상 : BOOL; (* AT %MW1024.10 *)
    R101_1_M_RB_통신이상 : BOOL; (* AT %MW1024.11 *)
    R101_1_M_용접완료 : BOOL; (* AT %MW1011.1 *)
    R101_1_M_용접타점수_OK : BOOL; (* AT %MW1011.5 *)
    R101_1_M_용접타점수_이상 : BOOL; (* AT %MW1011.10 *)
    R101_2_M_RB_통신이상 : BOOL; (* AT %MW1024.12 *)
    R101_2_M_용접완료 : BOOL; (* AT %MW1011.2 *)
    R101_2_M_용접타점수_OK : BOOL; (* AT %MW1011.6 *)
    R101_2_M_용접타점수_이상 : BOOL; (* AT %MW1011.11 *)
    R101_3_M_RB_통신이상 : BOOL; (* AT %MW1024.13 *)
    S101_6_10_PLC_BOX_CP_TRIP : BOOL; (* AT %MW86102.15 *) (* 입력 접점 15 *)
    S101_M_3축로보트_CTR_통신이상 : BOOL; (* AT %MW1024.8 *)
    S101_M_3축로보트_FRT_통신이상 : BOOL; (* AT %MW1024.7 *)
    S101_M_3축로보트_RR_통신이상 : BOOL; (* AT %MW1024.9 *)
    S101_M_APRON_LH_제품감지_이상 : BOOL; (* AT %MW1014.0 *)
    S101_M_APRON_RH_안착OK_POS : BOOL; (* AT %MW1004.9 *)
    S101_M_APRON_RH_제품감지_이상 : BOOL; (* AT %MW1014.1 *)
    S101_M_APRON_랙방1_2_통신이상 : BOOL; (* AT %MW1024.1 *)
    S101_M_APRON_랙방3_4_통신이상 : BOOL; (* AT %MW1024.2 *)
    S101_M_AX_래치_전진_LS_이상 : BOOL; (* AT %MW1100.5 *)
    S101_M_AX_래치_후진_LS_이상 : BOOL; (* AT %MW1100.6 *)
    S101_M_DASH_제품감지_이상 : BOOL; (* AT %MW1014.2 *)
    S101_M_DASH_클램프_전진_LS_이상 : BOOL; (* AT %MW1105.5 *)
    S101_M_DASH_클램프_후진_LS_이상 : BOOL; (* AT %MW1105.6 *)
    S101_M_SHIFT_전진_LS_이상 : BOOL; (* AT %MW1101.5 *)
    S101_M_SHIFT_후진_LS_이상 : BOOL; (* AT %MW1101.6 *)
    S101_M_STN_DASH_로딩완료 : BOOL; (* AT %MW1001.12 *)
    S101_M_STN_LH_로딩완료 : BOOL; (* AT %MW1001.10 *)
    S101_M_STN_RH_로딩완료 : BOOL; (* AT %MW1001.11 *)
    S101_M_공정_APRON_제품감지_ON : BOOL; (* AT %MW1001.3 *)
    S101_M_공정_간섭무 : BOOL; (* AT %MW1004.1 *)
    S101_M_공정_통신이상 : BOOL; (* AT %MW1024.0 *)
    S101_M_서보1_통신이상 : BOOL; (* AT %MW1024.4 *)
    S101_M_서보2_통신이상 : BOOL; (* AT %MW1024.5 *)
    S101_M_서보3_통신이상 : BOOL; (* AT %MW1024.6 *)
    S101_M_서보판넬_통신이상 : BOOL; (* AT %MW1024.3 *)
    S101_M_차종1_AX : BOOL; (* AT %MW10021.0 *) (* S101_M_차종1_AX *)
    S101_M_차종3_LHD : BOOL; (* AT %MW10021.14 *) (* S101_M_차종3_LHD *)
    S101_M_차종3_RHD : BOOL; (* AT %MW10021.15 *) (* S101_M_차종3_RHD *)
    S101_M_총괄_CP_이상 : BOOL; (* AT %MW1009.7 *)
    S101_M_총괄_CT_이상 : BOOL; (* AT %MW1010.4 *)
    S101_M_총괄_EOCR_이상 : BOOL; (* AT %MW1009.8 *)
    S101_M_총괄_INV_이상 : BOOL; (* AT %MW1009.9 *)
    S101_M_총괄_LS_이상 : BOOL; (* AT %MW1009.15 *)
    S101_M_총괄_MATCH_이상 : BOOL; (* AT %MW1010.0 *)
    S101_M_총괄_MC_이상 : BOOL; (* AT %MW1009.13 *)
    S101_M_총괄_NFB_이상 : BOOL; (* AT %MW1009.11 *)
    S101_M_총괄_ROBOT_이상 : BOOL; (* AT %MW1010.1 *)
    S101_M_총괄_SAFETY_이상 : BOOL; (* AT %MW1009.2 *)
    S101_M_총괄_공기압_이상 : BOOL; (* AT %MW1009.3 *)
    S101_M_총괄_비상정지_이상 : BOOL; (* AT %MW1009.1 *)
    S101_M_총괄_사양_이상 : BOOL; (* AT %MW1009.6 *)
    S101_M_총괄_오버런_이상 : BOOL; (* AT %MW1009.12 *)
    S101_M_총괄_용점타점수_이상 : BOOL; (* AT %MW1010.2 *)
    S101_M_총괄_이상 : BOOL; (* AT %MW1009.0 *)
    S101_M_총괄_제품감지_이상 : BOOL; (* AT %MW1009.4 *)
    S101_M_총괄_차종_이상 : BOOL; (* AT %MW1009.5 *)
    S101_M_총괄_통신_이상 : BOOL; (* AT %MW1009.14 *)
    S101_M_핀클램프_전진_LS_이상 : BOOL; (* AT %MW1106.5 *)
    S101_M_핀클램프_후진_LS_이상 : BOOL; (* AT %MW1106.6 *)
    S101_PRS_I_AX_APRON_LHD_사양감지 : BOOL; (* AT %MW86102.8 *)
    S101_PRS_I_AX_APRON_RHD_사양감지 : BOOL; (* AT %MW86102.9 *)
    S101_PRS_I_AX_DASH_파트_ON : BOOL; (* AT %MW86102.2 *)
    S101_PRS_I_AX_LH_파트_ON : BOOL; (* AT %MW86102.0 *)
    S101_PRS_I_AX_RH_파트_ON : BOOL; (* AT %MW86102.1 *)
    S101_공기압_AIR_CHECK : BOOL; (* AT %MW86102.14 *) (* 입력 접점 14 *)
    _0004_EB01_CFG_ER : BOOL; (* AT %MX59360 *) (* EB 구성 에러 *)
    _0004_EB01_DEER : BOOL; (* AT %MX59361 *) (* EB 운전 중 탈락 *)
    _0004_EB04_CFG_ER : BOOL; (* AT %MX59400 *) (* EB 구성 에러 *)
    _0004_EB04_DEER : BOOL; (* AT %MX59401 *) (* EB 운전 중 탈락 *)
    _0004_EB05_CFG_ER : BOOL; (* AT %MX59440 *) (* EB 구성 에러 *)
    _0004_EB05_DEER : BOOL; (* AT %MX59441 *) (* EB 운전 중 탈락 *)
    _0004_EB06_CFG_ER : BOOL; (* AT %MX59480 *) (* EB 구성 에러 *)
    _0004_EB06_DEER : BOOL; (* AT %MX59481 *) (* EB 운전 중 탈락 *)
    _0004_EB07_CFG_ER : BOOL; (* AT %MX59520 *) (* EB 구성 에러 *)
    _0004_EB07_DEER : BOOL; (* AT %MX59521 *) (* EB 운전 중 탈락 *)
    _0005_EB11_S00_SVC_ER : BOOL; (* AT %MW185024.7 *) (* 통신 서비스 에러 *)
    _0005_EB11_S01_SVC_ER : BOOL; (* AT %MW185024.15 *) (* 통신 서비스 에러 *)
    _0005_EB12_S00_SVC_ER : BOOL; (* AT %MW185058.7 *) (* 통신 서비스 에러 *)
    _0005_EB12_S01_SVC_ER : BOOL; (* AT %MW185058.15 *) (* 통신 서비스 에러 *)
    _0005_EB13_S00_SVC_ER : BOOL; (* AT %MW185092.7 *) (* 통신 서비스 에러 *)
    _0005_EB13_S01_SVC_ER : BOOL; (* AT %MW185092.15 *) (* 통신 서비스 에러 *)
    _0005_EB20_CFG_ER : BOOL; (* AT %MW185124.0 *) (* EB 구성 에러 *)
    _0005_EB20_DEER : BOOL; (* AT %MW185124.1 *) (* EB 운전 중 탈락 *)
    _0005_EB20_IO_DEER : BOOL; (* AT %MW185125.2 *) (* EB IO 탈락 에러 *)
    _0005_EB20_IO_TYER : BOOL; (* AT %MW185125.1 *) (* EB IO 타입 에러 *)
    _0006_EB10_CFG_ER : BOOL; (* AT %MW186022.0 *) (* EB 구성 에러 *)
    _0006_EB10_DEER : BOOL; (* AT %MW186022.1 *) (* EB 운전 중 탈락 *)
    _0006_EB10_IO_DEER : BOOL; (* AT %MW186023.2 *) (* EB IO 탈락 에러 *)
    _0006_EB10_IO_TYER : BOOL; (* AT %MW186023.1 *) (* EB IO 타입 에러 *)
    _0007_EB21_CFG_ER : BOOL; (* AT %MW187028.0 *) (* EB 구성 에러 *)
    _0007_EB21_DEER : BOOL; (* AT %MW187028.1 *) (* EB 운전 중 탈락 *)
    _0007_EB21_IO_DEER : BOOL; (* AT %MW187029.2 *) (* EB IO 탈락 에러 *)
    _0007_EB21_IO_TYER : BOOL; (* AT %MW187029.1 *) (* EB IO 타입 에러 *)
    전체_M_이상_리셋 : BOOL; (* AT %MW308.2 *) (* 전체 M 이상 리셋 *)
END_VAR

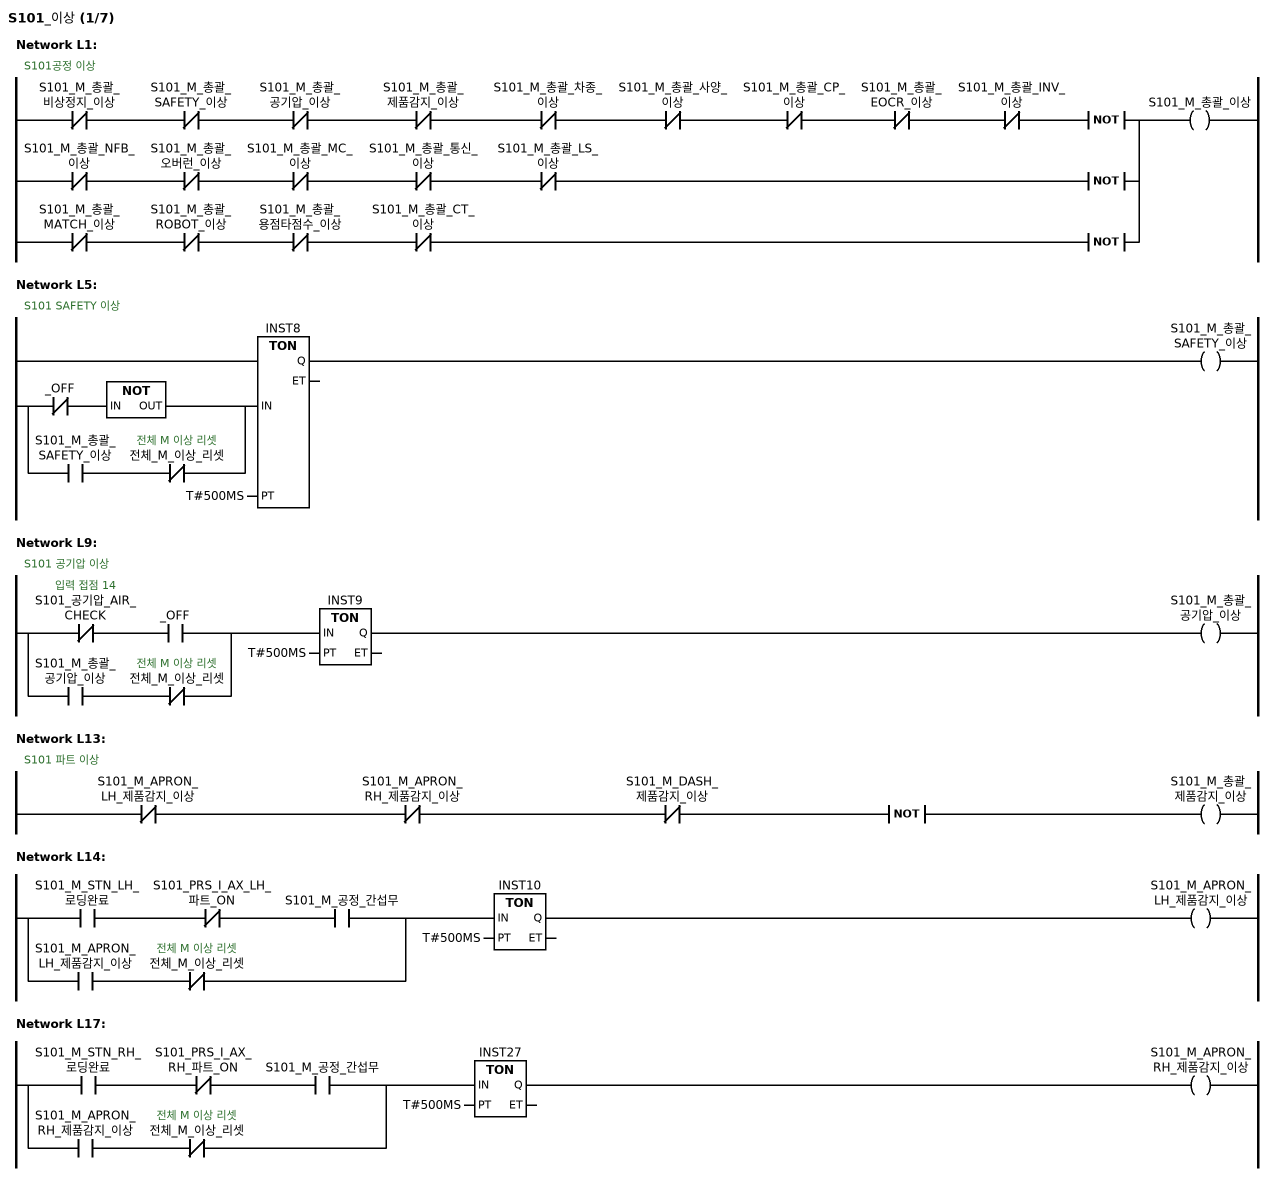
(* S101공정 이상 *)
(* Rung L1 *)
S101_M_총괄_이상 := NOT (NOT S101_M_총괄_비상정지_이상 AND NOT S101_M_총괄_SAFETY_이상 AND NOT S101_M_총괄_공기압_이상 AND NOT S101_M_총괄_제품감지_이상 AND NOT S101_M_총괄_차종_이상 AND NOT S101_M_총괄_사양_이상 AND NOT S101_M_총괄_CP_이상 AND NOT S101_M_총괄_EOCR_이상 AND NOT S101_M_총괄_INV_이상) OR NOT (NOT S101_M_총괄_NFB_이상 AND NOT S101_M_총괄_오버런_이상 AND NOT S101_M_총괄_MC_이상 AND NOT S101_M_총괄_통신_이상 AND NOT S101_M_총괄_LS_이상) OR NOT (NOT S101_M_총괄_MATCH_이상 AND NOT S101_M_총괄_ROBOT_이상 AND NOT S101_M_총괄_용점타점수_이상 AND NOT S101_M_총괄_CT_이상);
(* S101 SAFETY 이상 *)
(* Rung L5 *)
INST8(IN := (NOT (NOT _OFF)) OR (S101_M_총괄_SAFETY_이상 AND NOT 전체_M_이상_리셋), PT := T#500MS);
S101_M_총괄_SAFETY_이상 := INST8.Q;
(* S101 공기압 이상 *)
(* Rung L9 *)
INST9(IN := (NOT S101_공기압_AIR_CHECK AND _OFF) OR (S101_M_총괄_공기압_이상 AND NOT 전체_M_이상_리셋), PT := T#500MS);
S101_M_총괄_공기압_이상 := INST9.Q;
(* S101 파트 이상 *)
(* Rung L13 *)
S101_M_총괄_제품감지_이상 := NOT (NOT S101_M_APRON_LH_제품감지_이상 AND NOT S101_M_APRON_RH_제품감지_이상 AND NOT S101_M_DASH_제품감지_이상);
(* Rung L14 *)
INST10(IN := (S101_M_STN_LH_로딩완료 AND NOT S101_PRS_I_AX_LH_파트_ON AND S101_M_공정_간섭무) OR (S101_M_APRON_LH_제품감지_이상 AND NOT 전체_M_이상_리셋), PT := T#500MS);
S101_M_APRON_LH_제품감지_이상 := INST10.Q;
(* Rung L17 *)
INST27(IN := (S101_M_STN_RH_로딩완료 AND NOT S101_PRS_I_AX_RH_파트_ON AND S101_M_공정_간섭무) OR (S101_M_APRON_RH_제품감지_이상 AND NOT 전체_M_이상_리셋), PT := T#500MS);
S101_M_APRON_RH_제품감지_이상 := INST27.Q;

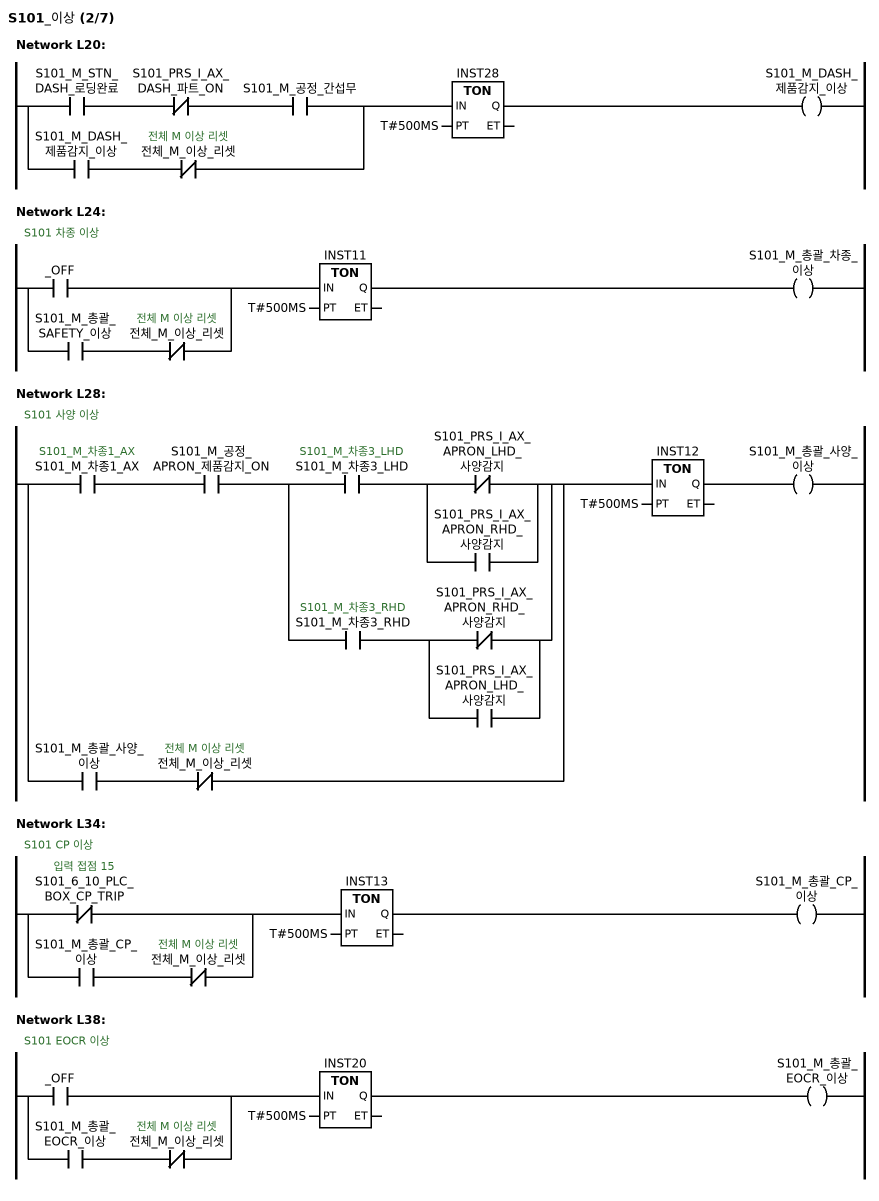
(* Rung L20 *)
INST28(IN := (S101_M_STN_DASH_로딩완료 AND NOT S101_PRS_I_AX_DASH_파트_ON AND S101_M_공정_간섭무) OR (S101_M_DASH_제품감지_이상 AND NOT 전체_M_이상_리셋), PT := T#500MS);
S101_M_DASH_제품감지_이상 := INST28.Q;
(* S101 차종 이상 *)
(* Rung L24 *)
INST11(IN := _OFF OR (S101_M_총괄_SAFETY_이상 AND NOT 전체_M_이상_리셋), PT := T#500MS);
S101_M_총괄_차종_이상 := INST11.Q;
(* S101 사양 이상 *)
(* Rung L28 *)
INST12(IN := (S101_M_차종1_AX AND S101_M_공정_APRON_제품감지_ON AND ((S101_M_차종3_LHD AND (NOT S101_PRS_I_AX_APRON_LHD_사양감지 OR S101_PRS_I_AX_APRON_RHD_사양감지)) OR (S101_M_차종3_RHD AND (NOT S101_PRS_I_AX_APRON_RHD_사양감지 OR S101_PRS_I_AX_APRON_LHD_사양감지)))) OR (S101_M_총괄_사양_이상 AND NOT 전체_M_이상_리셋), PT := T#500MS);
S101_M_총괄_사양_이상 := INST12.Q;
(* S101 CP 이상 *)
(* Rung L34 *)
INST13(IN := NOT S101_6_10_PLC_BOX_CP_TRIP OR (S101_M_총괄_CP_이상 AND NOT 전체_M_이상_리셋), PT := T#500MS);
S101_M_총괄_CP_이상 := INST13.Q;
(* S101 EOCR 이상 *)
(* Rung L38 *)
INST20(IN := _OFF OR (S101_M_총괄_EOCR_이상 AND NOT 전체_M_이상_리셋), PT := T#500MS);
S101_M_총괄_EOCR_이상 := INST20.Q;

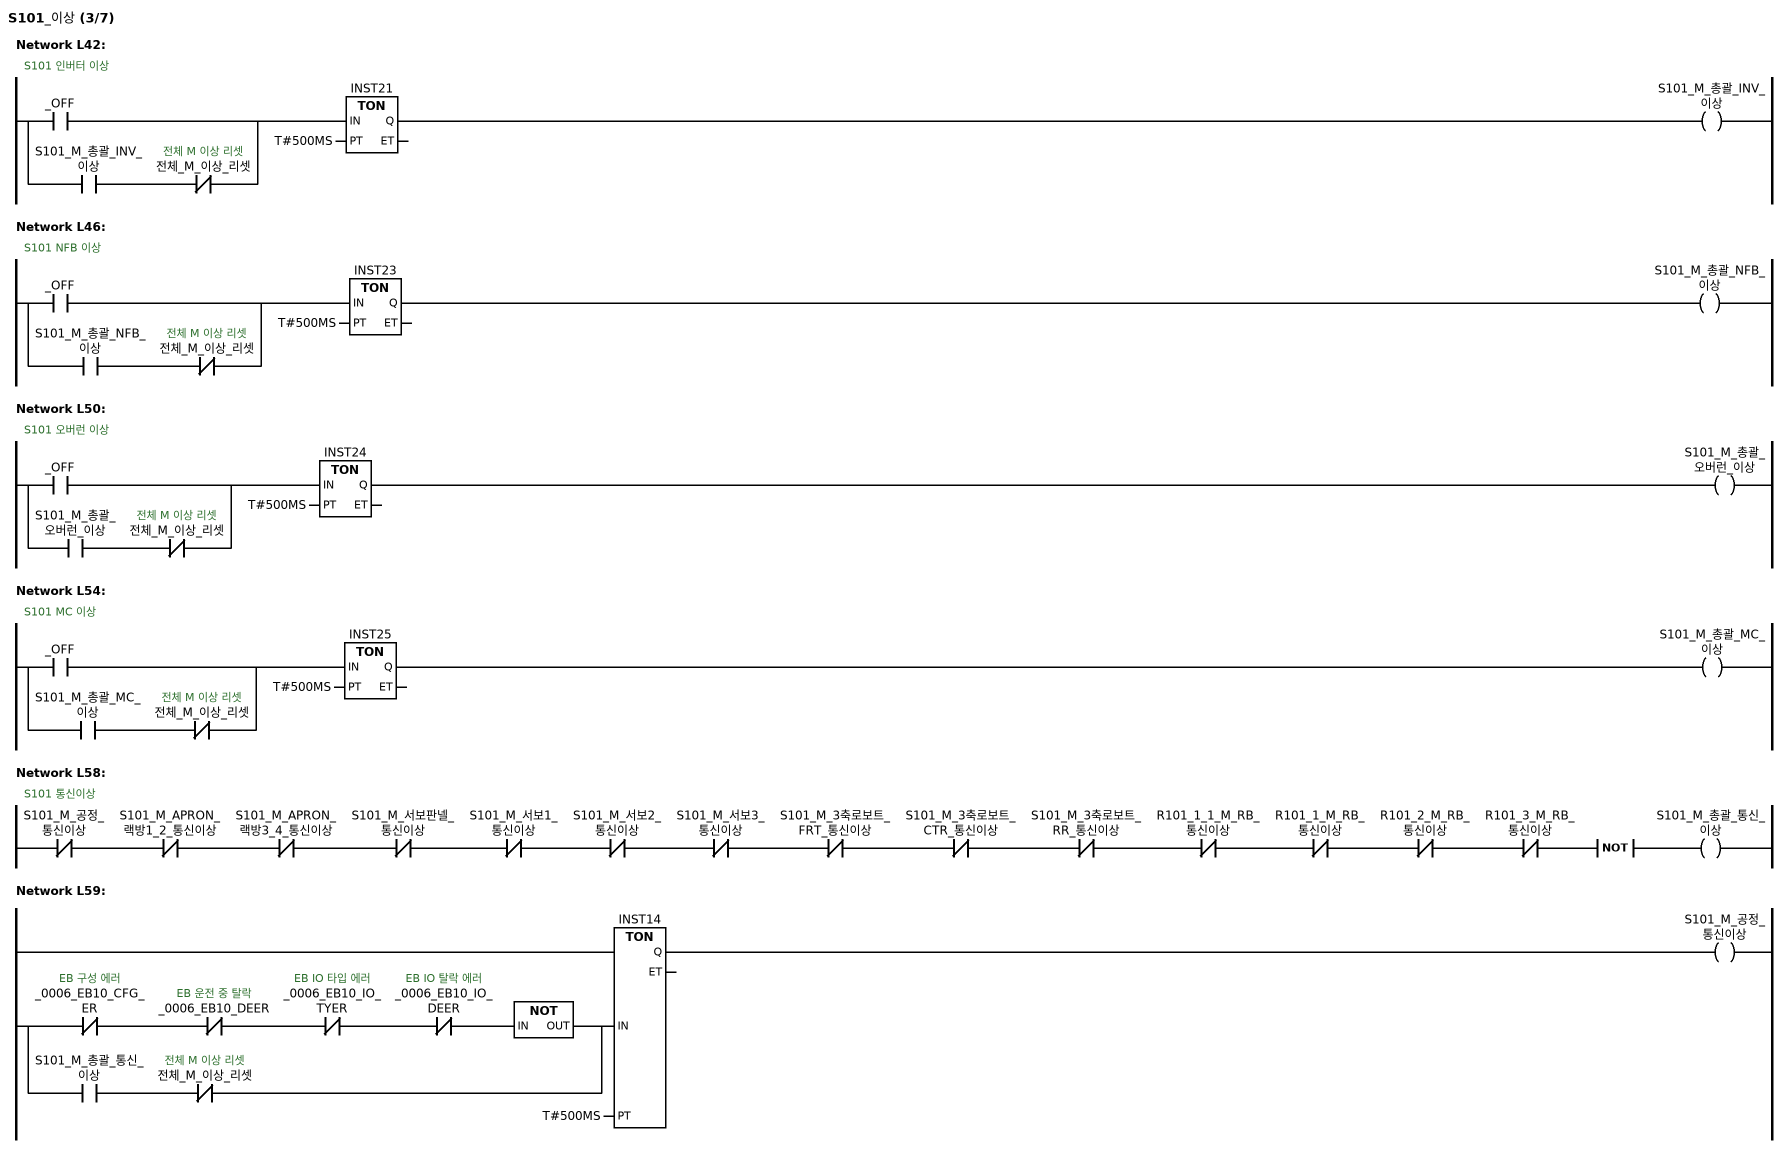
(* S101 인버터 이상 *)
(* Rung L42 *)
INST21(IN := _OFF OR (S101_M_총괄_INV_이상 AND NOT 전체_M_이상_리셋), PT := T#500MS);
S101_M_총괄_INV_이상 := INST21.Q;
(* S101 NFB 이상 *)
(* Rung L46 *)
INST23(IN := _OFF OR (S101_M_총괄_NFB_이상 AND NOT 전체_M_이상_리셋), PT := T#500MS);
S101_M_총괄_NFB_이상 := INST23.Q;
(* S101 오버런 이상 *)
(* Rung L50 *)
INST24(IN := _OFF OR (S101_M_총괄_오버런_이상 AND NOT 전체_M_이상_리셋), PT := T#500MS);
S101_M_총괄_오버런_이상 := INST24.Q;
(* S101 MC 이상 *)
(* Rung L54 *)
INST25(IN := _OFF OR (S101_M_총괄_MC_이상 AND NOT 전체_M_이상_리셋), PT := T#500MS);
S101_M_총괄_MC_이상 := INST25.Q;
(* S101 통신이상 *)
(* Rung L58 *)
S101_M_총괄_통신_이상 := NOT (NOT S101_M_공정_통신이상 AND NOT S101_M_APRON_랙방1_2_통신이상 AND NOT S101_M_APRON_랙방3_4_통신이상 AND NOT S101_M_서보판넬_통신이상 AND NOT S101_M_서보1_통신이상 AND NOT S101_M_서보2_통신이상 AND NOT S101_M_서보3_통신이상 AND NOT S101_M_3축로보트_FRT_통신이상 AND NOT S101_M_3축로보트_CTR_통신이상 AND NOT S101_M_3축로보트_RR_통신이상 AND NOT R101_1_1_M_RB_통신이상 AND NOT R101_1_M_RB_통신이상 AND NOT R101_2_M_RB_통신이상 AND NOT R101_3_M_RB_통신이상);
(* Rung L59 *)
INST14(IN := (NOT (NOT _0006_EB10_CFG_ER AND NOT _0006_EB10_DEER AND NOT _0006_EB10_IO_TYER AND NOT _0006_EB10_IO_DEER)) OR (S101_M_총괄_통신_이상 AND NOT 전체_M_이상_리셋), PT := T#500MS);
S101_M_공정_통신이상 := INST14.Q;

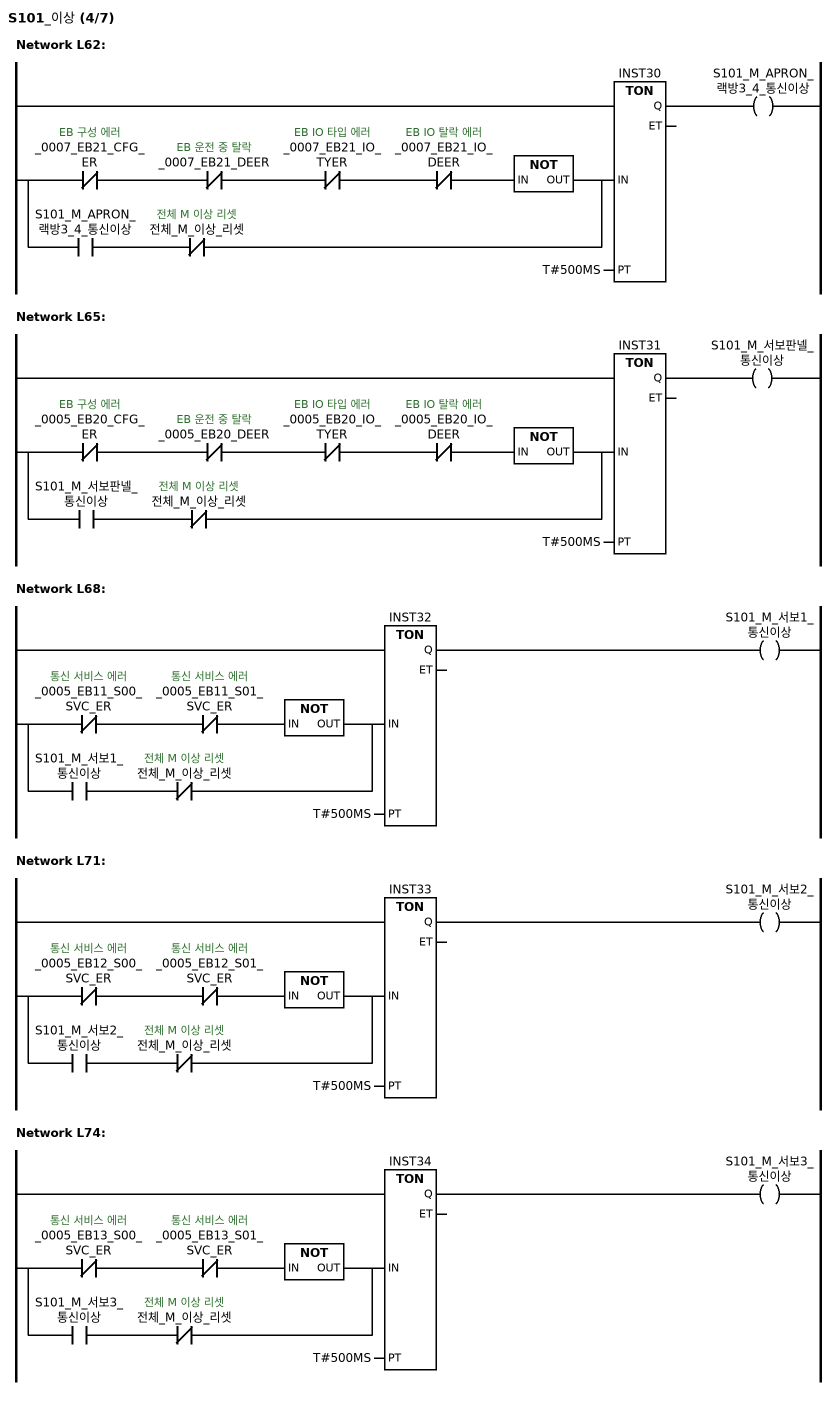
(* Rung L62 *)
INST30(IN := (NOT (NOT _0007_EB21_CFG_ER AND NOT _0007_EB21_DEER AND NOT _0007_EB21_IO_TYER AND NOT _0007_EB21_IO_DEER)) OR (S101_M_APRON_랙방3_4_통신이상 AND NOT 전체_M_이상_리셋), PT := T#500MS);
S101_M_APRON_랙방3_4_통신이상 := INST30.Q;
(* Rung L65 *)
INST31(IN := (NOT (NOT _0005_EB20_CFG_ER AND NOT _0005_EB20_DEER AND NOT _0005_EB20_IO_TYER AND NOT _0005_EB20_IO_DEER)) OR (S101_M_서보판넬_통신이상 AND NOT 전체_M_이상_리셋), PT := T#500MS);
S101_M_서보판넬_통신이상 := INST31.Q;
(* Rung L68 *)
INST32(IN := (NOT (NOT _0005_EB11_S00_SVC_ER AND NOT _0005_EB11_S01_SVC_ER)) OR (S101_M_서보1_통신이상 AND NOT 전체_M_이상_리셋), PT := T#500MS);
S101_M_서보1_통신이상 := INST32.Q;
(* Rung L71 *)
INST33(IN := (NOT (NOT _0005_EB12_S00_SVC_ER AND NOT _0005_EB12_S01_SVC_ER)) OR (S101_M_서보2_통신이상 AND NOT 전체_M_이상_리셋), PT := T#500MS);
S101_M_서보2_통신이상 := INST33.Q;
(* Rung L74 *)
INST34(IN := (NOT (NOT _0005_EB13_S00_SVC_ER AND NOT _0005_EB13_S01_SVC_ER)) OR (S101_M_서보3_통신이상 AND NOT 전체_M_이상_리셋), PT := T#500MS);
S101_M_서보3_통신이상 := INST34.Q;

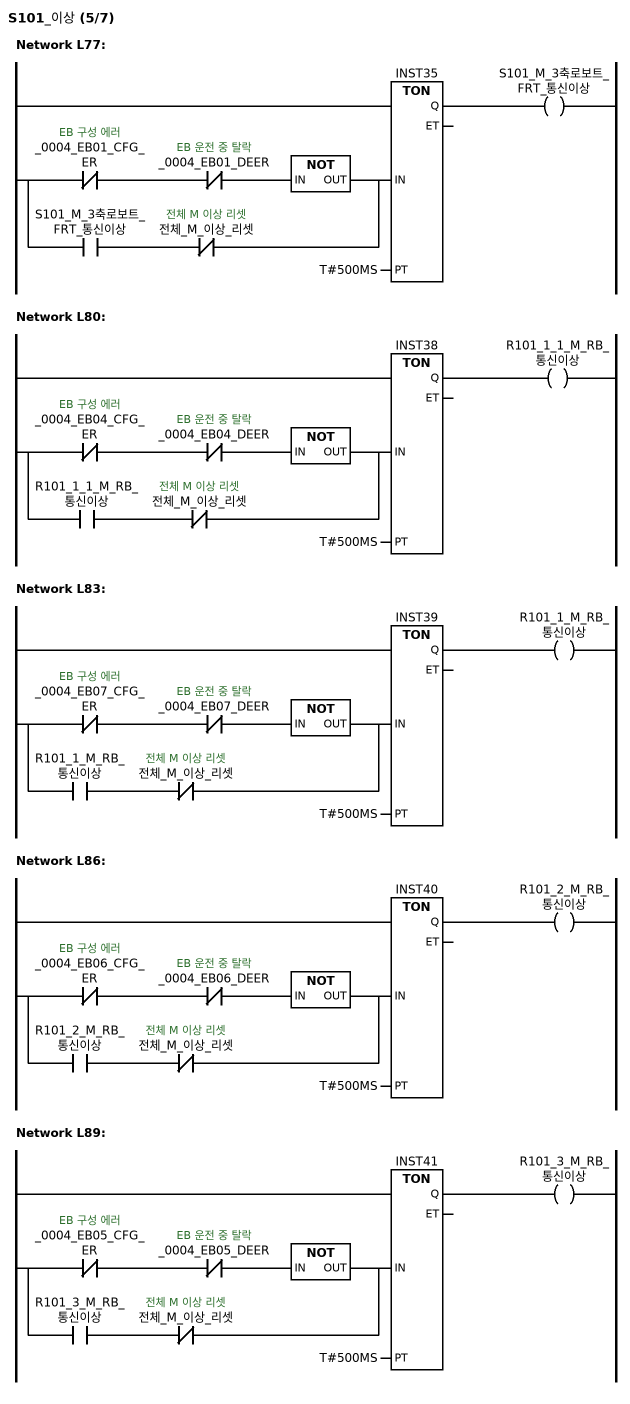
(* Rung L77 *)
INST35(IN := (NOT (NOT _0004_EB01_CFG_ER AND NOT _0004_EB01_DEER)) OR (S101_M_3축로보트_FRT_통신이상 AND NOT 전체_M_이상_리셋), PT := T#500MS);
S101_M_3축로보트_FRT_통신이상 := INST35.Q;
(* Rung L80 *)
INST38(IN := (NOT (NOT _0004_EB04_CFG_ER AND NOT _0004_EB04_DEER)) OR (R101_1_1_M_RB_통신이상 AND NOT 전체_M_이상_리셋), PT := T#500MS);
R101_1_1_M_RB_통신이상 := INST38.Q;
(* Rung L83 *)
INST39(IN := (NOT (NOT _0004_EB07_CFG_ER AND NOT _0004_EB07_DEER)) OR (R101_1_M_RB_통신이상 AND NOT 전체_M_이상_리셋), PT := T#500MS);
R101_1_M_RB_통신이상 := INST39.Q;
(* Rung L86 *)
INST40(IN := (NOT (NOT _0004_EB06_CFG_ER AND NOT _0004_EB06_DEER)) OR (R101_2_M_RB_통신이상 AND NOT 전체_M_이상_리셋), PT := T#500MS);
R101_2_M_RB_통신이상 := INST40.Q;
(* Rung L89 *)
INST41(IN := (NOT (NOT _0004_EB05_CFG_ER AND NOT _0004_EB05_DEER)) OR (R101_3_M_RB_통신이상 AND NOT 전체_M_이상_리셋), PT := T#500MS);
R101_3_M_RB_통신이상 := INST41.Q;

